762.00 BOOL  ; RK_16 U6_Z 激光焊接Z轴待机位[SW]
762.01 BOOL  ; RK_16 U6_Z 激光焊接Z轴#1移载焊接位[SW]
762.02 BOOL  ; RK_16 U6_Z 激光焊接Z轴#2移载焊接位[SW]
762.03 BOOL  ; 备用[SW]
762.04 BOOL  ; 备用[SW]
762.05 BOOL  ; 备用[SW]
762.06 BOOL  ; 备用[SW]
762.07 BOOL  ; 备用[SW]
762.08 BOOL  ; 备用[SW]
762.09 BOOL  ; 备用[SW]
762.10 BOOL  ; RK_16 U6_Z 激光焊接Z轴回原点[SW]
762.11 BOOL  ; RK_16 U6_Z 激光焊接Z轴JOG+[SW]
762.12 BOOL  ; RK_16 U6_Z 激光焊接Z轴JOG-[SW]
762.13 BOOL  ; RK_16 U6_Z 激光焊接Z轴JOG高速[SW]
762.14 BOOL  ; RK_16 U6_Z 激光焊接Z轴JOG低速[SW]
762.15 BOOL  ; 备用[SW]
763.00 BOOL  ; RK_06 U8_X 电池上下料X轴待机位[SW]
763.01 BOOL  ; RK_06 U8_X 电池上下料X轴铝壳除尘取料位[SW]
763.02 BOOL  ; RK_06 U8_X 电池上下料X轴#1入壳放料位[SW]
763.03 BOOL  ; RK_06 U8_X 电池上下料X轴#2入壳放料位[SW]
763.04 BOOL  ; RK_06 U8_X 电池上下料X轴#1入壳取料位[SW]
763.05 BOOL  ; RK_06 U8_X 电池上下料X轴#2入壳取料位[SW]
763.06 BOOL  ; RK_06 U8_X 电池上下料X轴#1Hipot检测放料位[SW]
763.07 BOOL  ; RK_06 U8_X 电池上下料X轴#2Hipot检测放料位[SW]
763.08 BOOL  ; 备用[SW]
763.09 BOOL  ; 备用[SW]
763.10 BOOL  ; RK_06 U8_X 电池上下料X轴回原点[SW]
763.11 BOOL  ; RK_06 U8_X 电池上下料X轴JOG+[SW]
763.12 BOOL  ; RK_06 U8_X 电池上下料X轴JOG-[SW]
763.13 BOOL  ; RK_06 U8_X 电池上下料X轴JOG高速[SW]
763.14 BOOL  ; RK_06 U8_X 电池上下料X轴JOG低速[SW]
763.15 BOOL  ; 备用[SW]
764.00 BOOL  ; RK_07 U8_Y 铝壳进料X轴等待位[SW]
764.01 BOOL  ; RK_07 U8_Y 铝壳进料X轴取料位[SW]
764.02 BOOL  ; RK_07 U8_Y 铝壳进料X轴放料位[SW]
764.03 BOOL  ; 备用[SW]
764.04 BOOL  ; 备用[SW]
764.05 BOOL  ; 备用[SW]
764.06 BOOL  ; 备用[SW]
764.07 BOOL  ; 备用[SW]
764.08 BOOL  ; 备用[SW]
764.09 BOOL  ; 备用[SW]
764.10 BOOL  ; RK_07 U8_Y 铝壳进料X轴回原点[SW]
764.11 BOOL  ; RK_07 U8_Y 铝壳进料X轴JOG+[SW]
764.12 BOOL  ; RK_07 U8_Y 铝壳进料X轴JOG-[SW]
764.13 BOOL  ; RK_07 U8_Y 铝壳进料X轴JOG高速[SW]
764.14 BOOL  ; RK_07 U8_Y 铝壳进料X轴JOG低速[SW]
764.15 BOOL  ; 备用[SW]
765.00 BOOL  ; RK_07 U8_Z 铝壳上料移载Y轴待料位[SW]
765.01 BOOL  ; RK_07 U8_Z 铝壳上料移载Y轴#1铝壳上料位[SW]
765.02 BOOL  ; RK_07 U8_Z 铝壳上料移载Y轴#2铝壳上料位[SW]
765.03 BOOL  ; RK_07 U8_Z 铝壳上料移载Y轴#3铝壳托盘下料位[SW]
765.04 BOOL  ; RK_07 U8_Z 铝壳上料移载Y轴铝壳取料位[SW]
765.05 BOOL  ; 备用[SW]
765.06 BOOL  ; 备用[SW]
765.07 BOOL  ; 备用[SW]
765.08 BOOL  ; 备用[SW]
765.09 BOOL  ; 备用[SW]
765.10 BOOL  ; RK_07 U8_Z 铝壳上料移载Y轴回原点[SW]
765.11 BOOL  ; RK_07 U8_Z 铝壳上料移载Y轴JOG+[SW]
765.12 BOOL  ; RK_07 U8_Z 铝壳上料移载Y轴JOG-[SW]
765.13 BOOL  ; RK_07 U8_Z 铝壳上料移载Y轴JOG高速[SW]
765.14 BOOL  ; RK_07 U8_Z 铝壳上料移载Y轴JOG低速[SW]
765.15 BOOL  ; 备用[SW]
766.00 BOOL  ; RK_10 U8_U 电池除尘上料X轴待料位[SW]
766.01 BOOL  ; RK_10 U8_U 电池除尘上料X轴#1Hipot检测取料位[SW]
766.02 BOOL  ; RK_10 U8_U 电池除尘上料X轴#2Hipot检测取料位[SW]
766.03 BOOL  ; RK_10 U8_U 电池除尘上料X轴Hipot OK放料位[SW]
766.04 BOOL  ; RK_10 U8_U 电池除尘上料X轴Hipot NG放料位[SW]
766.05 BOOL  ; 备用[SW]
766.06 BOOL  ; 备用[SW]
766.07 BOOL  ; 备用[SW]
766.08 BOOL  ; 备用[SW]
766.09 BOOL  ; 备用[SW]
766.10 BOOL  ; RK_10 U8_U 电池除尘上料X轴回原点[SW]
766.11 BOOL  ; RK_10 U8_U 电池除尘上料X轴JOG+[SW]
766.12 BOOL  ; RK_10 U8_U 电池除尘上料X轴JOG-[SW]
766.13 BOOL  ; RK_10 U8_U 电池除尘上料X轴JOG高速[SW]
766.14 BOOL  ; RK_10 U8_U 电池除尘上料X轴JOG低速[SW]
766.15 BOOL  ; 备用[SW]
787.00 BOOL  ; RK_07 铝壳进料机构X轴当前列数+[SW]
787.01 BOOL  ; RK_07 铝壳进料机构X轴当前列数-[SW]
788.00 BOOL  ; RK_07 铝壳上料移载机构Y轴当前行数+[SW]
788.01 BOOL  ; RK_07 铝壳上料移载机构Y轴当前行数-[SW]
7.00 BOOL  ; 扫码阻挡#1伸出传感器
7.01 BOOL  ; 扫码阻挡#1缩回传感器
7.02 BOOL  ; 扫码阻挡#2伸出传感器
7.03 BOOL  ; 扫码阻挡#2缩回
7.04 BOOL  ; 扫码位有料检测
7.05 BOOL  ; 扫码完成信号
800.00 BOOL  ; RK_02 电芯进料机械手夹爪气缸夹紧位标志[0000.00]
800.01 BOOL  ; RK_02 电芯进料机械手夹爪气缸张开位标志[0000.01]
800.02 BOOL  ; RK_02 电芯进料机械手#1压紧气缸松开位标志[0000.02]
800.03 BOOL  ; RK_02 电芯进料机械手#2压紧气缸松开位标志[0000.03]
800.04 BOOL  ; RK_03 电芯上料机械手夹爪气缸夹紧位标志[0000.04]
800.05 BOOL  ; RK_03 电芯上料机械手夹爪气缸张开位标志[0000.05]
800.06 BOOL  ; RK_03 电芯上料机械手#1压紧气缸松开位标志[0000.06]
800.07 BOOL  ; RK_03 电芯上料机械手#2压紧气缸松开位标志[0000.07]
800.08 BOOL  ; RK_03 电芯上料升降气缸下降位标志[0000.08]
800.09 BOOL  ; RK_03 电芯上料升降气缸上升位标志[0000.09]
800.10 BOOL  ; RK_04 电芯除尘伸缩气缸缩回位标志[0000.10]
800.11 BOOL  ; RK_04 电芯除尘伸缩气缸伸出位标志[0000.11]
800.12 BOOL  ; RK_05 #1入壳滚轮夹紧气缸夹紧位标志[0000.12]
800.13 BOOL  ; RK_05 #1入壳滚轮夹紧气缸松开位标志[0000.13]
800.14 BOOL  ; RK_05 #1入壳铝壳定位平台伸缩气缸缩回位标志[0000.14]
800.15 BOOL  ; RK_05 #1入壳铝壳定位平台伸缩气缸伸出位标志[0000.15]
801.00 BOOL  ; RK_05 #1入壳铝壳定位平台升降气缸上升位标志[0001.00]
801.01 BOOL  ; RK_05 #1入壳铝壳定位平台升降气缸下降位标志[0001.01]
801.02 BOOL  ; RK_05 #1入壳铝壳定位伸缩气缸缩回位标志[0001.02]
801.03 BOOL  ; RK_05 #1入壳铝壳定位伸缩气缸伸出位标志[0001.03]
801.04 BOOL  ; RK_05 #1入壳铝壳定位夹爪气缸夹紧位标志[0001.04]
801.05 BOOL  ; RK_05 #1入壳铝壳定位夹爪气缸张开位标志[0001.05]
801.06 BOOL  ; RK_05 #2入壳滚轮夹紧气缸夹紧位标志[0001.06]
801.07 BOOL  ; RK_05 #2入壳滚轮夹紧气缸松开位标志[0001.07]
801.08 BOOL  ; RK_05 #2入壳铝壳定位平台伸缩气缸缩回位标志[0001.08]
801.09 BOOL  ; RK_05 #2入壳铝壳定位平台伸缩气缸伸出位标志[0001.09]
801.10 BOOL  ; RK_05 #2入壳铝壳定位平台升降气缸上升位标志[0001.10]
801.11 BOOL  ; RK_05 #2入壳铝壳定位平台升降气缸下降位标志[0001.11]
801.12 BOOL  ; RK_05 #2入壳铝壳定位伸缩气缸缩回位标志[0001.12]
801.13 BOOL  ; RK_05 #2入壳铝壳定位伸缩气缸伸出位标志[0001.13]
801.14 BOOL  ; RK_05 #2入壳铝壳定位夹爪气缸夹紧位标志[0001.14]
801.15 BOOL  ; RK_05 #2入壳铝壳定位夹爪气缸张开位标志[0001.15]
802.00 BOOL  ; RK_01 U0_X 电芯来料Y轴报警信号标志[0002.00]
802.01 BOOL  ; RK_01 U0_X 电芯来料Y轴准备好了信号标志[0002.01]
802.02 BOOL  ; RK_02 U0_Y 电芯进料X轴报警信号标志[0002.02]
802.03 BOOL  ; RK_02 U0_Y 电芯进料X轴准备好了信号标志[0002.03]
802.04 BOOL  ; RK_02 U0_Z 电芯进料Z轴报警信号标志[0002.04]
802.05 BOOL  ; RK_02 U0_Z 电芯进料Z轴准备好了信号标志[0002.05]
802.06 BOOL  ; RK_03 U0_U 电芯上料X轴报警信号标志[0002.06]
802.07 BOOL  ; RK_03 U0_U 电芯上料X轴准备好了信号标志[0002.07]
802.08 BOOL  ; RK_05 U2_X #1入壳Y轴报警信号标志[0002.08]
802.09 BOOL  ; RK_05 U2_X #1入壳Y轴准备好了信号标志[0002.09]
802.10 BOOL  ; RK_05 U2_Y #2入壳Y轴报警信号标志[0002.10]
802.11 BOOL  ; RK_05 U2_Y #2入壳Y轴准备好了信号标志[0002.11]
802.12 BOOL  ; 0标志[0002.12]
802.13 BOOL  ; RK_05 #1入壳定位陶瓷棒上#1夹紧气缸伸出位标志[0002.13]
802.14 BOOL  ; RK_05 #1入壳定位陶瓷棒上#2夹紧气缸伸出位标志[0002.14]
802.15 BOOL  ; RK_05 #1入壳定位陶瓷棒下#1夹紧气缸伸出位标志[0002.15]
803.00 BOOL  ; RK_05 #1入壳定位陶瓷棒下#2夹紧气缸伸出位标志[0003.00]
803.01 BOOL  ; RK_05 #1入壳定位陶瓷棒上#1夹紧气缸缩回位标志[0003.01]
803.02 BOOL  ; RK_05 #1入壳定位陶瓷棒上#2夹紧气缸缩回位标志[0003.02]
803.03 BOOL  ; RK_05 #1入壳定位陶瓷棒下#1夹紧气缸缩回位标志[0003.03]
803.04 BOOL  ; RK_05 #1入壳定位陶瓷棒下#2夹紧气缸缩回位标志[0003.04]
803.05 BOOL  ; RK_05 #1入壳吸盘上#1伸缩气缸缩回位标志[0003.05]
803.06 BOOL  ; RK_05 #1入壳吸盘上#2伸缩气缸缩回位标志[0003.06]
803.07 BOOL  ; RK_05 #1入壳吸盘上#3伸缩气缸缩回位标志[0003.07]
803.08 BOOL  ; RK_05 #1入壳吸盘下#1伸缩气缸缩回位标志[0003.08]
803.09 BOOL  ; RK_05 #1入壳吸盘下#2伸缩气缸缩回位标志[0003.09]
803.10 BOOL  ; RK_05 #1入壳吸盘下#3伸缩气缸缩回位标志[0003.10]
803.11 BOOL  ; RK_05 #1入壳电芯#1定位夹爪气缸松开位标志[0003.11]
803.12 BOOL  ; RK_05 #1入壳电芯#2定位夹爪气缸松开位标志[0003.12]
803.13 BOOL  ; RK_05 #1入壳电芯#1定位夹爪气缸夹紧位标志[0003.13]
803.14 BOOL  ; RK_05 #1入壳电芯#2定位夹爪气缸夹紧位标志[0003.14]
803.15 BOOL  ; RK_05 #2入壳定位陶瓷棒上#1夹紧气缸伸出位标志[0003.15]
804.00 BOOL  ; RK_05 #2入壳定位陶瓷棒上#2夹紧气缸伸出位标志[0004.00]
804.01 BOOL  ; RK_05 #2入壳定位陶瓷棒下#1夹紧气缸伸出位标志[0004.01]
804.02 BOOL  ; RK_05 #2入壳定位陶瓷棒下#2夹紧气缸伸出位标志[0004.02]
804.03 BOOL  ; RK_05 #2入壳定位陶瓷棒上#1夹紧气缸缩回位标志[0004.03]
804.04 BOOL  ; RK_05 #2入壳定位陶瓷棒上#2夹紧气缸缩回位标志[0004.04]
804.05 BOOL  ; RK_05 #2入壳定位陶瓷棒下#1夹紧气缸缩回位标志[0004.05]
804.06 BOOL  ; RK_05 #2入壳定位陶瓷棒下#2夹紧气缸缩回位标志[0004.06]
804.07 BOOL  ; RK_05 #2入壳吸盘上#1伸缩气缸缩回位标志[0004.07]
804.08 BOOL  ; RK_05 #2入壳吸盘上#2伸缩气缸缩回位标志[0004.08]
804.09 BOOL  ; RK_05 #2入壳吸盘上#3伸缩气缸缩回位标志[0004.09]
804.10 BOOL  ; RK_05 #2入壳吸盘下#1伸缩气缸缩回位标志[0004.10]
804.11 BOOL  ; RK_05 #2入壳吸盘下#2伸缩气缸缩回位标志[0004.11]
804.12 BOOL  ; RK_05 #2入壳吸盘下#3伸缩气缸缩回位标志[0004.12]
804.13 BOOL  ; RK_05 #2入壳电芯#1定位夹爪气缸松开位标志[0004.13]
804.14 BOOL  ; RK_05 #2入壳电芯#2定位夹爪气缸松开位标志[0004.14]
804.15 BOOL  ; RK_05 #2入壳电芯#1定位夹爪气缸夹紧位标志[0004.15]
805.00 BOOL  ; RK_05 #2入壳电芯#2定位夹爪气缸夹紧位标志[0005.00]
805.01 BOOL  ; RK_01 电芯来料有料感应标志[0005.01]
805.02 BOOL  ; RK_02 电芯进料机械手夹爪柔性报警标志[0005.02]
805.03 BOOL  ; RK_03 电芯上料机械手夹爪柔性报警标志[0005.03]
805.04 BOOL  ; RK_04 电芯除尘有料感应标志[0005.04]
805.05 BOOL  ; RK_02 扫码NG拉带有料感应#1标志[0005.05]
805.06 BOOL  ; RK_02 扫码NG拉带有料感应#2标志[0005.06]
805.07 BOOL  ; RK_02 扫码NG拉带料满感应标志[0005.07]
805.08 BOOL  ; RK_05 #1入壳电芯有料感应标志[0005.08]
805.09 BOOL  ; RK_05 #1入壳铝壳有料感应标志[0005.09]
805.10 BOOL  ; RK_05 #2入壳电芯有料感应标志[0005.10]
805.11 BOOL  ; RK_05 #2入壳铝壳有料感应标志[0005.11]
805.12 BOOL  ; RK_05 #1入壳吸盘真空标志[0005.12]
805.13 BOOL  ; RK_05 #2入壳吸盘真空标志[0005.13]
805.14 BOOL  ; 前端设备对接输入信号（公共）标志[0005.14]
805.15 BOOL  ; 后端设备对接输入信号（公共）标志[0005.15]
806.00 BOOL  ; 小屏插入信号（公共）标志[0006.00]
806.01 BOOL  ; NC433模块DC5V电源信号（公共）标志[0006.01]
806.02 BOOL  ; DC24V伺服刹车电源信号（公共）标志[0006.02]
806.03 BOOL  ; 出料端急停（公共）标志[0006.03]
806.04 BOOL  ; 小移动屏急停（公共）标志[0006.04]
806.05 BOOL  ; A机架#1门磁（公共）标志[0006.05]
806.06 BOOL  ; A机架#2门磁（公共）标志[0006.06]
806.07 BOOL  ; A机架#3门磁（公共）标志[0006.07]
806.08 BOOL  ; A机架#4门磁（公共）标志[0006.08]
806.09 BOOL  ; A机架#5门磁（公共）标志[0006.09]
806.10 BOOL  ; A机架#6门磁（公共）标志[0006.10]
806.11 BOOL  ; A机架#7门磁（公共）标志[0006.11]
806.12 BOOL  ; A机架#8门磁（公共）标志[0006.12]
806.13 BOOL  ; A机架#9门磁（公共）标志[0006.13]
806.14 BOOL  ; RK_01 电芯来料上料位有料感应标志[0006.14]
806.15 BOOL  ; 0标志[0006.15]
807.00 BOOL  ; 0标志[0007.00]
807.01 BOOL  ; 0标志[0007.01]
807.02 BOOL  ; 0标志[0007.02]
807.03 BOOL  ; 0标志[0007.03]
807.04 BOOL  ; 0标志[0007.04]
807.05 BOOL  ; 0标志[0007.05]
807.06 BOOL  ; 0标志[0007.06]
807.07 BOOL  ; 0标志[0007.07]
807.08 BOOL  ; 0标志[0007.08]
807.09 BOOL  ; 0标志[0007.09]
807.10 BOOL  ; 0标志[0007.10]
807.11 BOOL  ; 0标志[0007.11]
807.12 BOOL  ; 0标志[0007.12]
807.13 BOOL  ; 0标志[0007.13]
807.14 BOOL  ; 0标志[0007.14]
807.15 BOOL  ; 0标志[0007.15]
808.00 BOOL  ; RK_11 电池除尘旋转伸缩气缸到位标志[0008.00]
808.01 BOOL  ; RK_11 电池除尘旋转伸缩气缸原位标志[0008.01]
808.02 BOOL  ; RK_11 电池除尘伸缩气缸伸出位标志[0008.02]
808.03 BOOL  ; RK_11 电池除尘伸缩气缸缩回位标志[0008.03]
808.04 BOOL  ; RK_11 电池除尘夹爪气缸夹紧位标志[0008.04]
808.05 BOOL  ; RK_11 电池除尘夹爪气缸张开位标志[0008.05]
808.06 BOOL  ; RK_12 预焊上料机械手夹爪气缸夹紧位标志[0008.06]
808.07 BOOL  ; RK_12 预焊上料机械手夹爪气缸张开位标志[0008.07]
808.08 BOOL  ; RK_12 预焊下料机械手夹爪气缸夹紧位标志[0008.08]
808.09 BOOL  ; RK_12 预焊下料机械手夹爪气缸张开位标志[0008.09]
808.10 BOOL  ; RK_13 #1移载升降气缸上升位标志[0008.10]
808.11 BOOL  ; RK_13 #1移载升降气缸下降位标志[0008.11]
808.12 BOOL  ; RK_13 #1移载定位#1伸缩气缸缩回位标志[0008.12]
808.13 BOOL  ; RK_13 #1移载定位#1伸缩气缸伸出位标志[0008.13]
808.14 BOOL  ; RK_13 #1移载定位#2伸缩气缸缩回位标志[0008.14]
808.15 BOOL  ; RK_13 #1移载定位#2伸缩气缸伸出位标志[0008.15]
809.00 BOOL  ; RK_13 #1移载导向#1伸缩气缸伸出位标志[0009.00]
809.01 BOOL  ; RK_13 #1移载导向#1伸缩气缸缩回位标志[0009.01]
809.02 BOOL  ; RK_13 #1移载导向#2伸缩气缸伸出位标志[0009.02]
809.03 BOOL  ; RK_13 #1移载导向#2伸缩气缸缩回位标志[0009.03]
809.04 BOOL  ; RK_13 #1移载左右定位伸缩气缸伸出位标志[0009.04]
809.05 BOOL  ; RK_13 #1移载左右定位伸缩气缸缩回位标志[0009.05]
809.06 BOOL  ; RK_13 #2移载升降气缸上升位标志[0009.06]
809.07 BOOL  ; RK_13 #2移载升降气缸下降位标志[0009.07]
809.08 BOOL  ; RK_13 #2移载定位#1伸缩气缸缩回位标志[0009.08]
809.09 BOOL  ; RK_13 #2移载定位#1伸缩气缸伸出位标志[0009.09]
809.10 BOOL  ; RK_13 #2移载定位#2伸缩气缸缩回位标志[0009.10]
809.11 BOOL  ; RK_13 #2移载定位#2伸缩气缸伸出位标志[0009.11]
809.12 BOOL  ; RK_13 #2移载导向#1伸缩气缸伸出位标志[0009.12]
809.13 BOOL  ; RK_13 #2移载导向#1伸缩气缸缩回位标志[0009.13]
809.14 BOOL  ; RK_13 #2移载导向#2伸缩气缸伸出位标志[0009.14]
809.15 BOOL  ; RK_13 #2移载导向#2伸缩气缸缩回位标志[0009.15]
810.00 BOOL  ; RK_13 #2移载左右定位伸缩气缸伸出位标志[0010.00]
810.01 BOOL  ; RK_13 #2移载左右定位伸缩气缸缩回位标志[0010.01]
810.02 BOOL  ; RK_14 #1压装升降气缸下降位标志[0010.02]
810.03 BOOL  ; RK_14 #1压装升降气缸上升位标志[0010.03]
810.04 BOOL  ; RK_14 #1压装#1吸盘升降气缸下降位标志[0010.04]
810.05 BOOL  ; RK_14 #1压装#1吸盘升降气缸上升位标志[0010.05]
810.06 BOOL  ; RK_14 #1压装#2吸盘升降气缸下降位标志[0010.06]
810.07 BOOL  ; RK_14 #1压装#2吸盘升降气缸上升位标志[0010.07]
810.08 BOOL  ; RK_14 #2压装升降气缸下降位标志[0010.08]
810.09 BOOL  ; RK_14 #2压装升降气缸上升位标志[0010.09]
810.10 BOOL  ; RK_14 #2压装#1吸盘升降气缸下降位标志[0010.10]
810.11 BOOL  ; RK_14 #2压装#1吸盘升降气缸上升位标志[0010.11]
810.12 BOOL  ; RK_14 #2压装#2吸盘升降气缸下降位标志[0010.12]
810.13 BOOL  ; RK_14 #2压装#2吸盘升降气缸上升位标志[0010.13]
810.14 BOOL  ; RK_15 轮廓检测#1伸缩气缸伸出位标志[0010.14]
810.15 BOOL  ; RK_15 轮廓检测#1伸缩气缸缩回位标志[0010.15]
811.00 BOOL  ; RK_15 轮廓检测#2伸缩气缸伸出位标志[0011.00]
811.01 BOOL  ; RK_15 轮廓检测#2伸缩气缸缩回位标志[0011.01]
811.02 BOOL  ; RK_12 轮廓检测NG拨料气缸伸出位标志[0011.02]
811.03 BOOL  ; RK_12 轮廓检测NG拨料气缸缩回位标志[0011.03]
811.04 BOOL  ; RK_11 电池除尘有料感应标志[0011.04]
811.05 BOOL  ; RK_12 预焊上料机械手夹爪柔性报警标志[0011.05]
811.06 BOOL  ; RK_12 预焊下料机械手夹爪柔性报警标志[0011.06]
811.07 BOOL  ; RK_16 激光焊接完成信号标志[0011.07]
811.08 BOOL  ; RK_16 激光焊机故障信号标志[0011.08]
811.09 BOOL  ; RK_13 #1移载电池顶盖超高检测标志[0011.09]
811.10 BOOL  ; RK_16 激光焊机急停信号标志[0011.10]
811.11 BOOL  ; RK_13 #2移载电池顶盖超高检测标志[0011.09]
811.12 BOOL  ; RK_13 #1移载有料感应标志[0011.12]
811.13 BOOL  ; RK_13 #2移载有料感应标志[0011.13]
811.14 BOOL  ; RK_14 #1压装吸盘真空标志[0011.14]
811.15 BOOL  ; RK_14 #2压装吸盘真空标志[0011.15]
812.00 BOOL  ; RK_12 U4_X 预焊上下料X轴报警信号标志[0012.00]
812.01 BOOL  ; RK_12 U4_X 预焊上下料X轴准备好了信号标志[0012.01]
812.02 BOOL  ; RK_12 U4_Y 预焊上料Z轴报警信号标志[0012.02]
812.03 BOOL  ; RK_12 U4_Y 预焊上料Z轴准备好了信号标志[0012.03]
812.04 BOOL  ; RK_12 U4_Z 预焊下料Z轴报警信号标志[0012.04]
812.05 BOOL  ; RK_12 U4_Z 预焊下料Z轴准备好了信号标志[0012.05]
812.06 BOOL  ; RK_13 U4_U #1移载Y轴报警信号标志[0012.06]
812.07 BOOL  ; RK_13 U4_U #1移载Y轴准备好了信号标志[0012.07]
812.08 BOOL  ; RK_13 U6_X #2移载Y轴报警信号标志[0012.08]
812.09 BOOL  ; RK_13 U6_X #2移载Y轴准备好了信号标志[0012.09]
812.10 BOOL  ; RK_16 U6_Y 激光焊接X轴报警信号标志[0012.10]
812.11 BOOL  ; RK_16 U6_Y 激光焊接X轴准备好了信号标志[0012.11]
812.12 BOOL  ; RK_16 U6_Z 激光焊接Z轴报警信号标志[0012.12]
812.13 BOOL  ; RK_16 U6_Z 激光焊接Z轴准备好了信号标志[0012.13]
812.14 BOOL  ; 0标志[0012.14]
812.15 BOOL  ; 0标志[0012.15]
813.00 BOOL  ; 0标志[0013.00]
813.01 BOOL  ; RK_12 轮廓检测NG料槽#1有料感应标志[0013.01]
813.02 BOOL  ; RK_12 轮廓检测NG料槽#1料满感应标志[0013.02]
813.03 BOOL  ; RK_12 轮廓检测NG料槽#2有料感应标志[0013.03]
813.04 BOOL  ; RK_12 轮廓检测NG料槽#2料满感应标志[0013.04]
813.05 BOOL  ; RK_12 OK出料拉带放料位有料感应#1标志[0013.05]
813.06 BOOL  ; RK_12 OK出料拉带放料位有料感应#2标志[0013.06]
813.07 BOOL  ; RK_12 OK出料拉带出料位有料感应标志[0013.07]
813.08 BOOL  ; 0标志[0013.08]
813.09 BOOL  ; 0标志[0013.09]
813.10 BOOL  ; 0标志[0013.10]
813.11 BOOL  ; 0标志[0013.11]
813.12 BOOL  ; 0标志[0013.12]
813.13 BOOL  ; 0标志[0013.13]
813.14 BOOL  ; 0标志[0013.14]
813.15 BOOL  ; 0标志[0013.15]
814.00 BOOL  ; RK_06 铝壳上料升降气缸下降位标志[0014.00]
814.01 BOOL  ; RK_06 铝壳上料升降气缸上升位标志[0014.01]
814.02 BOOL  ; RK_06 电池下料升降气缸下降位标志[0014.02]
814.03 BOOL  ; RK_06 电池下料升降气缸上升位标志[0014.03]
814.04 BOOL  ; RK_06 铝壳上料夹爪气缸夹紧位标志[0014.04]
814.05 BOOL  ; RK_06 铝壳上料夹爪气缸张开位标志[0014.05]
814.06 BOOL  ; RK_06 电池下料夹爪气缸夹紧位标志[0014.06]
814.07 BOOL  ; RK_06 电池下料夹爪气缸张开位标志[0014.07]
814.08 BOOL  ; RK_07 #1铝壳上料车定位升降气缸上升位标志[0014.08]
814.09 BOOL  ; RK_07 #1铝壳上料车定位升降气缸下降位标志[0014.09]
814.10 BOOL  ; RK_07 #2铝壳上料车定位升降气缸上升位标志[0014.10]
814.11 BOOL  ; RK_07 #2铝壳上料车定位升降气缸下降位标志[0014.11]
814.12 BOOL  ; RK_07 #3托盘下料车定位升降气缸上升位标志[0014.12]
814.13 BOOL  ; RK_07 #3托盘下料车定位升降气缸下降位标志[0014.13]
814.14 BOOL  ; RK_07 铝壳进料机械手升降气缸下降位标志[0014.14]
814.15 BOOL  ; $?St$Bk?_#[5050] / RK_07 铝壳进料机械手升降气缸上升位标志[0014.15] / $?St$Bk?_#[5050]
815.00 BOOL  ; RK_08 铝壳除尘旋转伸缩气缸原位标志[0015.00]
815.01 BOOL  ; RK_08 铝壳除尘旋转伸缩气缸到位标志[0015.01]
815.02 BOOL  ; RK_08 铝壳除尘伸缩气缸伸出位标志[0015.02]
815.03 BOOL  ; RK_08 铝壳除尘伸缩气缸缩回位标志[0015.03]
815.04 BOOL  ; RK_08 铝壳除尘夹爪气缸夹紧位标志[0015.04]
815.05 BOOL  ; RK_08 铝壳除尘夹爪气缸张开位标志[0015.05]
815.06 BOOL  ; RK_09 #1Hipot测试旋转伸缩气缸到位标志[0015.06]
815.07 BOOL  ; RK_09 #1Hipot测试旋转伸缩气缸原位标志[0015.07]
815.08 BOOL  ; RK_09 #1Hipot测试平台伸缩气缸缩回位标志[0015.08]
815.09 BOOL  ; RK_09 #1Hipot测试平台伸缩气缸伸出位标志[0015.09]
815.10 BOOL  ; RK_09 #1Hipot测试伸缩气缸伸出位标志[0015.10]
815.11 BOOL  ; RK_09 #1Hipot测试伸缩气缸缩回位标志[0015.11]
815.12 BOOL  ; RK_09 #2Hipot测试旋转伸缩气缸到位标志[0015.12]
815.13 BOOL  ; RK_09 #2Hipot测试旋转伸缩气缸原位标志[0015.13]
815.14 BOOL  ; RK_09 #2Hipot测试平台伸缩气缸缩回位标志[0015.14]
815.15 BOOL  ; RK_09 #2Hipot测试平台伸缩气缸伸出位标志[0015.15]
816.00 BOOL  ; RK_09 #2Hipot测试伸缩气缸伸出位标志[0016.00]
816.01 BOOL  ; RK_09 #2Hipot测试伸缩气缸缩回位标志[0016.01]
816.02 BOOL  ; RK_10 电池除尘上料机械手升降气缸下降位标志[0016.02]
816.03 BOOL  ; RK_10 电池除尘上料机械手升降气缸上升位标志[0016.03]
816.04 BOOL  ; RK_10 电池除尘上料机械手夹爪气缸夹紧位标志[0016.04]
816.05 BOOL  ; RK_10 电池除尘上料机械手夹爪气缸张开位标志[0016.05]
816.06 BOOL  ; RK_06 U8_X 电池上下料X轴报警信号标志[0016.06]
816.07 BOOL  ; RK_06 U8_X 电池上下料X轴准备好了信号标志[0016.07]
816.08 BOOL  ; RK_07 U8_Y 铝壳进料X轴报警信号标志[0016.08]
816.09 BOOL  ; RK_07 U8_Y 铝壳进料X轴准备好了信号标志[0016.09]
816.10 BOOL  ; RK_07 U8_Z 铝壳上料移载Y轴报警信号标志[0016.10]
816.11 BOOL  ; RK_07 U8_Z 铝壳上料移载Y轴准备好了信号标志[0016.11]
816.12 BOOL  ; RK_10 U8_U 电池除尘上料X轴报警信号标志[0016.12]
816.13 BOOL  ; RK_10 U8_U 电池除尘上料X轴准备好了信号标志[0016.13]
816.14 BOOL  ; RK_09 Hipot测试完成信号标志[0016.14]
816.15 BOOL  ; RK_07 #1铝壳上料启动按钮标志[0016.15]
817.00 BOOL  ; RK_07 #2铝壳上料启动按钮标志[0017.00]
817.01 BOOL  ; RK_07 #3托盘下料启动按钮标志[0017.01]
817.02 BOOL  ; RK_07 铝壳上料移载吸盘真空标志[0017.02]
817.03 BOOL  ; RK_07 铝壳进料吸盘真空标志[0017.03]
817.04 BOOL  ; RK_07 #1铝壳上料托盘到位感应标志[0017.04]
817.05 BOOL  ; RK_07 #1铝壳上料位物料车到位感应标志[0017.05]
817.06 BOOL  ; RK_07 #1铝壳上料初始位（#1）标志[0017.06]
817.07 BOOL  ; RK_07 #1铝壳上料一个托盘位（#2）标志[0017.07]
817.08 BOOL  ; RK_07 #1铝壳上料高限位（#3）标志[0017.08]
817.09 BOOL  ; RK_07 #2铝壳上料托盘到位感应标志[0017.09]
817.10 BOOL  ; RK_07 #2铝壳上料位物料车到位感应标志[0017.10]
817.11 BOOL  ; RK_07 #2铝壳上料初始位（#1）标志[0017.11]
817.12 BOOL  ; RK_07 #2铝壳上料一个托盘位（#2）标志[0017.12]
817.13 BOOL  ; RK_07 #2铝壳上料高限位（#3）标志[0017.13]
817.14 BOOL  ; RK_07 #3托盘下料上升到位感应标志[0017.14]
817.15 BOOL  ; RK_07 #3托盘下料位物料车到位感应标志[0017.15]
818.00 BOOL  ; RK_07 #3托盘下料初始位（#1）标志[0018.00]
818.01 BOOL  ; RK_07 #3托盘下料满托盘位（#2）标志[0018.01]
818.02 BOOL  ; RK_07 #3托盘下料高限位（#3）标志[0018.02]
818.03 BOOL  ; RK_07 铝壳上料移载托盘到位感应标志[0018.03]
818.04 BOOL  ; RK_08 铝壳除尘有料感应标志[0018.04]
818.05 BOOL  ; RK_09 #1Hipot测试有料感应标志[0018.05]
818.06 BOOL  ; RK_09 #2Hipot测试有料感应标志[0018.06]
818.07 BOOL  ; RK_10 Hipot检测NG拉带有料感应#1标志[0018.07]
818.08 BOOL  ; RK_10 Hipot检测NG拉带有料感应#2标志[0018.08]
818.09 BOOL  ; RK_10 Hipot检测NG拉带料满感应标志[0018.09]
818.10 BOOL  ; RK_06 铝壳上料夹爪柔性报警标志[0018.10]
818.11 BOOL  ; RK_06 电池下料夹爪柔性报警标志[0018.11]
818.12 BOOL  ; RK_07 铝壳进料机械手柔性报警标志[0018.12]
818.13 BOOL  ; RK_10 电池除尘上料机械手夹爪柔性报警标志[0018.13]
818.14 BOOL  ; 手/自动选择（公共）标志[0018.14]
818.15 BOOL  ; 启动按钮_绿（公共）标志[0018.15]
819.00 BOOL  ; 停止按钮_红（公共）标志[0019.00]
819.01 BOOL  ; 复位按钮_黄（公共）标志[0019.01]
819.02 BOOL  ; 机台进气压力（正压）（公共）标志[0019.02]
819.03 BOOL  ; 机台进气压力（负压）（公共）标志[0019.03]
819.04 BOOL  ; 主屏急停（公共）标志[0019.04]
819.05 BOOL  ; 铝壳上料端急停（公共）标志[0019.05]
819.06 BOOL  ; HipotNG端急停（公共）标志[0019.06]
819.07 BOOL  ; B机架#1门磁（公共）标志[0019.07]
819.08 BOOL  ; B机架#2门磁（公共）标志[0019.08]
819.09 BOOL  ; B机架#3门磁（公共）标志[0019.09]
819.10 BOOL  ; B机架#4门磁（公共）标志[0019.10]
819.11 BOOL  ; B机架#5门磁（公共）标志[0019.11]
819.12 BOOL  ; B机架#6门磁（公共）标志[0019.12]
819.13 BOOL  ; RK_07 #3托盘下料下降到位感应标志[0019.13]
819.14 BOOL  ; RK_07 #3托盘下料位物料车到位感应#2标志[0019.14]
819.15 BOOL  ; RK_07 铝壳上料移载托盘到位保护感应标志[0019.15]
820.02 BOOL  ; RK_02 电芯进料机械手#1压紧气缸压紧位标志
820.03 BOOL  ; RK_02 电芯进料机械手#2压紧气缸压紧位标志
820.06 BOOL  ; RK_03 电芯上料机械手#1压紧气缸压紧位标志
820.07 BOOL  ; RK_03 电芯上料机械手#2压紧气缸压紧位标志
823.05 BOOL  ; RK_05 #1入壳吸盘上#1伸缩气缸伸出位标志
823.06 BOOL  ; RK_05 #1入壳吸盘上#2伸缩气缸伸出位标志
823.07 BOOL  ; RK_05 #1入壳吸盘上#3伸缩气缸伸出位标志
823.08 BOOL  ; RK_05 #1入壳吸盘下#1伸缩气缸伸出位标志
823.09 BOOL  ; RK_05 #1入壳吸盘下#2伸缩气缸伸出位标志
823.10 BOOL  ; RK_05 #1入壳吸盘下#3伸缩气缸伸出位标志
824.07 BOOL  ; RK_05 #2入壳吸盘上#1伸缩气缸伸出位标志
824.08 BOOL  ; RK_05 #2入壳吸盘上#2伸缩气缸伸出位标志
824.09 BOOL  ; RK_05 #2入壳吸盘上#3伸缩气缸伸出位标志
824.10 BOOL  ; RK_05 #2入壳吸盘下#1伸缩气缸伸出位标志
824.11 BOOL  ; RK_05 #2入壳吸盘下#2伸缩气缸伸出位标志
824.12 BOOL  ; RK_05 #2入壳吸盘下#3伸缩气缸伸出位标志
850.00 BOOL  ; RK_01 U0_X 电芯来料Y轴待料位标志
850.01 BOOL  ; RK_01 U0_X 电芯来料Y轴上料位标志
850.02 BOOL  ; RK_01 U0_X 电芯来料Y轴扫码位标志
850.03 BOOL  ; RK_01 U0_X 电芯来料Y轴下料位标志
851.00 BOOL  ; RK_02 U0_Y 电芯进料X轴待料位标志
851.01 BOOL  ; RK_02 U0_Y 电芯进料X轴取料位标志
851.02 BOOL  ; RK_02 U0_Y 电芯进料X轴扫码OK放料位标志
851.03 BOOL  ; RK_02 U0_Y 电芯进料X轴扫码NG放料位标志
852.00 BOOL  ; RK_02 U0_Z 电芯进料Z轴待料位（扫码）标志
852.01 BOOL  ; RK_02 U0_Z 电芯进料Z轴取料位标志
852.02 BOOL  ; RK_02 U0_Z 电芯进料Z轴扫码OK放料位标志
852.03 BOOL  ; RK_02 U0_Z 电芯进料Z轴扫码NG放料位标志
852.04 BOOL  ; RK_02 U0_Z 电芯进料Z轴扫码位标志
853.00 BOOL  ; RK_03 U0_U 电芯上料X轴待料位标志
853.01 BOOL  ; RK_03 U0_U 电芯上料X轴取料位标志
853.02 BOOL  ; RK_03 U0_U 电芯上料X轴#1入壳放料位标志
853.03 BOOL  ; RK_03 U0_U 电芯上料X轴#2入壳放料位标志
854.00 BOOL  ; RK_05 U2_X #1入壳Y轴待料位标志
854.01 BOOL  ; RK_05 U2_X #1入壳Y轴滚轮压紧位标志
854.02 BOOL  ; RK_05 U2_X #1入壳Y轴滚轮松开位标志
854.03 BOOL  ; RK_05 U2_X #1入壳Y轴入壳位标志
854.04 BOOL  ; RK_05 U2_X #1入壳Y轴电芯定位夹爪松开位标志
855.00 BOOL  ; RK_05 U2_Y #2入壳Y轴待料位标志
855.01 BOOL  ; RK_05 U2_Y #2入壳Y轴滚轮压紧位标志
855.02 BOOL  ; RK_05 U2_Y #2入壳Y轴滚轮松开位标志
855.03 BOOL  ; RK_05 U2_Y #2入壳Y轴入壳位标志
855.04 BOOL  ; RK_05 U2_Y #2入壳Y轴电芯定位夹爪松开位标志
856.00 BOOL  ; RK_12 U4_X 预焊上下料X轴待料位标志
856.01 BOOL  ; RK_12 U4_X 预焊上下料X轴除尘取料位标志
856.02 BOOL  ; RK_12 U4_X 预焊上下料X轴#1移载放料位标志
856.03 BOOL  ; RK_12 U4_X 预焊上下料X轴#2移载放料位标志
856.04 BOOL  ; RK_12 U4_X 预焊上下料X轴#1移载取料位标志
856.05 BOOL  ; RK_12 U4_X 预焊上下料X轴#2移载取料位标志
856.06 BOOL  ; RK_12 U4_X 预焊上下料X轴OK放料位标志
856.07 BOOL  ; RK_12 U4_X 预焊上下料X轴#1NG放料位标志
856.08 BOOL  ; RK_12 U4_X 预焊上下料X轴#2NG放料位标志
857.00 BOOL  ; RK_12 U4_Y 预焊上料Z轴待料位标志
857.01 BOOL  ; RK_12 U4_Y 预焊上料Z轴除尘取料位标志
857.02 BOOL  ; RK_12 U4_Y 预焊上料Z轴#1移载放料位标志
857.03 BOOL  ; RK_12 U4_Y 预焊上料Z轴#2移载放料位标志
858.00 BOOL  ; RK_12 U4_Z 预焊下料Z轴待料位标志
858.01 BOOL  ; RK_12 U4_Z 预焊下料Z轴#1移载取料位标志
858.02 BOOL  ; RK_12 U4_Z 预焊下料Z轴#2移载取料位标志
858.03 BOOL  ; RK_12 U4_Z 预焊下料Z轴OK放料位标志
858.04 BOOL  ; RK_12 U4_Z 预焊下料Z轴#1NG放料位标志
858.05 BOOL  ; RK_12 U4_Z 预焊下料Z轴#2NG放料位标志
859.00 BOOL  ; RK_13 U4_U #1移载Y轴待料位标志
859.01 BOOL  ; RK_13 U4_U #1移载Y轴取放料位标志
859.02 BOOL  ; RK_13 U4_U #1移载Y轴压装位标志
859.03 BOOL  ; RK_13 U4_U #1移载Y轴#1轮廓检测位标志
859.04 BOOL  ; RK_13 U4_U #1移载Y轴#2轮廓检测位标志
859.05 BOOL  ; RK_13 U4_U #1移载Y轴激光焊接位标志
860.00 BOOL  ; RK_13 U6_X #2移载Y轴待料位标志
860.01 BOOL  ; RK_13 U6_X #2移载Y轴取放料位标志
860.02 BOOL  ; RK_13 U6_X #2移载Y轴压装位标志
860.03 BOOL  ; RK_13 U6_X #2移载Y轴#1轮廓检测位标志
860.04 BOOL  ; RK_13 U6_X #2移载Y轴#2轮廓检测位标志
860.05 BOOL  ; RK_13 U6_X #2移载Y轴激光焊接位标志
861.00 BOOL  ; RK_16 U6_Y 激光焊接X轴待机位标志
861.01 BOOL  ; RK_16 U6_Y 激光焊接X轴#1移载焊接位标志
861.02 BOOL  ; RK_16 U6_Y 激光焊接X轴#2移载焊接位标志
862.00 BOOL  ; RK_16 U6_Z 激光焊接Z轴待机位标志
862.01 BOOL  ; RK_16 U6_Z 激光焊接Z轴#1移载焊接位标志
862.02 BOOL  ; RK_16 U6_Z 激光焊接Z轴#2移载焊接位标志
863.00 BOOL  ; RK_06 U8_X 电池上下料X轴待机位标志
863.01 BOOL  ; RK_06 U8_X 电池上下料X轴铝壳除尘取料位标志
863.02 BOOL  ; RK_06 U8_X 电池上下料X轴#1入壳放料位标志
863.03 BOOL  ; RK_06 U8_X 电池上下料X轴#2入壳放料位标志
863.04 BOOL  ; RK_06 U8_X 电池上下料X轴#1入壳取料位标志
863.05 BOOL  ; RK_06 U8_X 电池上下料X轴#2入壳取料位标志
863.06 BOOL  ; RK_06 U8_X 电池上下料X轴#1Hipot检测放料位标志
863.07 BOOL  ; RK_06 U8_X 电池上下料X轴#2Hipot检测放料位标志
864.00 BOOL  ; RK_07 U8_Y 铝壳进料X轴等待位标志
864.01 BOOL  ; RK_07 U8_Y 铝壳进料X轴取料位标志
864.02 BOOL  ; RK_07 U8_Y 铝壳进料X轴放料位标志
865.00 BOOL  ; RK_07 U8_Z 铝壳上料移载Y轴待料位标志
865.01 BOOL  ; RK_07 U8_Z 铝壳上料移载Y轴#1铝壳上料位标志
865.02 BOOL  ; RK_07 U8_Z 铝壳上料移载Y轴#2铝壳上料位标志
865.03 BOOL  ; RK_07 U8_Z 铝壳上料移载Y轴#3铝壳托盘下料位标志
865.04 BOOL  ; RK_07 U8_Z 铝壳上料移载Y轴铝壳取料位标志
866.00 BOOL  ; RK_10 U8_U 电池除尘上料X轴待料位标志
866.01 BOOL  ; RK_10 U8_U 电池除尘上料X轴#1Hipot检测取料位标志
866.02 BOOL  ; RK_10 U8_U 电池除尘上料X轴#2Hipot检测取料位标志
866.03 BOOL  ; RK_10 U8_U 电池除尘上料X轴Hipot OK放料位标志
866.04 BOOL  ; RK_10 U8_U 电池除尘上料X轴Hipot NG放料位标志
886.00 BOOL  ; RK_07 U8_Y 铝壳进料X轴#1取料位标志
886.01 BOOL  ; RK_07 U8_Y 铝壳进料X轴#2取料位标志
886.02 BOOL  ; RK_07 U8_Y 铝壳进料X轴#3取料位标志
886.03 BOOL  ; RK_07 U8_Y 铝壳进料X轴#4取料位标志
886.04 BOOL  ; RK_07 U8_Y 铝壳进料X轴#5取料位标志
888.00 BOOL  ; RK_07 U8_Z 铝壳上料移载Y轴#1铝壳取料位标志
888.01 BOOL  ; RK_07 U8_Z 铝壳上料移载Y轴#2铝壳取料位标志
888.02 BOOL  ; RK_07 U8_Z 铝壳上料移载Y轴#3铝壳取料位标志
8.00 BOOL  ; RK_11 电池除尘旋转伸缩气缸到位
8.01 BOOL  ; RK_11 电池除尘旋转伸缩气缸原位
8.02 BOOL  ; RK_11 电池除尘伸缩气缸伸出位
8.03 BOOL  ; RK_11 电池除尘伸缩气缸缩回位
8.04 BOOL  ; RK_11 电池除尘夹爪气缸夹紧位
8.05 BOOL  ; RK_11 电池除尘夹爪气缸张开位
8.06 BOOL  ; RK_12 预焊上料机械手夹爪气缸夹紧位
8.07 BOOL  ; RK_12 预焊上料机械手夹爪气缸张开位
8.08 BOOL  ; RK_12 预焊下料机械手夹爪气缸夹紧位
8.09 BOOL  ; RK_12 预焊下料机械手夹爪气缸张开位
8.10 BOOL  ; RK_13 #1移载升降气缸上升位
8.11 BOOL  ; RK_13 #1移载升降气缸下降位
8.12 BOOL  ; RK_13 #1移载定位#1伸缩气缸缩回位
8.13 BOOL  ; RK_13 #1移载定位#1伸缩气缸伸出位
8.14 BOOL  ; RK_13 #1移载定位#2伸缩气缸缩回位
8.15 BOOL  ; RK_13 #1移载定位#2伸缩气缸伸出位
900.00 BOOL  ; RK_02 电芯进料机械手夹爪气缸夹紧位[lamp]
900.01 BOOL  ; RK_02 电芯进料机械手夹爪气缸张开位[lamp]
900.02 BOOL  ; RK_02 电芯进料机械手#1压紧气缸压紧位[lamp]
900.03 BOOL  ; RK_02 电芯进料机械手#2压紧气缸松开位[lamp]
900.04 BOOL  ; RK_03 电芯上料机械手夹爪气缸夹紧位[lamp]
900.05 BOOL  ; RK_03 电芯上料机械手夹爪气缸张开位[lamp]
900.06 BOOL  ; RK_03 电芯上料机械手#1压紧气缸压紧位[lamp]
900.07 BOOL  ; RK_03 电芯上料机械手#2压紧气缸松开位[lamp]
900.08 BOOL  ; RK_03 电芯上料升降气缸下降位[lamp]
900.09 BOOL  ; RK_03 电芯上料升降气缸上升位[lamp]
900.10 BOOL  ; RK_04 电芯除尘伸缩气缸缩回位[lamp]
900.11 BOOL  ; RK_04 电芯除尘伸缩气缸伸出位[lamp]
900.12 BOOL  ; RK_05 #1入壳滚轮夹紧气缸夹紧位[lamp]
900.13 BOOL  ; RK_05 #1入壳滚轮夹紧气缸松开位[lamp]
900.14 BOOL  ; RK_05 #1入壳铝壳定位平台伸缩气缸缩回位[lamp]
900.15 BOOL  ; RK_05 #1入壳铝壳定位平台伸缩气缸伸出位[lamp]
901.00 BOOL  ; RK_05 #1入壳铝壳定位平台升降气缸上升位[lamp]
901.01 BOOL  ; RK_05 #1入壳铝壳定位平台升降气缸下降位[lamp]
901.02 BOOL  ; RK_05 #1入壳铝壳定位伸缩气缸缩回位[lamp]
901.03 BOOL  ; RK_05 #1入壳铝壳定位伸缩气缸伸出位[lamp]
901.04 BOOL  ; RK_05 #1入壳铝壳定位夹爪气缸夹紧位[lamp]
901.05 BOOL  ; RK_05 #1入壳铝壳定位夹爪气缸张开位[lamp]
901.06 BOOL  ; RK_05 #2入壳滚轮夹紧气缸夹紧位[lamp]
901.07 BOOL  ; RK_05 #2入壳滚轮夹紧气缸松开位[lamp]
901.08 BOOL  ; RK_05 #2入壳铝壳定位平台伸缩气缸缩回位[lamp]
901.09 BOOL  ; RK_05 #2入壳铝壳定位平台伸缩气缸伸出位[lamp]
901.10 BOOL  ; RK_05 #2入壳铝壳定位平台升降气缸上升位[lamp]
901.11 BOOL  ; RK_05 #2入壳铝壳定位平台升降气缸下降位[lamp]
901.12 BOOL  ; RK_05 #2入壳铝壳定位伸缩气缸缩回位[lamp]
901.13 BOOL  ; RK_05 #2入壳铝壳定位伸缩气缸伸出位[lamp]
901.14 BOOL  ; RK_05 #2入壳铝壳定位夹爪气缸夹紧位[lamp]
901.15 BOOL  ; RK_05 #2入壳铝壳定位夹爪气缸张开位[lamp]
902.00 BOOL  ; RK_01 U0_X 电芯来料Y轴报警信号[lamp]
902.01 BOOL  ; RK_01 U0_X 电芯来料Y轴准备好了信号[lamp]
902.02 BOOL  ; RK_02 U0_Y 电芯进料X轴报警信号[lamp]
902.03 BOOL  ; RK_02 U0_Y 电芯进料X轴准备好了信号[lamp]
902.04 BOOL  ; RK_02 U0_Z 电芯进料Z轴报警信号[lamp]
902.05 BOOL  ; RK_02 U0_Z 电芯进料Z轴准备好了信号[lamp]
902.06 BOOL  ; RK_03 U0_U 电芯上料X轴报警信号[lamp]
902.07 BOOL  ; RK_03 U0_U 电芯上料X轴准备好了信号[lamp]
902.08 BOOL  ; RK_05 U2_X #1入壳Y轴报警信号[lamp]
902.09 BOOL  ; RK_05 U2_X #1入壳Y轴准备好了信号[lamp]
902.10 BOOL  ; RK_05 U2_Y #2入壳Y轴报警信号[lamp]
902.11 BOOL  ; RK_05 U2_Y #2入壳Y轴准备好了信号[lamp]
902.12 BOOL  ; RK_02 电芯进料Z轴刹车使能[lamp]
902.13 BOOL  ; RK_05 #1入壳定位陶瓷棒上#1夹紧气缸伸出位[lamp]
902.14 BOOL  ; RK_05 #1入壳定位陶瓷棒上#2夹紧气缸伸出位[lamp]
902.15 BOOL  ; RK_05 #1入壳定位陶瓷棒下#1夹紧气缸伸出位[lamp]
903.00 BOOL  ; RK_05 #1入壳定位陶瓷棒下#2夹紧气缸伸出位[lamp]
903.01 BOOL  ; RK_05 #1入壳定位陶瓷棒上#1夹紧气缸缩回位[lamp]
903.02 BOOL  ; RK_05 #1入壳定位陶瓷棒上#2夹紧气缸缩回位[lamp]
903.03 BOOL  ; RK_05 #1入壳定位陶瓷棒下#1夹紧气缸缩回位[lamp]
903.04 BOOL  ; RK_05 #1入壳定位陶瓷棒下#2夹紧气缸缩回位[lamp]
903.05 BOOL  ; RK_05 #1入壳吸盘上#1伸缩气缸缩回位[lamp]
903.06 BOOL  ; RK_05 #1入壳吸盘上#2伸缩气缸缩回位[lamp]
903.07 BOOL  ; RK_05 #1入壳吸盘上#3伸缩气缸缩回位[lamp]
903.08 BOOL  ; RK_05 #1入壳吸盘下#1伸缩气缸缩回位[lamp]
903.09 BOOL  ; RK_05 #1入壳吸盘下#2伸缩气缸缩回位[lamp]
903.10 BOOL  ; RK_05 #1入壳吸盘下#3伸缩气缸缩回位[lamp]
903.11 BOOL  ; RK_05 #1入壳电芯#1定位夹爪气缸松开位[lamp]
903.12 BOOL  ; RK_05 #1入壳电芯#2定位夹爪气缸松开位[lamp]
903.13 BOOL  ; RK_05 #1入壳电芯#1定位夹爪气缸夹紧位[lamp]
903.14 BOOL  ; RK_05 #1入壳电芯#2定位夹爪气缸夹紧位[lamp]
903.15 BOOL  ; RK_05 #2入壳定位陶瓷棒上#1夹紧气缸伸出位[lamp]
904.00 BOOL  ; RK_05 #2入壳定位陶瓷棒上#2夹紧气缸伸出位[lamp]
904.01 BOOL  ; RK_05 #2入壳定位陶瓷棒下#1夹紧气缸伸出位[lamp]
904.02 BOOL  ; RK_05 #2入壳定位陶瓷棒下#2夹紧气缸伸出位[lamp]
904.03 BOOL  ; RK_05 #2入壳定位陶瓷棒上#1夹紧气缸缩回位[lamp]
904.04 BOOL  ; RK_05 #2入壳定位陶瓷棒上#2夹紧气缸缩回位[lamp]
904.05 BOOL  ; RK_05 #2入壳定位陶瓷棒下#1夹紧气缸缩回位[lamp]
904.06 BOOL  ; RK_05 #2入壳定位陶瓷棒下#2夹紧气缸缩回位[lamp]
904.07 BOOL  ; RK_05 #2入壳吸盘上#1伸缩气缸缩回位[lamp]
904.08 BOOL  ; RK_05 #2入壳吸盘上#2伸缩气缸缩回位[lamp]
904.09 BOOL  ; RK_05 #2入壳吸盘上#3伸缩气缸缩回位[lamp]
904.10 BOOL  ; RK_05 #2入壳吸盘下#1伸缩气缸缩回位[lamp]
904.11 BOOL  ; RK_05 #2入壳吸盘下#2伸缩气缸缩回位[lamp]
904.12 BOOL  ; RK_05 #2入壳吸盘下#3伸缩气缸缩回位[lamp]
904.13 BOOL  ; RK_05 #2入壳电芯#1定位夹爪气缸松开位[lamp]
904.14 BOOL  ; RK_05 #2入壳电芯#2定位夹爪气缸松开位[lamp]
904.15 BOOL  ; RK_05 #2入壳电芯#1定位夹爪气缸夹紧位[lamp]
905.00 BOOL  ; RK_05 #2入壳电芯#2定位夹爪气缸夹紧位[lamp]
905.01 BOOL  ; RK_01 电芯来料有料感应[lamp]
905.02 BOOL  ; RK_02 电芯进料机械手夹爪柔性报警[lamp]
905.03 BOOL  ; RK_03 电芯上料机械手夹爪柔性报警[lamp]
905.04 BOOL  ; RK_04 电芯除尘有料感应[lamp]
905.05 BOOL  ; RK_02 扫码NG拉带有料感应#1[lamp]
905.06 BOOL  ; RK_02 扫码NG拉带有料感应#2[lamp]
905.07 BOOL  ; RK_02 扫码NG拉带料满感应[lamp]
905.08 BOOL  ; RK_05 #1入壳电芯有料感应[lamp]
905.09 BOOL  ; RK_05 #1入壳铝壳有料感应[lamp]
905.10 BOOL  ; RK_05 #2入壳电芯有料感应[lamp]
905.11 BOOL  ; RK_05 #2入壳铝壳有料感应[lamp]
905.12 BOOL  ; RK_05 #1入壳吸盘真空[lamp]
905.13 BOOL  ; RK_05 #2入壳吸盘真空[lamp]
905.14 BOOL  ; 前端设备对接输入信号（公共）[lamp]
905.15 BOOL  ; 后端设备对接输入信号（公共）[lamp]
906.00 BOOL  ; 小屏插入信号（公共）[lamp]
906.01 BOOL  ; NC433模块DC5V电源信号（公共）[lamp]
906.02 BOOL  ; DC24V伺服刹车电源信号（公共）[lamp]
906.03 BOOL  ; 出料端急停（公共）[lamp]
906.04 BOOL  ; 小移动屏急停（公共）[lamp]
906.05 BOOL  ; A机架#1门磁（公共）[lamp]
906.06 BOOL  ; A机架#2门磁（公共）[lamp]
906.07 BOOL  ; A机架#3门磁（公共）[lamp]
906.08 BOOL  ; A机架#4门磁（公共）[lamp]
906.09 BOOL  ; A机架#5门磁（公共）[lamp]
906.10 BOOL  ; A机架#6门磁（公共）[lamp]
906.11 BOOL  ; A机架#7门磁（公共）[lamp]
906.12 BOOL  ; A机架#8门磁（公共）[lamp]
906.13 BOOL  ; A机架#9门磁（公共）[lamp]
906.14 BOOL  ; 0[lamp]
906.15 BOOL  ; 0[lamp]
907.00 BOOL  ; 0[lamp]
907.01 BOOL  ; 0[lamp]
907.02 BOOL  ; 0[lamp]
907.03 BOOL  ; 0[lamp]
907.04 BOOL  ; 0[lamp]
907.05 BOOL  ; 0[lamp]
907.06 BOOL  ; 0[lamp]
907.07 BOOL  ; 0[lamp]
907.08 BOOL  ; 0[lamp]
907.09 BOOL  ; 0[lamp]
907.10 BOOL  ; 0[lamp]
907.11 BOOL  ; 0[lamp]
907.12 BOOL  ; 0[lamp]
907.13 BOOL  ; 0[lamp]
907.14 BOOL  ; 0[lamp]
907.15 BOOL  ; 0[lamp]
908.00 BOOL  ; RK_11 电池除尘旋转伸缩气缸到位[lamp]
908.01 BOOL  ; RK_11 电池除尘旋转伸缩气缸原位[lamp]
908.02 BOOL  ; RK_11 电池除尘伸缩气缸伸出位[lamp]
908.03 BOOL  ; RK_11 电池除尘伸缩气缸缩回位[lamp]
908.04 BOOL  ; RK_11 电池除尘夹爪气缸夹紧位[lamp]
908.05 BOOL  ; RK_11 电池除尘夹爪气缸张开位[lamp]
908.06 BOOL  ; RK_12 预焊上料机械手夹爪气缸夹紧位[lamp]
908.07 BOOL  ; RK_12 预焊上料机械手夹爪气缸张开位[lamp]
908.08 BOOL  ; RK_12 预焊下料机械手夹爪气缸夹紧位[lamp]
908.09 BOOL  ; RK_12 预焊下料机械手夹爪气缸张开位[lamp]
908.10 BOOL  ; RK_13 #1移载升降气缸上升位[lamp]
908.11 BOOL  ; RK_13 #1移载升降气缸下降位[lamp]
908.12 BOOL  ; RK_13 #1移载定位#1伸缩气缸缩回位[lamp]
908.13 BOOL  ; RK_13 #1移载定位#1伸缩气缸伸出位[lamp]
908.14 BOOL  ; RK_13 #1移载定位#2伸缩气缸缩回位[lamp]
908.15 BOOL  ; RK_13 #1移载定位#2伸缩气缸伸出位[lamp]
909.00 BOOL  ; RK_13 #1移载导向#1伸缩气缸伸出位[lamp]
909.01 BOOL  ; RK_13 #1移载导向#1伸缩气缸缩回位[lamp]
909.02 BOOL  ; RK_13 #1移载导向#2伸缩气缸伸出位[lamp]
909.03 BOOL  ; RK_13 #1移载导向#2伸缩气缸缩回位[lamp]
909.04 BOOL  ; RK_13 #1移载左右定位伸缩气缸伸出位[lamp]
909.05 BOOL  ; RK_13 #1移载左右定位伸缩气缸缩回位[lamp]
909.06 BOOL  ; RK_13 #2移载升降气缸上升位[lamp]
909.07 BOOL  ; RK_13 #2移载升降气缸下降位[lamp]
909.08 BOOL  ; RK_13 #2移载定位#1伸缩气缸缩回位[lamp]
909.09 BOOL  ; RK_13 #2移载定位#1伸缩气缸伸出位[lamp]
909.10 BOOL  ; RK_13 #2移载定位#2伸缩气缸缩回位[lamp]
909.11 BOOL  ; RK_13 #2移载定位#2伸缩气缸伸出位[lamp]
909.12 BOOL  ; RK_13 #2移载导向#1伸缩气缸伸出位[lamp]
909.13 BOOL  ; RK_13 #2移载导向#1伸缩气缸缩回位[lamp]
909.14 BOOL  ; RK_13 #2移载导向#2伸缩气缸伸出位[lamp]
909.15 BOOL  ; RK_13 #2移载导向#2伸缩气缸缩回位[lamp]
910.00 BOOL  ; RK_13 #2移载左右定位伸缩气缸伸出位[lamp]
910.01 BOOL  ; RK_13 #2移载左右定位伸缩气缸缩回位[lamp]
910.02 BOOL  ; RK_14 #1压装升降气缸下降位[lamp]
910.03 BOOL  ; RK_14 #1压装升降气缸上升位[lamp]
910.04 BOOL  ; RK_14 #1压装#1吸盘升降气缸下降位[lamp]
910.05 BOOL  ; RK_14 #1压装#1吸盘升降气缸上升位[lamp]
910.06 BOOL  ; RK_14 #1压装#2吸盘升降气缸下降位[lamp]
910.07 BOOL  ; RK_14 #1压装#2吸盘升降气缸上升位[lamp]
910.08 BOOL  ; RK_14 #2压装升降气缸下降位[lamp]
910.09 BOOL  ; RK_14 #2压装升降气缸上升位[lamp]
910.10 BOOL  ; RK_14 #2压装#1吸盘升降气缸下降位[lamp]
910.11 BOOL  ; RK_14 #2压装#1吸盘升降气缸上升位[lamp]
910.12 BOOL  ; RK_14 #2压装#2吸盘升降气缸下降位[lamp]
910.13 BOOL  ; RK_14 #2压装#2吸盘升降气缸上升位[lamp]
910.14 BOOL  ; RK_15 轮廓检测#1伸缩气缸伸出位[lamp]
910.15 BOOL  ; RK_15 轮廓检测#1伸缩气缸缩回位[lamp]
911.00 BOOL  ; RK_15 轮廓检测#2伸缩气缸伸出位[lamp]
911.01 BOOL  ; RK_15 轮廓检测#2伸缩气缸缩回位[lamp]
911.02 BOOL  ; RK_12 轮廓检测NG拨料气缸伸出位[lamp]
911.03 BOOL  ; RK_12 轮廓检测NG拨料气缸缩回位[lamp]
911.04 BOOL  ; RK_11 电池除尘有料感应[lamp]
911.05 BOOL  ; RK_12 预焊上料机械手夹爪柔性报警[lamp]
911.06 BOOL  ; RK_12 预焊下料机械手夹爪柔性报警[lamp]
911.07 BOOL  ; RK_16 激光焊接完成信号[lamp]
911.08 BOOL  ; RK_16 激光焊机故障信号[lamp]
911.09 BOOL  ; RK_13 #1移载电池顶盖超高检测[lamp]
911.10 BOOL  ; RK_16 激光焊机急停信号[lamp]
911.11 BOOL  ; RK_13 #2移载电池顶盖超高检测[lamp]
911.12 BOOL  ; RK_16 集尘器运行信号[lamp]
911.13 BOOL  ; RK_16 集尘器故障信号[lamp]
911.14 BOOL  ; RK_14 #1压装吸盘真空[lamp]
911.15 BOOL  ; RK_14 #2压装吸盘真空[lamp]
912.00 BOOL  ; RK_12 U4_X 预焊上下料X轴报警信号[lamp]
912.01 BOOL  ; RK_12 U4_X 预焊上下料X轴准备好了信号[lamp]
912.02 BOOL  ; RK_12 U4_Y 预焊上料Z轴报警信号[lamp]
912.03 BOOL  ; RK_12 U4_Y 预焊上料Z轴准备好了信号[lamp]
912.04 BOOL  ; RK_12 U4_Z 预焊下料Z轴报警信号[lamp]
912.05 BOOL  ; RK_12 U4_Z 预焊下料Z轴准备好了信号[lamp]
912.06 BOOL  ; RK_13 U4_U #1移载Y轴报警信号[lamp]
912.07 BOOL  ; RK_13 U4_U #1移载Y轴准备好了信号[lamp]
912.08 BOOL  ; RK_13 U6_X #2移载Y轴报警信号[lamp]
912.09 BOOL  ; RK_13 U6_X #2移载Y轴准备好了信号[lamp]
912.10 BOOL  ; RK_16 U6_Y 激光焊接X轴报警信号[lamp]
912.11 BOOL  ; RK_16 U6_Y 激光焊接X轴准备好了信号[lamp]
912.12 BOOL  ; RK_16 U6_Z 激光焊接Z轴报警信号[lamp]
912.13 BOOL  ; RK_16 U6_Z 激光焊接Z轴准备好了信号[lamp]
912.14 BOOL  ; RK_12 预焊上料Z轴刹车使能[lamp]
912.15 BOOL  ; RK_12 预焊下料Z轴刹车使能[lamp]
913.00 BOOL  ; RK_16 激光焊接Z轴刹车使能[lamp]
913.01 BOOL  ; RK_12 轮廓检测NG料槽#1有料感应[lamp]
913.02 BOOL  ; RK_12 轮廓检测NG料槽#1料满感应[lamp]
913.03 BOOL  ; RK_12 轮廓检测NG料槽#2有料感应[lamp]
913.04 BOOL  ; RK_12 轮廓检测NG料槽#2料满感应[lamp]
913.05 BOOL  ; RK_12 OK出料拉带放料位有料感应#1[lamp]
913.06 BOOL  ; RK_12 OK出料拉带放料位有料感应#2[lamp]
913.07 BOOL  ; RK_12 OK出料拉带出料位有料感应[lamp]
913.08 BOOL  ; 0[lamp]
913.09 BOOL  ; 0[lamp]
913.10 BOOL  ; 0[lamp]
913.11 BOOL  ; 0[lamp]
913.12 BOOL  ; 0[lamp]
913.13 BOOL  ; 0[lamp]
913.14 BOOL  ; 0[lamp]
913.15 BOOL  ; 0[lamp]
914.00 BOOL  ; RK_06 铝壳上料升降气缸下降位[lamp]
914.01 BOOL  ; RK_06 铝壳上料升降气缸上升位[lamp]
914.02 BOOL  ; RK_06 电池下料升降气缸下降位[lamp]
914.03 BOOL  ; RK_06 电池下料升降气缸上升位[lamp]
914.04 BOOL  ; RK_06 铝壳上料夹爪气缸夹紧位[lamp]
914.05 BOOL  ; RK_06 铝壳上料夹爪气缸张开位[lamp]
914.06 BOOL  ; RK_06 电池下料夹爪气缸夹紧位[lamp]
914.07 BOOL  ; RK_06 电池下料夹爪气缸张开位[lamp]
914.08 BOOL  ; RK_07 #1铝壳上料车定位升降气缸上升位[lamp]
914.09 BOOL  ; RK_07 #1铝壳上料车定位升降气缸下降位[lamp]
914.10 BOOL  ; RK_07 #2铝壳上料车定位升降气缸上升位[lamp]
914.11 BOOL  ; RK_07 #2铝壳上料车定位升降气缸下降位[lamp]
914.12 BOOL  ; RK_07 #3托盘下料车定位升降气缸上升位[lamp]
914.13 BOOL  ; RK_07 #3托盘下料车定位升降气缸下降位[lamp]
914.14 BOOL  ; RK_07 铝壳进料机械手升降气缸下降位[lamp]
914.15 BOOL  ; RK_07 铝壳进料机械手升降气缸上升位[lamp]
915.00 BOOL  ; RK_08 铝壳除尘旋转伸缩气缸原位[lamp]
915.01 BOOL  ; RK_08 铝壳除尘旋转伸缩气缸到位[lamp]
915.02 BOOL  ; RK_08 铝壳除尘伸缩气缸伸出位[lamp]
915.03 BOOL  ; RK_08 铝壳除尘伸缩气缸缩回位[lamp]
915.04 BOOL  ; RK_08 铝壳除尘夹爪气缸夹紧位[lamp]
915.05 BOOL  ; RK_08 铝壳除尘夹爪气缸张开位[lamp]
915.06 BOOL  ; RK_09 #1Hipot测试旋转伸缩气缸到位[lamp]
915.07 BOOL  ; RK_09 #1Hipot测试旋转伸缩气缸原位[lamp]
915.08 BOOL  ; RK_09 #1Hipot测试平台伸缩气缸缩回位[lamp]
915.09 BOOL  ; RK_09 #1Hipot测试平台伸缩气缸伸出位[lamp]
915.10 BOOL  ; RK_09 #1Hipot测试伸缩气缸伸出位[lamp]
915.11 BOOL  ; RK_09 #1Hipot测试伸缩气缸缩回位[lamp]
915.12 BOOL  ; RK_09 #2Hipot测试旋转伸缩气缸到位[lamp]
915.13 BOOL  ; RK_09 #2Hipot测试旋转伸缩气缸原位[lamp]
915.14 BOOL  ; RK_09 #2Hipot测试平台伸缩气缸缩回位[lamp]
915.15 BOOL  ; RK_09 #2Hipot测试平台伸缩气缸伸出位[lamp]
916.00 BOOL  ; RK_09 #2Hipot测试伸缩气缸伸出位[lamp]
916.01 BOOL  ; RK_09 #2Hipot测试伸缩气缸缩回位[lamp]
916.02 BOOL  ; RK_10 电池除尘上料机械手升降气缸下降位[lamp]
916.03 BOOL  ; RK_10 电池除尘上料机械手升降气缸上升位[lamp]
916.04 BOOL  ; RK_10 电池除尘上料机械手夹爪气缸夹紧位[lamp]
916.05 BOOL  ; RK_10 电池除尘上料机械手夹爪气缸张开位[lamp]
916.06 BOOL  ; RK_06 U8_X 电池上下料X轴报警信号[lamp]
916.07 BOOL  ; RK_06 U8_X 电池上下料X轴准备好了信号[lamp]
916.08 BOOL  ; RK_07 U8_Y 铝壳进料X轴报警信号[lamp]
916.09 BOOL  ; RK_07 U8_Y 铝壳进料X轴准备好了信号[lamp]
916.10 BOOL  ; RK_07 U8_Z 铝壳上料移载Y轴报警信号[lamp]
916.11 BOOL  ; RK_07 U8_Z 铝壳上料移载Y轴准备好了信号[lamp]
916.12 BOOL  ; RK_10 U8_U 电池除尘上料X轴报警信号[lamp]
916.13 BOOL  ; RK_10 U8_U 电池除尘上料X轴准备好了信号[lamp]
916.14 BOOL  ; RK_09 Hipot测试完成信号[lamp]
916.15 BOOL  ; RK_07 #1铝壳上料启动按钮[lamp]
917.00 BOOL  ; RK_07 #2铝壳上料启动按钮[lamp]
917.01 BOOL  ; RK_07 #3托盘下料启动按钮[lamp]
917.02 BOOL  ; RK_07 铝壳上料移载吸盘真空[lamp]
917.03 BOOL  ; RK_07 铝壳进料吸盘真空[lamp]
917.04 BOOL  ; RK_07 #1铝壳上料托盘到位感应[lamp]
917.05 BOOL  ; RK_07 #1铝壳上料位物料车到位感应[lamp]
917.06 BOOL  ; RK_07 #1铝壳上料初始位（#1）[lamp]
917.07 BOOL  ; RK_07 #1铝壳上料一个托盘位（#2）[lamp]
917.08 BOOL  ; RK_07 #1铝壳上料高限位（#3）[lamp]
917.09 BOOL  ; RK_07 #2铝壳上料托盘到位感应[lamp]
917.10 BOOL  ; RK_07 #2铝壳上料位物料车到位感应[lamp]
917.11 BOOL  ; RK_07 #2铝壳上料初始位（#1）[lamp]
917.12 BOOL  ; RK_07 #2铝壳上料一个托盘位（#2）[lamp]
917.13 BOOL  ; RK_07 #2铝壳上料高限位（#3）[lamp]
917.14 BOOL  ; RK_07 #3托盘下料上升到位感应[lamp]
917.15 BOOL  ; RK_07 #3托盘下料位物料车到位感应[lamp]
918.00 BOOL  ; RK_07 #3托盘下料初始位（#1）[lamp]
918.01 BOOL  ; RK_07 #3托盘下料一个托盘位（#2）[lamp]
918.02 BOOL  ; RK_07 #3托盘下料高限位（#3）[lamp]
918.03 BOOL  ; RK_07 铝壳上料移载托盘到位感应[lamp]
918.04 BOOL  ; RK_08 铝壳除尘有料感应[lamp]
918.05 BOOL  ; RK_09 #1Hipot测试有料感应[lamp]
918.06 BOOL  ; RK_09 #2Hipot测试有料感应[lamp]
918.07 BOOL  ; RK_10 Hipot检测NG拉带有料感应#1[lamp]
918.08 BOOL  ; RK_10 Hipot检测NG拉带有料感应#2[lamp]
918.09 BOOL  ; RK_10 Hipot检测NG拉带料满感应[lamp]
918.10 BOOL  ; RK_06 铝壳上料夹爪柔性报警[lamp]
918.11 BOOL  ; RK_06 电池下料夹爪柔性报警[lamp]
918.12 BOOL  ; RK_07 铝壳进料机械手柔性报警[lamp]
918.13 BOOL  ; RK_10 电池除尘上料机械手夹爪柔性报警[lamp]
918.14 BOOL  ; 手/自动选择（公共）[lamp]
918.15 BOOL  ; 启动按钮_绿（公共）[lamp]
919.00 BOOL  ; 停止按钮_红（公共）[lamp]
919.01 BOOL  ; 复位按钮_黄（公共）[lamp]
919.02 BOOL  ; 机台进气压力（正压）（公共）[lamp]
919.03 BOOL  ; 机台进气压力（负压）（公共）[lamp]
919.04 BOOL  ; 主屏急停（公共）[lamp]
919.05 BOOL  ; 铝壳上料端急停（公共）[lamp]
919.06 BOOL  ; HipotNG端急停（公共）[lamp]
919.07 BOOL  ; B机架#1门磁（公共）[lamp]
919.08 BOOL  ; B机架#2门磁（公共）[lamp]
919.09 BOOL  ; B机架#3门磁（公共）[lamp]
919.10 BOOL  ; B机架#4门磁（公共）[lamp]
919.11 BOOL  ; B机架#5门磁（公共）[lamp]
919.12 BOOL  ; B机架#6门磁（公共）[lamp]
919.13 BOOL  ; RK_07 #3托盘下料下降到位感应[lamp]
920.02 BOOL  ; RK_02 电芯进料机械手#1压紧气缸压紧位[lamp]
920.03 BOOL  ; RK_02 电芯进料机械手#2压紧气缸压紧位[lamp]
920.06 BOOL  ; RK_03 电芯上料机械手#1压紧气缸压紧位[lamp]
920.07 BOOL  ; RK_03 电芯上料机械手#2压紧气缸压紧位[lamp]
923.05 BOOL  ; RK_05 #1入壳吸盘上#1伸缩气缸伸出位[lamp]
923.06 BOOL  ; RK_05 #1入壳吸盘上#2伸缩气缸伸出位[lamp]
923.07 BOOL  ; RK_05 #1入壳吸盘上#3伸缩气缸伸出位[lamp]
923.08 BOOL  ; RK_05 #1入壳吸盘下#1伸缩气缸伸出位[lamp]
923.09 BOOL  ; RK_05 #1入壳吸盘下#2伸缩气缸伸出位[lamp]
923.10 BOOL  ; RK_05 #1入壳吸盘下#3伸缩气缸伸出位[lamp]
924.07 BOOL  ; RK_05 #2入壳吸盘上#1伸缩气缸伸出位[lamp]
924.08 BOOL  ; RK_05 #2入壳吸盘上#2伸缩气缸伸出位[lamp]
924.09 BOOL  ; RK_05 #2入壳吸盘上#3伸缩气缸伸出位[lamp]
924.10 BOOL  ; RK_05 #2入壳吸盘下#1伸缩气缸伸出位[lamp]
924.11 BOOL  ; RK_05 #2入壳吸盘下#2伸缩气缸伸出位[lamp]
924.12 BOOL  ; RK_05 #2入壳吸盘下#3伸缩气缸伸出位[lamp]
950.00 BOOL  ; RK_01 U0_X 电芯来料Y轴待料位[lamp]
950.01 BOOL  ; RK_01 U0_X 电芯来料Y轴上料位[lamp]
950.02 BOOL  ; RK_01 U0_X 电芯来料Y轴扫码位[lamp]
950.03 BOOL  ; RK_01 U0_X 电芯来料Y轴下料位[lamp]
950.10 BOOL  ; RK_01 U0_X 电芯来料Y轴回原点[lamp]
950.11 BOOL  ; $?St$Bk?_#[5051] / RK_01 U0_X 电芯来料Y轴JOG+[lamp] / $?St$Bk?_#[5051]
950.12 BOOL  ; RK_01 U0_X 电芯来料Y轴JOG-[lamp]
950.13 BOOL  ; RK_01 U0_X 电芯来料Y轴JOG高速[lamp]
950.14 BOOL  ; RK_01 U0_X 电芯来料Y轴JOG低速[lamp]
951.00 BOOL  ; RK_02 U0_Y 电芯进料X轴待料位[lamp]
951.01 BOOL  ; RK_02 U0_Y 电芯进料X轴取料位[lamp]
951.02 BOOL  ; RK_02 U0_Y 电芯进料X轴扫码OK放料位[lamp]
951.03 BOOL  ; RK_02 U0_Y 电芯进料X轴扫码NG放料位[lamp]
951.10 BOOL  ; RK_02 U0_Y 电芯进料X轴回原点[lamp]
951.11 BOOL  ; RK_02 U0_Y 电芯进料X轴JOG+[lamp]
951.12 BOOL  ; RK_02 U0_Y 电芯进料X轴JOG-[lamp]
951.13 BOOL  ; RK_02 U0_Y 电芯进料X轴JOG高速[lamp]
951.14 BOOL  ; RK_02 U0_Y 电芯进料X轴JOG低速[lamp]
952.00 BOOL  ; RK_02 U0_Z 电芯进料Z轴待料位（扫码）[lamp]
952.01 BOOL  ; RK_02 U0_Z 电芯进料Z轴取料位[lamp]
952.02 BOOL  ; RK_02 U0_Z 电芯进料Z轴扫码OK放料位[lamp]
952.03 BOOL  ; RK_02 U0_Z 电芯进料Z轴扫码NG放料位[lamp]
952.04 BOOL  ; RK_02 U0_Z 电芯进料Z轴扫码位[lamp]
952.10 BOOL  ; RK_02 U0_Z 电芯进料Z轴回原点[lamp]
952.11 BOOL  ; RK_02 U0_Z 电芯进料Z轴JOG+[lamp]
952.12 BOOL  ; RK_02 U0_Z 电芯进料Z轴JOG-[lamp]
952.13 BOOL  ; RK_02 U0_Z 电芯进料Z轴JOG高速[lamp]
952.14 BOOL  ; RK_02 U0_Z 电芯进料Z轴JOG低速[lamp]
953.00 BOOL  ; RK_03 U0_U 电芯上料X轴待料位[lamp]
953.01 BOOL  ; RK_03 U0_U 电芯上料X轴取料位[lamp]
953.02 BOOL  ; RK_03 U0_U 电芯上料X轴#1入壳放料位[lamp]
953.03 BOOL  ; RK_03 U0_U 电芯上料X轴#2入壳放料位[lamp]
953.10 BOOL  ; RK_03 U0_U 电芯上料X轴回原点[lamp]
953.11 BOOL  ; RK_03 U0_U 电芯上料X轴JOG+[lamp]
953.12 BOOL  ; RK_03 U0_U 电芯上料X轴JOG-[lamp]
953.13 BOOL  ; RK_03 U0_U 电芯上料X轴JOG高速[lamp]
953.14 BOOL  ; RK_03 U0_U 电芯上料X轴JOG低速[lamp]
954.00 BOOL  ; RK_05 U2_X #1入壳Y轴待料位[lamp]
954.01 BOOL  ; RK_05 U2_X #1入壳Y轴滚轮压紧位[lamp]
954.02 BOOL  ; RK_05 U2_X #1入壳Y轴滚轮松开位[lamp]
954.03 BOOL  ; RK_05 U2_X #1入壳Y轴入壳位[lamp]
954.04 BOOL  ; RK_05 U2_X #1入壳Y轴电芯定位夹爪松开位[lamp]
954.10 BOOL  ; RK_05 U2_X #1入壳Y轴回原点[lamp]
954.11 BOOL  ; RK_05 U2_X #1入壳Y轴JOG+[lamp]
954.12 BOOL  ; RK_05 U2_X #1入壳Y轴JOG-[lamp]
954.13 BOOL  ; RK_05 U2_X #1入壳Y轴JOG高速[lamp]
954.14 BOOL  ; RK_05 U2_X #1入壳Y轴JOG低速[lamp]
955.00 BOOL  ; RK_05 U2_Y #2入壳Y轴待料位[lamp]
955.01 BOOL  ; RK_05 U2_Y #2入壳Y轴滚轮压紧位[lamp]
955.02 BOOL  ; RK_05 U2_Y #2入壳Y轴滚轮松开位[lamp]
955.03 BOOL  ; RK_05 U2_Y #2入壳Y轴入壳位[lamp]
955.04 BOOL  ; RK_05 U2_Y #2入壳Y轴电芯定位夹爪松开位[lamp]
955.10 BOOL  ; RK_05 U2_Y #2入壳Y轴回原点[lamp]
955.11 BOOL  ; RK_05 U2_Y #2入壳Y轴JOG+[lamp]
955.12 BOOL  ; RK_05 U2_Y #2入壳Y轴JOG-[lamp]
955.13 BOOL  ; RK_05 U2_Y #2入壳Y轴JOG高速[lamp]
955.14 BOOL  ; RK_05 U2_Y #2入壳Y轴JOG低速[lamp]
956.00 BOOL  ; RK_12 U4_X 预焊上下料X轴待料位[lamp]
956.01 BOOL  ; RK_12 U4_X 预焊上下料X轴除尘取料位[lamp]
956.02 BOOL  ; RK_12 U4_X 预焊上下料X轴#1移载放料位[lamp]
956.03 BOOL  ; RK_12 U4_X 预焊上下料X轴#2移载放料位[lamp]
956.04 BOOL  ; RK_12 U4_X 预焊上下料X轴#1移载取料位[lamp]
956.05 BOOL  ; RK_12 U4_X 预焊上下料X轴#2移载取料位[lamp]
956.06 BOOL  ; RK_12 U4_X 预焊上下料X轴OK放料位[lamp]
956.07 BOOL  ; RK_12 U4_X 预焊上下料X轴#1NG放料位[lamp]
956.08 BOOL  ; RK_12 U4_X 预焊上下料X轴#2NG放料位[lamp]
956.10 BOOL  ; RK_12 U4_X 预焊上下料X轴回原点[lamp]
956.11 BOOL  ; RK_12 U4_X 预焊上下料X轴JOG+[lamp]
956.12 BOOL  ; RK_12 U4_X 预焊上下料X轴JOG-[lamp]
956.13 BOOL  ; RK_12 U4_X 预焊上下料X轴JOG高速[lamp]
956.14 BOOL  ; RK_12 U4_X 预焊上下料X轴JOG低速[lamp]
957.00 BOOL  ; RK_12 U4_Y 预焊上料Z轴待料位[lamp]
957.01 BOOL  ; RK_12 U4_Y 预焊上料Z轴除尘取料位[lamp]
957.02 BOOL  ; RK_12 U4_Y 预焊上料Z轴#1移载放料位[lamp]
957.03 BOOL  ; RK_12 U4_Y 预焊上料Z轴#2移载放料位[lamp]
957.10 BOOL  ; RK_12 U4_Y 预焊上料Z轴回原点[lamp]
957.11 BOOL  ; RK_12 U4_Y 预焊上料Z轴JOG+[lamp]
957.12 BOOL  ; RK_12 U4_Y 预焊上料Z轴JOG-[lamp]
957.13 BOOL  ; RK_12 U4_Y 预焊上料Z轴JOG高速[lamp]
957.14 BOOL  ; RK_12 U4_Y 预焊上料Z轴JOG低速[lamp]
958.00 BOOL  ; RK_12 U4_Z 预焊下料Z轴待料位[lamp]
958.01 BOOL  ; RK_12 U4_Z 预焊下料Z轴#1移载取料位[lamp]
958.02 BOOL  ; RK_12 U4_Z 预焊下料Z轴#2移载取料位[lamp]
958.03 BOOL  ; RK_12 U4_Z 预焊下料Z轴OK放料位[lamp]
958.04 BOOL  ; RK_12 U4_Z 预焊下料Z轴#1NG放料位[lamp]
958.05 BOOL  ; RK_12 U4_Z 预焊下料Z轴#2NG放料位[lamp]
958.10 BOOL  ; RK_12 U4_Z 预焊下料Z轴回原点[lamp]
958.11 BOOL  ; RK_12 U4_Z 预焊下料Z轴JOG+[lamp]
958.12 BOOL  ; RK_12 U4_Z 预焊下料Z轴JOG-[lamp]
958.13 BOOL  ; RK_12 U4_Z 预焊下料Z轴JOG高速[lamp]
958.14 BOOL  ; RK_12 U4_Z 预焊下料Z轴JOG低速[lamp]
959.00 BOOL  ; RK_13 U4_U #1移载Y轴待料位[lamp]
959.01 BOOL  ; RK_13 U4_U #1移载Y轴取放料位[lamp]
959.02 BOOL  ; RK_13 U4_U #1移载Y轴压装位[lamp]
959.03 BOOL  ; RK_13 U4_U #1移载Y轴#1轮廓检测位[lamp]
959.04 BOOL  ; RK_13 U4_U #1移载Y轴#2轮廓检测位[lamp]
959.05 BOOL  ; RK_13 U4_U #1移载Y轴激光焊接位[lamp]
959.10 BOOL  ; RK_13 U4_U #1移载Y轴回原点[lamp]
959.11 BOOL  ; RK_13 U4_U #1移载Y轴JOG+[lamp]
959.12 BOOL  ; RK_13 U4_U #1移载Y轴JOG-[lamp]
959.13 BOOL  ; RK_13 U4_U #1移载Y轴JOG高速[lamp]
959.14 BOOL  ; RK_13 U4_U #1移载Y轴JOG低速[lamp]
960.00 BOOL  ; RK_13 U6_X #2移载Y轴待料位[lamp]
960.01 BOOL  ; RK_13 U6_X #2移载Y轴取放料位[lamp]
960.02 BOOL  ; RK_13 U6_X #2移载Y轴压装位[lamp]
960.03 BOOL  ; RK_13 U6_X #2移载Y轴#1轮廓检测位[lamp]
960.04 BOOL  ; RK_13 U6_X #2移载Y轴#2轮廓检测位[lamp]
960.05 BOOL  ; RK_13 U6_X #2移载Y轴激光焊接位[lamp]
960.10 BOOL  ; RK_13 U6_X #2移载Y轴回原点[lamp]
960.11 BOOL  ; RK_13 U6_X #2移载Y轴JOG+[lamp]
960.12 BOOL  ; RK_13 U6_X #2移载Y轴JOG-[lamp]
960.13 BOOL  ; RK_13 U6_X #2移载Y轴JOG高速[lamp]
960.14 BOOL  ; RK_13 U6_X #2移载Y轴JOG低速[lamp]
961.00 BOOL  ; RK_16 U6_Y 激光焊接X轴待机位[lamp]
961.01 BOOL  ; RK_16 U6_Y 激光焊接X轴#1移载焊接位[lamp]
961.02 BOOL  ; RK_16 U6_Y 激光焊接X轴#2移载焊接位[lamp]
961.10 BOOL  ; RK_16 U6_Y 激光焊接X轴回原点[lamp]
961.11 BOOL  ; RK_16 U6_Y 激光焊接X轴JOG+[lamp]
961.12 BOOL  ; RK_16 U6_Y 激光焊接X轴JOG-[lamp]
961.13 BOOL  ; RK_16 U6_Y 激光焊接X轴JOG高速[lamp]
961.14 BOOL  ; RK_16 U6_Y 激光焊接X轴JOG低速[lamp]
962.00 BOOL  ; RK_16 U6_Z 激光焊接Z轴待机位[lamp]
962.01 BOOL  ; RK_16 U6_Z 激光焊接Z轴#1移载焊接位[lamp]
962.02 BOOL  ; RK_16 U6_Z 激光焊接Z轴#2移载焊接位[lamp]
962.10 BOOL  ; RK_16 U6_Z 激光焊接Z轴回原点[lamp]
962.11 BOOL  ; RK_16 U6_Z 激光焊接Z轴JOG+[lamp]
962.12 BOOL  ; RK_16 U6_Z 激光焊接Z轴JOG-[lamp]
962.13 BOOL  ; RK_16 U6_Z 激光焊接Z轴JOG高速[lamp]
962.14 BOOL  ; RK_16 U6_Z 激光焊接Z轴JOG低速[lamp]
963.00 BOOL  ; RK_06 U8_X 电池上下料X轴待机位[lamp]
963.01 BOOL  ; RK_06 U8_X 电池上下料X轴铝壳除尘取料位[lamp]
963.02 BOOL  ; RK_06 U8_X 电池上下料X轴#1入壳放料位[lamp]
963.03 BOOL  ; RK_06 U8_X 电池上下料X轴#2入壳放料位[lamp]
963.04 BOOL  ; RK_06 U8_X 电池上下料X轴#1入壳取料位[lamp]
963.05 BOOL  ; RK_06 U8_X 电池上下料X轴#2入壳取料位[lamp]
963.06 BOOL  ; RK_06 U8_X 电池上下料X轴#1Hipot检测放料位[lamp]
963.07 BOOL  ; RK_06 U8_X 电池上下料X轴#2Hipot检测放料位[lamp]
963.10 BOOL  ; RK_06 U8_X 电池上下料X轴回原点[lamp]
963.11 BOOL  ; RK_06 U8_X 电池上下料X轴JOG+[lamp]
963.12 BOOL  ; RK_06 U8_X 电池上下料X轴JOG-[lamp]
963.13 BOOL  ; RK_06 U8_X 电池上下料X轴JOG高速[lamp]
963.14 BOOL  ; RK_06 U8_X 电池上下料X轴JOG低速[lamp]
964.00 BOOL  ; RK_07 U8_Y 铝壳进料X轴等待位[lamp]
964.01 BOOL  ; RK_07 U8_Y 铝壳进料X轴取料位[lamp]
964.02 BOOL  ; RK_07 U8_Y 铝壳进料X轴放料位[lamp]
964.10 BOOL  ; RK_07 U8_Y 铝壳进料X轴回原点[lamp]
964.11 BOOL  ; RK_07 U8_Y 铝壳进料X轴JOG+[lamp]
964.12 BOOL  ; RK_07 U8_Y 铝壳进料X轴JOG-[lamp]
964.13 BOOL  ; RK_07 U8_Y 铝壳进料X轴JOG高速[lamp]
964.14 BOOL  ; RK_07 U8_Y 铝壳进料X轴JOG低速[lamp]
965.00 BOOL  ; RK_07 U8_Z 铝壳上料移载Y轴待料位[lamp]
965.01 BOOL  ; RK_07 U8_Z 铝壳上料移载Y轴#1铝壳上料位[lamp]
965.02 BOOL  ; RK_07 U8_Z 铝壳上料移载Y轴#2铝壳上料位[lamp]
965.03 BOOL  ; RK_07 U8_Z 铝壳上料移载Y轴#3铝壳托盘下料位[lamp]
965.04 BOOL  ; RK_07 U8_Z 铝壳上料移载Y轴铝壳取料位[lamp]
965.10 BOOL  ; RK_07 U8_Z 铝壳上料移载Y轴回原点[lamp]
965.11 BOOL  ; RK_07 U8_Z 铝壳上料移载Y轴JOG+[lamp]
965.12 BOOL  ; RK_07 U8_Z 铝壳上料移载Y轴JOG-[lamp]
965.13 BOOL  ; RK_07 U8_Z 铝壳上料移载Y轴JOG高速[lamp]
965.14 BOOL  ; RK_07 U8_Z 铝壳上料移载Y轴JOG低速[lamp]
966.00 BOOL  ; RK_10 U8_U 电池除尘上料X轴待料位[lamp]
966.01 BOOL  ; RK_10 U8_U 电池除尘上料X轴#1Hipot检测取料位[lamp]
966.02 BOOL  ; RK_10 U8_U 电池除尘上料X轴#2Hipot检测取料位[lamp]
966.03 BOOL  ; RK_10 U8_U 电池除尘上料X轴Hipot OK放料位[lamp]
966.04 BOOL  ; RK_10 U8_U 电池除尘上料X轴Hipot NG放料位[lamp]
966.10 BOOL  ; RK_10 U8_U 电池除尘上料X轴回原点[lamp]
966.11 BOOL  ; RK_10 U8_U 电池除尘上料X轴JOG+[lamp]
966.12 BOOL  ; RK_10 U8_U 电池除尘上料X轴JOG-[lamp]
966.13 BOOL  ; RK_10 U8_U 电池除尘上料X轴JOG高速[lamp]
966.14 BOOL  ; RK_10 U8_U 电池除尘上料X轴JOG低速[lamp]
9.00 BOOL  ; RK_13 #1移载导向#1伸缩气缸伸出位
9.01 BOOL  ; RK_13 #1移载导向#1伸缩气缸缩回位
9.02 BOOL  ; RK_13 #1移载导向#2伸缩气缸伸出位
9.03 BOOL  ; RK_13 #1移载导向#2伸缩气缸缩回位
9.04 BOOL  ; RK_13 #1移载左右定位伸缩气缸伸出位
9.05 BOOL  ; RK_13 #1移载左右定位伸缩气缸缩回位
9.06 BOOL  ; RK_13 #2移载升降气缸上升位
9.07 BOOL  ; RK_13 #2移载升降气缸下降位
9.08 BOOL  ; RK_13 #2移载定位#1伸缩气缸缩回位
9.09 BOOL  ; RK_13 #2移载定位#1伸缩气缸伸出位
9.10 BOOL  ; RK_13 #2移载定位#2伸缩气缸缩回位
9.11 BOOL  ; RK_13 #2移载定位#2伸缩气缸伸出位
9.12 BOOL  ; RK_13 #2移载导向#1伸缩气缸伸出位
9.13 BOOL  ; RK_13 #2移载导向#1伸缩气缸缩回位
9.14 BOOL  ; RK_13 #2移载导向#2伸缩气缸伸出位
9.15 BOOL  ; RK_13 #2移载导向#2伸缩气缸缩回位
A202.01 BOOL  ; 通讯端口#1可执行标志
A202.02 BOOL  ; 通讯端口#2可执行标志
A392.04 BOOL  ; 内置串行端口错误标志
A392.05 BOOL  ; 内置串行端口发送就绪
A392.06 BOOL  ; 内置串口接收就绪
A392.07 BOOL  ; 串行端口 1接收超限标志
A392.12 BOOL  ; $?St$Bk?_#[5052] / 串行端口 1 / 通信异常标志$?St$Bk?_#[5052]
A392.13 BOOL  ; 串行端口 1 发送准备标志
A392.14 BOOL  ; 串行端口 1接收结束标志
A392.15 BOOL  ; 串行端口 1接收超限标志
A393 CHANNEL  ; 内置串口接收数据长度
A526.00 BOOL  ; 串行端口 0 端口再起动标志
A526.01 BOOL  ; 串行端口 1 端口再起动标志
A622.01 BOOL  ; #2unit#1port restar
A622.02 BOOL  ; #2unit#2port restar
C0050 BOOL  ; 电芯进料机构扫码NG后重复次数计数
D0 CHANNEL  ; HMI窗口控制
D10 CHANNEL  ; PLC&PC数据交互超时报警延时设定
D100 CHANNEL  ; 发送内容“T”+“0D”
D1000.00 BOOL  ; RK_01 电芯来料机构初始位
D1000.05 BOOL  ; RK_01 电芯来料机构停止标志
D1000.06 BOOL  ; RK_01 电芯来料机构清料完成标志
D1000.07 BOOL  ; RK_01 电芯来料机构异常标志
D1001.00 BOOL  ; RK_01 电芯来料机构运行条件
D1002.00 BOOL  ; RK_01 U0_X 电芯来料Y轴运行条件
D1002.01 BOOL  ; RK_01 U0_X 电芯来料Y轴回原点条件
D1002.15 BOOL  ; RK_01 U0_X 电芯来料Y轴手自动运行条件
D1003.00 BOOL  ; RK_01 电芯来料机构单步/自动循环运行中（总）
D1003.10 BOOL  ; RK_01 电芯来料机构记忆显示（Lamp）
D1003.11 BOOL  ; RK_01 电芯来料机构初始化显示（Lamp）
D1003.13 BOOL  ; RK_01 电芯来料机构记忆清除（SW）
D1003.14 BOOL  ; RK_01 电芯来料机构复位按钮（SW）
D1003.15 BOOL  ; RK_01 电芯来料机构单步（SW）
D1004.00 BOOL  ; RK_01 电芯来料机构单步运行中
D1004.01 BOOL  ; RK_01 电芯来料机构单步/自动循环运行中
D1004.10 BOOL  ; RK_01 电芯来料机构单步运行条件
D1005.00 BOOL  ; RK_01 电芯来料机构开始运行条件
D1005.01 BOOL  ; RK_01 电芯来料机构步进条件
D1005.15 BOOL  ; RK_01 电芯来料机构步进
D1006 CHANNEL  ; RK_01 电芯来料机构步序
D1006.00 BOOL  ; RK_01 电芯来料机构自动开始（步）
D1006.01 BOOL  ; RK_01  电芯来料机构允许前端设备放料（步）
D1006.02 BOOL  ; RK_01  电芯来料机构Y轴下料位（步）
D1006.03 BOOL  ; RK_01  电芯来料机构Y轴下料位取料（步）
D1006.04 BOOL  ; RK_01  电芯来料机构Y轴上料位（步）
D1006.05 BOOL  ; RK_01 电芯来料机构循环完成
D1007.00 BOOL  ; RK_01 电芯来料机构复位（M）
D1007.01 BOOL  ; RK_01 U0_X 电芯来料Y轴回原点（复位）
D1007.02 BOOL  ; RK_01 U0_X 电芯来料Y轴上料位（复位）
D1009 CHANNEL  ; RK_01 电芯来料机构步序号
D101 CHANNEL  ; 发送内容“0A”
D1010.00 BOOL  ; RK_02 电芯进料机构初始位
D1010.05 BOOL  ; RK_02 电芯进料机构停止标志
D1010.06 BOOL  ; RK_02 电芯进料机构清料完成标志
D1010.07 BOOL  ; RK_02 电芯进料机构异常标志
D1011.00 BOOL  ; RK_02 电芯进料机构运行条件
D1012.00 BOOL  ; RK_02 U0_Y 电芯进料X轴运行条件
D1012.01 BOOL  ; RK_02 U0_Y 电芯进料X轴回原点条件
D1012.02 BOOL  ; RK_02 U0_Z 电芯进料Z轴运行条件
D1012.03 BOOL  ; RK_02 U0_Z 电芯进料Z轴回原点条件
D1012.04 BOOL  ; RK_02 U0_Z 电芯进料Z轴取料位条件
D1012.05 BOOL  ; RK_02 U0_Z 电芯进料Z轴扫码OK放料位条件
D1012.06 BOOL  ; RK_02 U0_Y 电芯进料X轴扫码NG放料位条件
D1012.15 BOOL  ; RK_02 U0_Y 电芯进料X轴手自动运行条件
D1013.00 BOOL  ; RK_02 电芯进料机构单步/自动循环运行中（总）
D1013.10 BOOL  ; RK_02 电芯进料工站记忆显示（Lamp）
D1013.11 BOOL  ; RK_02 电芯进料工站初始化显示（Lamp）
D1013.13 BOOL  ; RK_02 电芯进料机构记忆清除（SW）
D1013.14 BOOL  ; RK_02 电芯进料机构复位按钮（SW）
D1013.15 BOOL  ; RK_02 电芯进料机构单步（SW）
D1014.00 BOOL  ; RK_02 电芯进料机构单步运行中
D1014.01 BOOL  ; RK_02 电芯进料机构单步/自动循环运行中
D1014.10 BOOL  ; RK_02 电芯进料机构单步运行条件
D1015.00 BOOL  ; RK_02 电芯进料机构开始运行条件
D1015.01 BOOL  ; RK_02 电芯进料机构步进条件
D1015.15 BOOL  ; RK_02 电芯进料机构步进
D1016 CHANNEL  ; RK_02 电芯进料机构步序
D1016.00 BOOL  ; RK_02 电芯进料机构自动开始（步）
D1016.01 BOOL  ; RK_02 电芯进料机构进料Z轴取料位（步）
D1016.02 BOOL  ; RK_02 电芯进料机构进料夹爪气缸夹紧（步）
D1016.03 BOOL  ; RK_02 电芯进料机构进料压紧气缸压紧（步）
D1016.04 BOOL  ; RK_02 电芯进料机构进料Z轴待料位（扫码）&扫码数据初始化（步）
D1016.05 BOOL  ; RK_02 电芯进料机构扫码触发（步）
D1016.06 BOOL  ; RK_02 电芯进料机构扫码结果&扫码入站MES校验结果（步）
D1016.07 BOOL  ; RK_02 电芯进料机构进料X轴NG/OK放料位（步）
D1016.08 BOOL  ; RK_02 电芯进料机构进料Z轴NG放料位（步）
D1016.09 BOOL  ; RK_02 电芯进料机构进料Z轴OK放料位（步）
D1016.10 BOOL  ; RK_02 电芯进料机构进料压紧气缸松开（步）
D1016.11 BOOL  ; RK_02 电芯进料机构进料夹爪气缸张开（步）
D1016.12 BOOL  ; RK_02 电芯进料机构进料Z轴待料位（扫码）（步）
D1016.13 BOOL  ; RK_02 电芯进料机构进料X轴取料位（步）
D1016.14 BOOL  ; 备用
D1016.15 BOOL  ; RK_02 电芯进料机构循环完成
D1017.00 BOOL  ; RK_02 电芯进料机构复位（M）
D1017.01 BOOL  ; RK_02 电芯进料机械手夹爪气缸张开（复位）
D1017.02 BOOL  ; RK_02 电芯进料机械手夹爪气缸夹紧（复位）
D1017.03 BOOL  ; RK_02 电芯进料机械手压紧气缸缩回（复位）
D1017.04 BOOL  ; RK_02 电芯进料机械手压紧气缸伸出（复位）
D1017.05 BOOL  ; RK_02 U0_Z 电芯进料Z轴回原点（复位）
D1017.06 BOOL  ; RK_02 U0_Z 电芯进料Z轴待料位（扫码）（复位）
D1017.07 BOOL  ; RK_02 U0_Y 电芯进料X轴回原点（复位）
D1017.08 BOOL  ; RK_02 U0_Y 电芯进料X轴取料位（复位）
D1019 CHANNEL  ; RK_02 电芯进料机构步序号
D1020.00 BOOL  ; RK_03 电芯上料机构初始位
D1020.05 BOOL  ; RK_03 电芯上料机构停止标志
D1020.06 BOOL  ; RK_03 电芯上料机构清料完成标志
D1020.07 BOOL  ; RK_03 电芯上料机构异常标志
D1021.00 BOOL  ; RK_03 电芯上料机构运行条件
D1022.00 BOOL  ; RK_03 U0_U 电芯上料X轴运行条件
D1022.01 BOOL  ; RK_03 U0_U 电芯上料X轴回原点条件
D1022.15 BOOL  ; RK_03 U0_U 电芯上料X轴手自动运行条件
D1023.00 BOOL  ; RK_03 电芯上料机构单步/自动循环运行中（总）
D1023.10 BOOL  ; RK_03 电芯上料工站记忆显示（Lamp）
D1023.11 BOOL  ; RK_03 电芯上料工站初始化显示（Lamp）
D1023.13 BOOL  ; RK_03 电芯上料机构记忆清除（SW）
D1023.14 BOOL  ; RK_03 电芯上料机构复位按钮（SW）
D1023.15 BOOL  ; RK_03 电芯上料机构单步（SW）
D1024.00 BOOL  ; RK_03 电芯上料机构单步运行中
D1024.01 BOOL  ; RK_03 电芯上料机构单步/自动循环运行中
D1024.10 BOOL  ; RK_03 电芯上料机构单步运行条件
D1025.00 BOOL  ; RK_03 电芯上料机构开始运行条件
D1025.01 BOOL  ; RK_03 电芯上料机构步进条件
D1025.15 BOOL  ; RK_03 电芯上料机构步进
D1026 CHANNEL  ; RK_03 电芯上料机构步序
D1026.00 BOOL  ; RK_03 电芯上料机构自动开始（步）
D1026.01 BOOL  ; RK_03 电芯上料机构上料X轴取料位（步）
D1026.02 BOOL  ; RK_03 电芯上料机构上料升降气缸下降1（步）
D1026.03 BOOL  ; RK_03 电芯上料机构上料夹爪气缸夹紧（步）
D1026.04 BOOL  ; RK_03 电芯上料机构上料压紧气缸压紧（步）
D1026.05 BOOL  ; RK_03 电芯上料机构上料升降气缸上升1（步）
D1026.06 BOOL  ; RK_03 电芯上料机构上料X轴待料位（步）
D1026.07 BOOL  ; RK_03 电芯上料机构上料X轴#1|#2入壳放料位（步）
D1026.08 BOOL  ; RK_03 电芯上料机构上料升降气缸下降2（步）
D1026.09 BOOL  ; RK_03 电芯上料机构上料压紧气缸松开（步）
D1026.10 BOOL  ; RK_03 电芯上料机构上料夹爪气缸张开（步）
D1026.11 BOOL  ; RK_03 电芯上料机构上料升降气缸上升2（步）
D1026.12 BOOL  ; 备用
D1026.13 BOOL  ; RK_03 电芯上料机构循环完成
D1027.00 BOOL  ; RK_03 电芯上料机构复位（M）
D1027.01 BOOL  ; RK_03 电芯上料机械手夹爪气缸张开（复位）
D1027.02 BOOL  ; RK_03 电芯上料机械手夹爪气缸夹紧（复位）
D1027.03 BOOL  ; RK_03 电芯上料机械手压紧气缸缩回（复位）
D1027.04 BOOL  ; RK_03 电芯上料机械手压紧气缸伸出（复位）
D1027.05 BOOL  ; RK_03 电芯上料升降气缸上升（复位）
D1027.06 BOOL  ; RK_03 U0_U 电芯上料X轴回原点（复位）
D1027.07 BOOL  ; RK_03 U0_U 电芯上料X轴#1入壳放料位（复位）
D1029 CHANNEL  ; RK_03 电芯上料机构步序号
D1030.00 BOOL  ; RK_04 电芯除尘机构初始位
D1030.05 BOOL  ; RK_04 电芯除尘机构停止标志
D1030.06 BOOL  ; RK_04 电芯除尘机构清料完成标志
D1030.07 BOOL  ; RK_04 电芯除尘机构异常标志
D1031.00 BOOL  ; RK_04 电芯除尘机构运行条件
D1033.00 BOOL  ; RK_04 电芯除尘机构单步/自动循环运行中（总）
D1033.10 BOOL  ; RK_04 电芯除尘工站记忆显示（Lamp）
D1033.11 BOOL  ; RK_04 电芯除尘工站初始化显示（Lamp）
D1033.13 BOOL  ; RK_04 电芯除尘机构记忆清除（SW）
D1033.14 BOOL  ; RK_04 电芯除尘机构复位按钮（SW）
D1033.15 BOOL  ; RK_04 电芯除尘机构单步（SW）
D1034.00 BOOL  ; RK_04 电芯除尘机构单步运行中
D1034.01 BOOL  ; RK_04 电芯除尘机构单步/自动循环运行中
D1034.10 BOOL  ; RK_04 电芯除尘机构单步运行条件
D1035.00 BOOL  ; RK_04 电芯除尘机构开始运行条件
D1035.01 BOOL  ; RK_04 电芯除尘机构步进条件
D1035.15 BOOL  ; RK_04 电芯除尘机构步进
D1036 CHANNEL  ; RK_04 电芯除尘机构步序
D1036.00 BOOL  ; RK_04 电芯除尘机构自动开始（步）
D1036.01 BOOL  ; RK_04 电芯除尘机构伸缩气缸缩回（步）
D1036.02 BOOL  ; RK_04 电芯除尘机构吹气阀开（步）
D1036.03 BOOL  ; RK_04 电芯除尘机构吹气阀关（步）
D1036.04 BOOL  ; RK_04 电芯除尘机构伸缩气缸伸出（步）
D1036.05 BOOL  ; 备用
D1036.06 BOOL  ; RK_04 电芯除尘机构循环完成
D1037.00 BOOL  ; RK_04 电芯除尘机构复位（M）
D1037.01 BOOL  ; RK_04 电芯除尘吹气阀关（复位）
D1037.02 BOOL  ; RK_04 电芯除尘伸缩气缸伸出（复位）
D1039 CHANNEL  ; RK_04 电芯除尘机构步序号
D1040.00 BOOL  ; RK_05 #1入壳机构初始位
D1040.05 BOOL  ; RK_05 #1入壳机构停止标志
D1040.06 BOOL  ; RK_05 #1入壳机构清料完成标志
D1040.07 BOOL  ; RK_05 #1入壳机构异常标志（总）
D1040.08 BOOL  ; RK_05 #1入壳机构异常标志1
D1040.09 BOOL  ; RK_05 #1入壳机构异常标志2
D1041.00 BOOL  ; #1入壳机构运行条件（公共）
D1041.01 BOOL  ; RK_05 #1入壳机构运行条件1（铝壳定位）
D1041.02 BOOL  ; RK_05 #1入壳机构运行条件2（电芯定位&入壳）
D1042.00 BOOL  ; RK_05 U2_X #1入壳Y轴运行条件
D1042.01 BOOL  ; RK_05 U2_X #1入壳Y轴回原点条件
D1042.02 BOOL  ; RK_05 U2_X #1入壳Y轴待料位条件
D1042.03 BOOL  ; RK_05 U2_X #1入壳Y轴滚轮压紧位条件
D1042.04 BOOL  ; RK_05 U2_X #1入壳Y轴滚轮松开位条件
D1042.05 BOOL  ; RK_05 U2_X #1入壳Y轴入壳位条件
D1042.06 BOOL  ; RK_05 U2_X #1入壳Y轴电芯定位夹爪松开位条件
D1043.00 BOOL  ; RK_05 #1入壳机构单步/自动循环运行中（总）
D1043.10 BOOL  ; RK_05 #1入壳工站记忆显示（Lamp）
D1043.11 BOOL  ; RK_05 #1入壳工站初始化显示（Lamp）
D1043.13 BOOL  ; RK_05 #1入壳机构记忆清除（SW）
D1043.14 BOOL  ; RK_05 #1入壳机构复位按钮（SW）
D1043.15 BOOL  ; RK_05 #1入壳机构单步（SW）
D1044.00 BOOL  ; RK_05 #1入壳机构单步运行中1（铝壳定位）
D1044.01 BOOL  ; RK_05 #1入壳机构单步/自动循环运行中1（铝壳定位）
D1044.02 BOOL  ; RK_05 #1入壳机构单步运行中2（电芯定位&入壳）
D1044.03 BOOL  ; RK_05 #1入壳机构单步/自动循环运行中2（电芯定位&入壳）
D1044.10 BOOL  ; RK_05 #1入壳机构单步运行条件1（铝壳定位）
D1044.11 BOOL  ; RK_05 #1入壳机构单步运行条件2（电芯定位&入壳）
D1045.00 BOOL  ; RK_05 #1入壳机构开始运行条件1（铝壳定位）
D1045.01 BOOL  ; RK_05 #1入壳机构步进条件1（铝壳定位）
D1045.15 BOOL  ; RK_05 #1入壳机构步进1（铝壳定位）
D1046 CHANNEL  ; RK_05 #1入壳机构步序1（铝壳定位）
D1046.00 BOOL  ; RK_05 #1入壳机构自动开始1（步）
D1046.01 BOOL  ; RK_05 #1入壳机构铝壳定位夹爪气缸夹紧1（步）
D1046.02 BOOL  ; RK_05 #1入壳机构铝壳定位伸缩气缸缩回&定位陶瓷棒夹紧气缸伸出1（步）
D1046.03 BOOL  ; 备用
D1046.04 BOOL  ; RK_05 #1入壳机构铝壳定位平台伸缩气缸缩回1（步）
D1046.05 BOOL  ; RK_05 #1入壳机构铝壳定位平台升降气缸上升1（步）
D1046.06 BOOL  ; RK_05 #1入壳机构吸盘伸缩气缸伸出1（步）
D1046.07 BOOL  ; RK_05 #1入壳机构吸盘立真空1（步）
D1046.08 BOOL  ; RK_05 #1入壳机构吸盘伸缩气缸缩回1（步）
D1046.09 BOOL  ; 备用
D1046.10 BOOL  ; RK_05 #1入壳机构吸盘破真空&定位陶瓷棒夹紧气缸缩回&铝壳定位平台升降气缸下降1（步）
D1046.11 BOOL  ; 备用
D1046.12 BOOL  ; RK_05 #1入壳机构铝壳定位平台伸缩气缸伸出1（步）
D1046.13 BOOL  ; RK_05 #1入壳机构铝壳定位夹爪气缸张开1（步）
D1046.14 BOOL  ; RK_05 #1入壳机构铝壳定位伸缩气缸伸出1（步）
D1046.15 BOOL  ; RK_05 #1入壳机构循环完成1
D1048.00 BOOL  ; RK_05 #1入壳机构开始运行条件2（电芯定位&入壳）
D1048.01 BOOL  ; RK_05 #1入壳机构步进条件2（电芯定位&入壳）
D1048.15 BOOL  ; RK_05 #1入壳机构步进2（电芯定位&入壳）
D1049 CHANNEL  ; RK_05 #1入壳机构步序2（电芯定位&入壳）
D1049.00 BOOL  ; RK_05 #1入壳机构自动开始2（步）
D1049.01 BOOL  ; RK_05 #1入壳机构电芯定位夹爪气缸夹紧2（步）
D1049.02 BOOL  ; RK_05 #1入壳机构Y轴电芯定位夹爪气缸松开位2（步）
D1049.03 BOOL  ; RK_05 #1入壳机构电芯定位夹爪气缸松开2（步）
D1049.04 BOOL  ; RK_05 #1入壳机构Y轴滚轮压紧位2（步）
D1049.05 BOOL  ; RK_05 #1入壳机构滚轮夹紧气缸夹紧2（步）
D1049.06 BOOL  ; RK_05 #1入壳机构Y轴滚轮松开位2（步）
D1049.07 BOOL  ; RK_05 #1入壳机构滚轮夹紧气缸松开2（步）
D1049.08 BOOL  ; RK_05 #1入壳机构Y轴入壳位2（步）
D1049.09 BOOL  ; RK_05 #1入壳机构Y轴待料位2（步）
D1049.10 BOOL  ; 备用
D1049.11 BOOL  ; RK_05 #1入壳机构循环完成2
D1055 CHANNEL  ; #1入壳机构步序号1（入壳定位）
D1056 CHANNEL  ; #1入壳机构步序号2（电芯定位&入壳）
D1057.00 BOOL  ; RK_05 #1入壳机构复位（M）
D1057.01 BOOL  ; RK_05 #1入壳电芯定位夹爪气缸缩回（复位）
D1057.02 BOOL  ; RK_05 #1入壳滚轮夹紧气缸缩回（复位）
D1057.03 BOOL  ; RK_05 #1入壳电芯定位夹爪气缸伸出（复位）
D1057.04 BOOL  ; RK_05 #1入壳滚轮夹紧气缸伸出（复位）
D1057.05 BOOL  ; RK_05 #1入壳吸盘破真空（复位）
D1057.06 BOOL  ; RK_05 #1入壳吸盘伸缩气缸缩回（复位）
D1057.07 BOOL  ; RK_05 #1入壳铝壳定位平台升降气缸下降（复位）
D1057.08 BOOL  ; RK_05 #1入壳定位陶瓷棒夹紧气缸缩回（复位）
D1057.09 BOOL  ; RK_05 #1入壳铝壳定位平台伸缩气缸伸出（复位）
D1057.10 BOOL  ; RK_05 #1入壳铝壳定位伸缩气缸伸出（复位）
D1057.11 BOOL  ; RK_05 #1入壳铝壳定位夹爪气缸张开（复位）
D1057.12 BOOL  ; RK_05 #1入壳铝壳定位夹爪气缸夹紧（复位）
D1057.13 BOOL  ; RK_05 #1入壳铝壳定位伸缩气缸缩回（复位）
D1057.14 BOOL  ; RK_05 #1入壳定位陶瓷棒夹紧气缸伸出（复位）
D1057.15 BOOL  ; RK_05 #1入壳铝壳定位平台伸缩气缸缩回（复位）
D1058.00 BOOL  ; RK_05 #1入壳铝壳定位平台升降气缸上升（复位）
D1058.01 BOOL  ; RK_05 #1入壳吸盘伸缩气缸伸出（复位）
D1058.02 BOOL  ; RK_05 #1入壳吸盘立真空（复位）
D1058.03 BOOL  ; RK_05 #1入壳吸盘伸缩气缸缩回（复位）
D1058.04 BOOL  ; $?St$Bk?_#[5053] / RK_05 U2_X #1入壳Y轴回原点（复位） / $?St$Bk?_#[5053]
D1058.05 BOOL  ; RK_05 U2_X #1入壳Y轴待料位（复位）
D1058.06 BOOL  ; RK_05 #1入壳铝壳定位伸缩气缸缩回（复位）
D1060.00 BOOL  ; RK_05 #2入壳机构初始位
D1060.05 BOOL  ; RK_05 #2入壳机构停止标志
D1060.06 BOOL  ; RK_05 #2入壳机构清料完成标志
D1060.07 BOOL  ; RK_05 #2入壳机构异常标志（总）
D1060.08 BOOL  ; RK_05 #2入壳机构异常标志1
D1060.09 BOOL  ; RK_05 #2入壳机构异常标志2
D1061.00 BOOL  ; #2入壳机构运行条件（公共）
D1061.01 BOOL  ; RK_05 #2入壳机构运行条件1（铝壳定位）
D1061.02 BOOL  ; RK_05 #2入壳机构运行条件2（电芯定位&入壳）
D1062.00 BOOL  ; RK_05 U2_Y #2入壳Y轴运行条件
D1062.01 BOOL  ; RK_05 U2_Y #2入壳Y轴回原点条件
D1062.02 BOOL  ; RK_05 U2_Y #2入壳Y轴待料位条件
D1062.03 BOOL  ; RK_05 U2_Y #2入壳Y轴滚轮压紧位条件
D1062.04 BOOL  ; RK_05 U2_Y #2入壳Y轴滚轮松开位条件
D1062.05 BOOL  ; RK_05 U2_Y #2入壳Y轴入壳位条件
D1062.06 BOOL  ; RK_05 U2_Y #2入壳Y轴电芯定位夹爪松开位条件
D1063.00 BOOL  ; RK_05 #2入壳机构单步/自动循环运行中（总）
D1063.10 BOOL  ; RK_05 #2入壳工站记忆显示（Lamp）
D1063.11 BOOL  ; RK_05 #2入壳工站初始化显示（Lamp）
D1063.13 BOOL  ; RK_05 #2入壳机构记忆清除（SW）
D1063.14 BOOL  ; RK_05 #2入壳机构复位按钮（SW）
D1063.15 BOOL  ; RK_05 #2入壳机构单步（SW）
D1064.00 BOOL  ; RK_05 #2入壳机构单步运行中1（铝壳定位）
D1064.01 BOOL  ; RK_05 #2入壳机构单步/自动循环运行中1（铝壳定位）
D1064.02 BOOL  ; RK_05 #2入壳机构单步运行中2（电芯定位&入壳）
D1064.03 BOOL  ; RK_05 #2入壳机构单步/自动循环运行中2（电芯定位&入壳）
D1064.10 BOOL  ; RK_05 #2入壳机构单步运行条件1（铝壳定位）
D1064.11 BOOL  ; RK_05 #2入壳机构单步运行条件2（电芯定位&入壳）
D1065.00 BOOL  ; RK_05 #2入壳机构开始运行条件1（铝壳定位）
D1065.01 BOOL  ; RK_05 #2入壳机构步进条件1（铝壳定位）
D1065.15 BOOL  ; RK_05 #2入壳机构步进1（铝壳定位）
D1066 CHANNEL  ; RK_05 #2入壳机构步序1（铝壳定位）
D1066.00 BOOL  ; RK_05 #2入壳机构自动开始1（步）
D1066.01 BOOL  ; RK_05 #2入壳机构铝壳定位夹爪气缸夹紧1（步）
D1066.02 BOOL  ; RK_05 #2入壳机构铝壳定位伸缩气缸缩回&定位陶瓷棒夹紧气缸伸出1（步）
D1066.03 BOOL  ; 备用
D1066.04 BOOL  ; RK_05 #2入壳机构铝壳定位平台伸缩气缸缩回1（步）
D1066.05 BOOL  ; RK_05 #2入壳机构铝壳定位平台升降气缸上升1（步）
D1066.06 BOOL  ; RK_05 #2入壳机构吸盘伸缩气缸伸出1（步）
D1066.07 BOOL  ; RK_05 #2入壳机构吸盘立真空1（步）
D1066.08 BOOL  ; RK_05 #2入壳机构吸盘伸缩气缸缩回1（步）
D1066.09 BOOL  ; 备用
D1066.10 BOOL  ; RK_05 #2入壳机构吸盘破真空&定位陶瓷棒夹紧气缸缩回&铝壳定位平台升降气缸下降1（步）
D1066.11 BOOL  ; 备用
D1066.12 BOOL  ; RK_05 #2入壳机构铝壳定位平台伸缩气缸伸出1（步）
D1066.13 BOOL  ; RK_05 #2入壳机构铝壳定位夹爪气缸张开1（步）
D1066.14 BOOL  ; RK_05 #2入壳机构铝壳定位伸缩气缸伸出1（步）
D1066.15 BOOL  ; RK_05 #2入壳机构循环完成1
D1068.00 BOOL  ; RK_05 #2入壳机构开始运行条件2（电芯定位&入壳）
D1068.01 BOOL  ; RK_05 #2入壳机构步进条件2（电芯定位&入壳）
D1068.15 BOOL  ; RK_05 #2入壳机构步进2（电芯定位&入壳）
D1069 CHANNEL  ; RK_05 #2入壳机构步序2（电芯定位&入壳）
D1069.00 BOOL  ; RK_05 #2入壳机构自动开始2（步）
D1069.01 BOOL  ; RK_05 #2入壳机构电芯定位夹爪气缸夹紧2（步）
D1069.02 BOOL  ; RK_05 #2入壳机构Y轴电芯定位夹爪气缸松开位2（步）
D1069.03 BOOL  ; RK_05 #2入壳机构电芯定位夹爪气缸松开2（步）
D1069.04 BOOL  ; RK_05 #2入壳机构Y轴滚轮压紧位2（步）
D1069.05 BOOL  ; RK_05 #2入壳机构滚轮夹紧气缸夹紧2（步）
D1069.06 BOOL  ; RK_05 #2入壳机构Y轴滚轮松开位2（步）
D1069.07 BOOL  ; RK_05 #2入壳机构滚轮夹紧气缸松开2（步）
D1069.08 BOOL  ; RK_05 #2入壳机构Y轴入壳位2（步）
D1069.09 BOOL  ; RK_05 #2入壳机构Y轴待料位2（步）
D1069.10 BOOL  ; 备用
D1069.11 BOOL  ; RK_05 #2入壳机构循环完成2
D1075 CHANNEL  ; #2入壳机构步序号1（入壳定位）
D1076 CHANNEL  ; #2入壳机构步序号2（电芯定位&入壳）
D1077.00 BOOL  ; RK_05 #2入壳机构复位（M）
D1077.01 BOOL  ; RK_05 #2入壳电芯定位夹爪气缸缩回（复位）
D1077.02 BOOL  ; RK_05 #2入壳滚轮夹紧气缸缩回（复位）
D1077.03 BOOL  ; RK_05 #2入壳电芯定位夹爪气缸伸出（复位）
D1077.04 BOOL  ; RK_05 #2入壳滚轮夹紧气缸伸出（复位）
D1077.05 BOOL  ; RK_05 #2入壳吸盘破真空（复位）
D1077.06 BOOL  ; RK_05 #2入壳吸盘伸缩气缸缩回（复位）
D1077.07 BOOL  ; RK_05 #2入壳铝壳定位平台升降气缸下降（复位）
D1077.08 BOOL  ; RK_05 #2入壳定位陶瓷棒夹紧气缸缩回（复位）
D1077.09 BOOL  ; RK_05 #2入壳铝壳定位平台伸缩气缸伸出（复位）
D1077.10 BOOL  ; RK_05 #2入壳铝壳定位伸缩气缸伸出（复位）
D1077.11 BOOL  ; RK_05 #2入壳铝壳定位夹爪气缸张开（复位）
D1077.12 BOOL  ; RK_05 #2入壳铝壳定位夹爪气缸夹紧（复位）
D1077.13 BOOL  ; RK_05 #2入壳铝壳定位伸缩气缸缩回（复位）
D1077.14 BOOL  ; RK_05 #2入壳定位陶瓷棒夹紧气缸伸出（复位）
D1077.15 BOOL  ; RK_05 #2入壳铝壳定位平台伸缩气缸缩回（复位）
D1078.00 BOOL  ; RK_05 #2入壳铝壳定位平台升降气缸上升（复位）
D1078.01 BOOL  ; RK_05 #2入壳吸盘伸缩气缸伸出（复位）
D1078.02 BOOL  ; RK_05 #2入壳吸盘立真空（复位）
D1078.03 BOOL  ; RK_05 #2入壳吸盘伸缩气缸缩回（复位）
D1078.04 BOOL  ; RK_05 U2_Y #2入壳Y轴回原点（复位）
D1078.05 BOOL  ; RK_05 U2_Y #2入壳Y轴待料位（复位）
D1078.06 BOOL  ; RK_05 #2入壳铝壳定位伸缩气缸缩回（复位）
D1080.00 BOOL  ; RK_06 电池上下料机构初始位
D1080.05 BOOL  ; RK_06 电池上下料机构停止标志
D1080.06 BOOL  ; RK_06 电池上下料机构清料完成标志
D1080.07 BOOL  ; RK_06 电池上下料机构异常标志
D1081.00 BOOL  ; RK_06 电池上下料机构运行条件（公共）
D1081.01 BOOL  ; RK_06 电池上下料机构运行条件1（铝壳取料）
D1081.02 BOOL  ; RK_06 电池上下料机构运行条件2（铝壳下料）
D1081.03 BOOL  ; RK_06 电池上下料机构运行条件3（电池取料）
D1081.04 BOOL  ; RK_06 电池上下料机构运行条件4（电池下料）
D1082.00 BOOL  ; RK_06 U8_X 电池上下料X轴运行条件
D1082.01 BOOL  ; RK_06 U8_X 电池上下料X轴回原点条件
D1082.15 BOOL  ; RK_06 U8_X 电池上下料X轴手自动运行条件
D1083.00 BOOL  ; RK_06 电池上下料机构单步/自动循环运行中（总）
D1083.10 BOOL  ; RK_06 电池上下料工站记忆显示（Lamp）
D1083.11 BOOL  ; RK_06 电池上下料工站初始化显示（Lamp）
D1083.13 BOOL  ; RK_06 电池上下料机构记忆清除（SW）
D1083.14 BOOL  ; RK_06 电池上下料机构复位按钮（SW）
D1083.15 BOOL  ; RK_06 电池上下料机构单步（SW）
D1084.00 BOOL  ; RK_06 电池上下料机构单步运行中1（铝壳取料）
D1084.01 BOOL  ; RK_06 电池上下料机构单步/自动循环运行中1（铝壳取料）
D1084.02 BOOL  ; RK_06 电池上下料机构单步运行中2（铝壳下料）
D1084.03 BOOL  ; RK_06 电池上下料机构单步/自动循环运行中2（铝壳下料）
D1084.04 BOOL  ; RK_06 电池上下料机构单步运行中3（电池取料）
D1084.05 BOOL  ; RK_06 电池上下料机构单步/自动循环运行中3（电池取料）
D1084.06 BOOL  ; RK_06 电池上下料机构单步运行中4（电池下料）
D1084.07 BOOL  ; RK_06 电池上下料机构单步/自动循环运行中4（电池下料）
D1084.10 BOOL  ; RK_06 电池上下料机构单步运行条件1（铝壳取料）
D1084.11 BOOL  ; RK_06 电池上下料机构单步运行条件2（铝壳下料）
D1084.12 BOOL  ; RK_06 电池上下料机构单步运行条件3（电池取料）
D1084.13 BOOL  ; RK_06 电池上下料机构单步运行条件4（电池下料）
D1085.00 BOOL  ; RK_06 电池上下料机构开始运行条件1（铝壳取料）
D1085.01 BOOL  ; RK_06 电池上下料机构步进条件1（铝壳取料）
D1085.15 BOOL  ; RK_06 电池上下料机构步进1（铝壳取料）
D1086 CHANNEL  ; RK_06 电池上下料机构步序1（铝壳取料）
D1086.00 BOOL  ; RK_06 电池上下料机构自动开始1（步）
D1086.01 BOOL  ; RK_06 电池上下料机构X轴铝壳除尘取料位1（步）
D1086.02 BOOL  ; RK_06 电池上下料机构铝壳上料升降气缸下降1（步）
D1086.03 BOOL  ; RK_06 电池上下料机构铝壳上料夹爪气缸夹紧1（步）
D1086.04 BOOL  ; RK_06 电池上下料机构铝壳上料升降气缸上升1（步）
D1086.05 BOOL  ; 备用
D1086.06 BOOL  ; RK_06 电池上下料机构循环完成1
D1088.00 BOOL  ; RK_06 电池上下料机构开始运行条件2（铝壳下料）
D1088.01 BOOL  ; RK_06 电池上下料机构步进条件2（铝壳下料）
D1088.15 BOOL  ; RK_06 电池上下料机构步进2（铝壳下料）
D1089 CHANNEL  ; RK_06 电池上下料机构步序2（铝壳下料）
D1089.00 BOOL  ; RK_06 电池上下料机构自动开始2（步）
D1089.01 BOOL  ; RK_06 电池上下料机构X轴#1|#2入壳放料位2（步）
D1089.02 BOOL  ; RK_06 电池上下料机构铝壳上料升降气缸下降2（步）
D1089.03 BOOL  ; RK_06 电池上下料机构铝壳上料夹爪气缸张开2（步）
D1089.04 BOOL  ; RK_06 电池上下料机构铝壳上料升降气缸上升2（步）
D1089.05 BOOL  ; 备用
D1089.06 BOOL  ; RK_06 电池上下料机构循环完成2
D1091.00 BOOL  ; RK_06 电池上下料机构开始运行条件3（电池取料）
D1091.01 BOOL  ; RK_06 电池上下料机构步进条件3（电池取料）
D1091.15 BOOL  ; RK_06 电池上下料机构步进3（电池取料）
D1092 CHANNEL  ; RK_06 电池上下料机构步序3（电池取料）
D1092.00 BOOL  ; RK_06 电池上下料机构自动开始3（步）
D1092.01 BOOL  ; RK_06 电池上下料机构X轴#1|#2入壳取料位3（步）
D1092.02 BOOL  ; RK_06 电池上下料机构电池下料升降气缸下降3（步）
D1092.03 BOOL  ; RK_06 电池上下料机构电池下料夹爪气缸夹紧3（步）
D1092.04 BOOL  ; RK_06 电池上下料机构电池下料升降气缸上升3（步）
D1092.05 BOOL  ; 备用
D1092.06 BOOL  ; RK_06 电池上下料机构循环完成3
D1094.00 BOOL  ; RK_06 电池上下料机构开始运行条件4（电池下料）
D1094.01 BOOL  ; RK_06 电池上下料机构步进条件4（电池下料）
D1094.15 BOOL  ; RK_06 电池上下料机构步进4（电池下料）
D1095 CHANNEL  ; RK_06 电池上下料机构步序4（电池下料）
D1095.00 BOOL  ; RK_06 电池上下料机构自动开始4（步）
D1095.01 BOOL  ; RK_06 电池上下料机构X轴#1|#2Hipot检测放料位4（步）
D1095.02 BOOL  ; RK_06 电池上下料机构电池下料升降气缸下降4（步）
D1095.03 BOOL  ; RK_06 电池上下料机构电池下料夹爪气缸张开4（步）
D1095.04 BOOL  ; RK_06 电池上下料机构电池下料升降气缸上升4（步）
D1095.05 BOOL  ; 备用
D1095.06 BOOL  ; RK_06 电池上下料机构循环完成4
D1097.00 BOOL  ; RK_06 电池上下料机构复位（M）
D1097.01 BOOL  ; RK_06 铝壳上料夹爪气缸张开（复位）
D1097.02 BOOL  ; RK_06 铝壳上料夹爪气缸夹紧（复位）
D1097.03 BOOL  ; RK_06 电池下料夹爪气缸张开（复位）
D1097.04 BOOL  ; RK_06 电池下料夹爪气缸夹紧（复位）
D1097.05 BOOL  ; RK_06 铝壳上料升降气缸上升（复位）
D1097.06 BOOL  ; RK_06 电池下料升降气缸上升（复位）
D1097.07 BOOL  ; RK_06 U8_X 电池上下料X轴回原（复位）
D1097.08 BOOL  ; RK_06 U8_X 电池上下料X轴铝壳除尘取料位（复位）
D1099 CHANNEL  ; RK_06 电池上下料机构步序号
D110 CHANNEL  ; 电芯进料扫码数据开始字
D1100.00 BOOL  ; RK_07 铝壳进料机构初始位
D1100.05 BOOL  ; RK_07 铝壳进料机构停止标志
D1100.06 BOOL  ; RK_07 铝壳进料机构清料完成标志
D1100.07 BOOL  ; RK_07 铝壳进料机构异常标志
D1101.00 BOOL  ; RK_07 铝壳进料机构运行条件
D1102.00 BOOL  ; RK_07 U8_Y 铝壳进料X轴运行条件
D1102.01 BOOL  ; RK_07 U8_Y 铝壳进料X轴回原点条件
D1102.15 BOOL  ; RK_07 U8_Y 铝壳进料X轴手自动运行条件
D1103.00 BOOL  ; RK_07 铝壳进料机构单步/自动循环运行中（总）
D1103.10 BOOL  ; RK_07 铝壳进料工站记忆显示（Lamp）
D1103.11 BOOL  ; RK_07 铝壳进料工站初始化显示（Lamp）
D1103.13 BOOL  ; RK_07 铝壳进料机构记忆清除（SW）
D1103.14 BOOL  ; RK_07 铝壳进料机构复位按钮（SW）
D1103.15 BOOL  ; RK_07 铝壳进料机构单步（SW）
D1104.00 BOOL  ; RK_07 铝壳进料机构单步运行中
D1104.01 BOOL  ; RK_07 铝壳进料机构单步/自动循环运行中
D1104.10 BOOL  ; RK_07 铝壳进料机构单步运行条件
D1105.00 BOOL  ; RK_07 铝壳进料机构开始运行条件
D1105.01 BOOL  ; RK_07 铝壳进料机构步进条件
D1105.15 BOOL  ; RK_07 铝壳进料机构步进
D1106 CHANNEL  ; RK_07 铝壳进料机构步序
D1106.00 BOOL  ; RK_07 铝壳进料机构自动开始（步）
D1106.01 BOOL  ; RK_07 铝壳进料机构升降气缸下降（步）
D1106.02 BOOL  ; RK_07 铝壳进料机构吸盘立真空（步）
D1106.03 BOOL  ; RK_07 铝壳进料机构升降气缸上升（步）
D1106.04 BOOL  ; RK_07 铝壳进料机构X轴放料位（步）
D1106.05 BOOL  ; RK_07 铝壳进料机构升降气缸下降（步）
D1106.06 BOOL  ; RK_07 铝壳进料机构吸盘破真空（步）
D1106.07 BOOL  ; RK_07 铝壳进料机构升降气缸上升（步）
D1106.08 BOOL  ; RK_07 铝壳进料机构X轴取料位（步）
D1106.09 BOOL  ; 备用
D1106.10 BOOL  ; 备用
D1106.11 BOOL  ; 备用
D1106.12 BOOL  ; RK_07 铝壳进料机构循环完成
D1107.00 BOOL  ; RK_07 铝壳进料机构复位（M）
D1107.01 BOOL  ; RK_07 铝壳进料吸盘破真空（复位）
D1107.02 BOOL  ; RK_07 铝壳进料吸盘立真空（复位）
D1107.03 BOOL  ; RK_07 铝壳进料机械手升降气缸上升（复位）
D1107.04 BOOL  ; RK_07 U8_Y 铝壳进料X轴回原点（复位）
D1107.05 BOOL  ; RK_07 U8_Y 铝壳进料X轴取料位（复位）
D1109 CHANNEL  ; RK_07 铝壳进料机构步序号
D1110.00 BOOL  ; RK_07 铝壳上料移载机构初始位
D1110.05 BOOL  ; RK_07 铝壳上料移载机构停止标志
D1110.06 BOOL  ; RK_07 铝壳上料移载机构清料完成标志
D1110.07 BOOL  ; RK_07 铝壳上料移载机构异常标志
D1111.00 BOOL  ; RK_07 铝壳上料移载机构运行条件（公共）
D1111.01 BOOL  ; RK_07 铝壳上料移载机构运行条件1（铝壳上料）
D1111.02 BOOL  ; RK_07 铝壳上料移载机构运行条件2（铝壳取料）
D1111.03 BOOL  ; RK_07 铝壳上料移载机构运行条件3（铝壳托盘卸载）
D1112.00 BOOL  ; RK_07 U8_Z 铝壳上料移载Y轴运行条件
D1112.01 BOOL  ; RK_07 U8_Z 铝壳上料移载Y轴回原点条件
D1112.15 BOOL  ; RK_07 U8_Z 铝壳上料移载Y轴手自动运行条件
D1113.00 BOOL  ; RK_07 铝壳上料移载机构单步/自动循环运行中（总）
D1113.10 BOOL  ; RK_07 铝壳上料移载工站记忆显示（Lamp）
D1113.11 BOOL  ; RK_07 铝壳上料移载工站初始化显示（Lamp）
D1113.13 BOOL  ; RK_07 铝壳上料移载机构记忆清除（SW）
D1113.14 BOOL  ; RK_07 铝壳上料移载机构复位按钮（SW）
D1113.15 BOOL  ; RK_07 铝壳上料移载机构单步（SW）
D1114.00 BOOL  ; RK_07 铝壳上料移载机构单步运行中1（铝壳上料）
D1114.01 BOOL  ; RK_07 铝壳进料机构单步/自动循环运行中1（铝壳上料）
D1114.02 BOOL  ; RK_07 铝壳上料移载机构单步运行中2（铝壳取料）
D1114.03 BOOL  ; RK_07 铝壳进料机构单步/自动循环运行中2（铝壳取料）
D1114.04 BOOL  ; RK_07 铝壳上料移载机构单步运行中3（铝壳托盘卸载）
D1114.05 BOOL  ; RK_07 铝壳进料机构单步/自动循环运行中3（铝壳托盘卸载）
D1114.10 BOOL  ; RK_07 铝壳上料移载机构单步运行条件1（铝壳上料）
D1114.11 BOOL  ; RK_07 铝壳上料移载机构单步运行条件2（铝壳取料）
D1114.12 BOOL  ; RK_07 铝壳上料移载机构单步运行条件3（铝壳托盘卸载）
D1115.00 BOOL  ; RK_07 铝壳上料移载机构开始运行条件1（铝壳上料）
D1115.01 BOOL  ; RK_07 铝壳上料移载机构步进条件1（铝壳上料）
D1115.15 BOOL  ; RK_07 铝壳上料移载机构步进1（铝壳上料）
D1116 CHANNEL  ; RK_07 铝壳上料移载机构步序1（铝壳上料）
D1116.00 BOOL  ; RK_07 铝壳上料移载机构自动开始1（步）
D1116.01 BOOL  ; RK_07 铝壳上料移载机构Y轴#1/2铝壳上料位1（步）
D1116.02 BOOL  ; RK_07 铝壳上料移载机构#1/2铝壳上料电机正转1（步）
D1116.03 BOOL  ; RK_07 铝壳上料移载机构吸盘立真空1（步）
D1116.04 BOOL  ; RK_07 铝壳上料移载机构#1/2铝壳上料电机反转1（步）
D1116.05 BOOL  ; RK_07 铝壳上料移载机构Y轴铝壳取料位1（步）
D1116.06 BOOL  ; 备用
D1116.07 BOOL  ; RK_07 铝壳上料移载机构循环完成1
D1118.00 BOOL  ; RK_07 铝壳上料移载机构开始运行条件2（铝壳取料）
D1118.01 BOOL  ; RK_07 铝壳上料移载机构步进条件2（铝壳取料）
D1118.15 BOOL  ; RK_07 铝壳上料移载机构步进2（铝壳取料）
D1119 CHANNEL  ; RK_07 铝壳上料移载机构步序2（铝壳取料）
D1119.00 BOOL  ; RK_07 铝壳上料移载机构自动开始2（步）
D1119.01 BOOL  ; RK_07 铝壳上料移载机构Y轴铝壳取料位2（步）
D1119.02 BOOL  ; 备用
D1119.03 BOOL  ; RK_07 铝壳上料移载机构循环完成2
D1121.00 BOOL  ; RK_07 铝壳上料移载机构开始运行条件3（铝壳托盘卸载）
D1121.01 BOOL  ; RK_07 铝壳上料移载机构步进条件3（铝壳托盘卸载）
D1121.15 BOOL  ; RK_07 铝壳上料移载机构步进3（铝壳托盘卸载）
D1122 CHANNEL  ; RK_07 铝壳上料移载机构步序3（铝壳托盘卸载）
D1122.00 BOOL  ; RK_07 铝壳上料移载机构自动开始3（步）
D1122.01 BOOL  ; RK_07 铝壳上料移载机构Y轴铝壳托盘卸载位3（步）
D1122.02 BOOL  ; RK_07 铝壳上料移载机构#3铝壳托盘卸载电机正转3（步）
D1122.03 BOOL  ; RK_07 铝壳上料移载机构吸盘破真空3（步）
D1122.04 BOOL  ; RK_07 铝壳上料移载机构#3铝壳托盘卸载电机反转3（步）
D1122.05 BOOL  ; RK_07 铝壳上料移载机构Y轴铝壳取料位&#1/2铝壳上料位3（步）
D1122.06 BOOL  ; 备用
D1122.07 BOOL  ; RK_07 铝壳上料移载机构循环完成3
D1137.00 BOOL  ; RK_07 铝壳上料移载机构复位（M）
D1137.01 BOOL  ; RK_07 #1铝壳上料电机反转（复位）
D1137.02 BOOL  ; RK_07 #2铝壳上料电机反转（复位）
D1137.03 BOOL  ; RK_07 #3铝壳下料电机反转（复位）
D1137.04 BOOL  ; RK_07 #1铝壳上料车定位升降气缸下降（复位）
D1137.05 BOOL  ; RK_07 #1铝壳上料车定位升降气缸上升（复位）
D1137.06 BOOL  ; RK_07 #2铝壳上料车定位升降气缸下降（复位）
D1137.07 BOOL  ; RK_07 #2铝壳上料车定位升降气缸上升（复位）
D1137.08 BOOL  ; RK_07 #3托盘下料车定位升降气缸下降（复位）
D1137.09 BOOL  ; RK_07 #3托盘下料车定位升降气缸上升（复位）
D1137.10 BOOL  ; RK_07 铝壳上料移载吸盘破真空（复位）
D1137.11 BOOL  ; RK_07 铝壳上料移载吸盘立真空（复位）
D1137.12 BOOL  ; RK_07 U8_Z 铝壳上料移载Y轴回原点（复位）
D1137.13 BOOL  ; RK_07 U8_Z 铝壳上料移载Y轴铝壳取料位（复位）
D1139 CHANNEL  ; RK_07 铝壳上料移载机构步序号
D114 CHANNEL  ; 电芯进料接收条码开始字
D1140.00 BOOL  ; RK_07 #1铝壳上料升降机构初始位
D1140.07 BOOL  ; RK_07 #1铝壳上料升降机构异常标志
D1143.00 BOOL  ; RK_07 #1铝壳上料机构单步/自动循环运行中（总）
D1150.00 BOOL  ; RK_07 #2铝壳上料升降机构初始位
D1150.07 BOOL  ; RK_07 #2铝壳上料升降机构异常标志
D1153.00 BOOL  ; RK_07 #2铝壳上料机构单步/自动循环运行中（总）
D1160.00 BOOL  ; RK_07 铝壳托盘下料升降机构初始位
D1160.07 BOOL  ; RK_07 铝壳托盘下料升降机构异常标志
D1163.00 BOOL  ; RK_07 #3托盘下料机构单步/自动循环运行中（总）
D1170.00 BOOL  ; RK_08 铝壳除尘机构初始位
D1170.05 BOOL  ; RK_08 铝壳除尘机构停止标志
D1170.06 BOOL  ; RK_08 铝壳除尘机构清料完成标志
D1170.07 BOOL  ; RK_08 铝壳除尘机构异常标志
D1171.00 BOOL  ; RK_08 铝壳除尘机构运行条件
D1173.00 BOOL  ; RK_08 铝壳除尘机构单步/自动循环运行中（总）
D1173.10 BOOL  ; RK_08 铝壳除尘工站记忆显示（Lamp）
D1173.11 BOOL  ; RK_08 铝壳除尘工站初始化显示（Lamp）
D1173.13 BOOL  ; RK_08 铝壳除尘机构记忆清除（SW）
D1173.14 BOOL  ; RK_08 铝壳除尘机构复位按钮（SW）
D1173.15 BOOL  ; RK_08 铝壳除尘机构单步（SW）
D1174.00 BOOL  ; RK_08 铝壳除尘机构单步运行中
D1174.01 BOOL  ; RK_08 铝壳除尘机构单步/自动循环运行中
D1174.10 BOOL  ; RK_08 铝壳除尘机构单步运行条件
D1175.00 BOOL  ; RK_08 铝壳除尘机构开始运行条件
D1175.01 BOOL  ; RK_08 铝壳除尘机构步进条件
D1175.15 BOOL  ; RK_08 铝壳除尘机构步进
D1176 CHANNEL  ; RK_08 铝壳除尘机构步序
D1176.00 BOOL  ; RK_08 铝壳除尘机构自动开始（步）
D1176.01 BOOL  ; RK_08 铝壳除尘机构夹爪气缸夹紧（步）
D1176.02 BOOL  ; RK_08 铝壳除尘机构旋转伸缩气缸伸出（步）
D1176.03 BOOL  ; RK_08 铝壳除尘机构吹气阀开（步）
D1176.04 BOOL  ; RK_08 铝壳除尘机构吹气阀关（步）
D1176.05 BOOL  ; RK_08 铝壳除尘机构旋转伸缩气缸缩回（步）
D1176.06 BOOL  ; RK_08 铝壳除尘机构伸缩气缸伸出（步）
D1176.07 BOOL  ; RK_08 铝壳除尘机构夹爪气缸张开（步）
D1176.08 BOOL  ; RK_08 铝壳除尘机构伸缩气缸缩回（步）
D1176.09 BOOL  ; 备用
D1176.10 BOOL  ; RK_08 铝壳除尘机构循环完成
D1177.00 BOOL  ; RK_08 铝壳除尘机构复位（M）
D1177.01 BOOL  ; RK_08 铝壳除尘吹气阀关（复位）
D1177.02 BOOL  ; RK_08 铝壳除尘夹爪气缸张开（复位）
D1177.03 BOOL  ; RK_08 铝壳除尘夹爪气缸夹紧（复位）
D1177.04 BOOL  ; RK_08 铝壳除尘旋转伸缩气缸缩回（复位）
D1177.05 BOOL  ; RK_08 铝壳除尘伸缩气缸缩回（复位）
D1177.06 BOOL  ; RK_08 铝壳除尘伸缩气缸伸出（复位）
D1179 CHANNEL  ; RK_08 铝壳除尘机构步序号
D1180.00 BOOL  ; RK_09 #1Hipot检测机构初始位
D1180.05 BOOL  ; RK_09 #1Hipot检测机构停止标志
D1180.06 BOOL  ; RK_09 #1Hipot检测机构清料完成标志
D1180.07 BOOL  ; RK_09 #1Hipot检测机构异常标志
D1181.00 BOOL  ; RK_09 #1Hipot检测机构运行条件
D1183.00 BOOL  ; RK_09 #1Hipot测试机构单步/自动循环运行中（总）
D1183.10 BOOL  ; RK_09 #1Hipot检测工站记忆显示（Lamp）
D1183.11 BOOL  ; RK_09 #1Hipot检测工站初始化显示（Lamp）
D1183.13 BOOL  ; RK_09 #1Hipot检测机构记忆清除（SW）
D1183.14 BOOL  ; RK_09 #1Hipot检测机构复位按钮（SW）
D1183.15 BOOL  ; RK_09 #1Hipot检测机构单步（SW）
D1184.00 BOOL  ; RK_09 #1Hipot检测机构单步运行中
D1184.01 BOOL  ; RK_09 #1Hipot检测机构单步/自动循环运行中
D1184.10 BOOL  ; RK_09 #1Hipot检测机构单步运行条件
D1185.00 BOOL  ; RK_09 #1Hipot检测机构开始运行条件
D1185.01 BOOL  ; RK_09 #1Hipot检测机构步进条件
D1185.15 BOOL  ; RK_09 #1Hipot检测机构步进
D1186 CHANNEL  ; RK_09 #1Hipot检测机构步序
D1186.00 BOOL  ; RK_09 #1Hipot检测机构自动开始（步）
D1186.01 BOOL  ; RK_09 #1Hipot检测机构检测伸缩气缸伸出&Hipot检测数据初始化（步）
D1186.02 BOOL  ; RK_09 #1Hipot检测机构测试触发（步）
D1186.03 BOOL  ; RK_09 #1Hipot检测机构测试结果等待（步）
D1186.04 BOOL  ; RK_09 #1Hipot检测机构测试结果读取（步）
D1186.05 BOOL  ; RK_09 #1Hipot检测机构检测伸缩气缸缩回（步）
D1186.06 BOOL  ; RK_09 #1Hipot检测机构平台伸缩气缸伸出
D1186.07 BOOL  ; RK_09 #1Hipot检测机构旋转伸缩气缸伸出（步）
D1186.08 BOOL  ; RK_09 #1Hipot检测机构旋转伸缩气缸缩回（步）
D1186.09 BOOL  ; RK_09 #1Hipot检测机构平台伸缩气缸缩回（步）
D1186.10 BOOL  ; RK_09 #1Hipot检测机构循环完成
D1187.00 BOOL  ; RK_09 #1Hipot检测机构复位（M）
D1187.01 BOOL  ; RK_09 #1Hipot测试伸缩气缸缩回（复位）
D1187.02 BOOL  ; RK_09 #1Hipot测试旋转伸缩气缸缩回（复位）
D1187.03 BOOL  ; RK_09 #1Hipot测试平台伸缩气缸缩回（复位）
D1187.04 BOOL  ; RK_09 #1Hipot测试伸缩气缸伸出（复位）
D1189 CHANNEL  ; RK_09 #1Hipot检测机构步序号
D1190.00 BOOL  ; RK_09 #2Hipot检测机构初始位
D1190.05 BOOL  ; RK_09 #2Hipot检测机构停止标志
D1190.06 BOOL  ; RK_09 #2Hipot检测机构清料完成标志
D1190.07 BOOL  ; RK_09 #2Hipot检测机构异常标志
D1191.00 BOOL  ; RK_09 #2Hipot检测机构运行条件
D1193.00 BOOL  ; RK_09 #2Hipot测试机构单步/自动循环运行中（总）
D1193.10 BOOL  ; RK_09 #2Hipot检测工站记忆显示（Lamp）
D1193.11 BOOL  ; RK_09 #2Hipot检测工站初始化显示（Lamp）
D1193.13 BOOL  ; RK_09 #2Hipot检测机构记忆清除（SW）
D1193.14 BOOL  ; RK_09 #2Hipot检测机构复位按钮（SW）
D1193.15 BOOL  ; RK_09 #2Hipot检测机构单步（SW）
D1194.00 BOOL  ; RK_09 #2Hipot检测机构单步运行中
D1194.01 BOOL  ; RK_09 #2Hipot检测机构单步/自动循环运行中
D1194.10 BOOL  ; RK_09 #2Hipot检测机构单步运行条件
D1195.00 BOOL  ; RK_09 #2Hipot检测机构开始运行条件
D1195.01 BOOL  ; RK_09 #2Hipot检测机构步进条件
D1195.15 BOOL  ; RK_09 #2Hipot检测机构步进
D1196 CHANNEL  ; RK_09 #2Hipot检测机构步序
D1196.00 BOOL  ; RK_09 #2Hipot检测机构自动开始（步）
D1196.01 BOOL  ; RK_09 #2Hipot检测机构检测伸缩气缸伸出&Hipot检测数据初始化（步）
D1196.02 BOOL  ; RK_09 #2Hipot检测机构测试触发（步）
D1196.03 BOOL  ; RK_09 #2Hipot检测机构测试结果等待（步）
D1196.04 BOOL  ; RK_09 #2Hipot检测机构测试结果读取（步）
D1196.05 BOOL  ; RK_09 #2Hipot检测机构检测伸缩气缸缩回（步）
D1196.06 BOOL  ; RK_09 #2Hipot检测机构平台伸缩气缸伸出（步）
D1196.07 BOOL  ; RK_09 #2Hipot检测机构旋转伸缩气缸伸出（步）
D1196.08 BOOL  ; RK_09 #2Hipot检测机构旋转伸缩气缸缩回（步）
D1196.09 BOOL  ; RK_09 #2Hipot检测机构平台伸缩气缸缩回（步）
D1196.10 BOOL  ; RK_09 #2Hipot检测机构循环完成
D1197.00 BOOL  ; RK_09 #2Hipot检测机构复位（M）
D1197.01 BOOL  ; RK_09 #2Hipot测试伸缩气缸缩回（复位）
D1197.02 BOOL  ; RK_09 #2Hipot测试旋转伸缩气缸缩回（复位）
D1197.03 BOOL  ; RK_09 #2Hipot测试平台伸缩气缸缩回（复位）
D1199 CHANNEL  ; RK_09 #2Hipot检测机构步序号
D1200.00 BOOL  ; RK_10 电池除尘上料机构初始位
D1200.05 BOOL  ; RK_10 电池除尘上料机构停止标志
D1200.06 BOOL  ; RK_10 电池除尘上料机构清料完成标志
D1200.07 BOOL  ; RK_10 电池除尘上料机构异常标志
D1201.00 BOOL  ; RK_10 电池除尘上料机构运行条件
D1202.00 BOOL  ; RK_10 U8_U 电池除尘上料X轴运行条件
D1202.01 BOOL  ; RK_10 U8_U 电池除尘上料X轴回原点条件
D1202.15 BOOL  ; RK_10 U8_U 电池除尘上料X轴手自动运行条件
D1203.00 BOOL  ; RK_10 电池除尘上料机构单步/自动循环运行中（总）
D1203.10 BOOL  ; RK_10 电池除尘上料工站记忆显示（Lamp）
D1203.11 BOOL  ; RK_10 电池除尘上料工站初始化显示（Lamp）
D1203.13 BOOL  ; RK_10 电池除尘上料机构记忆清除（SW）
D1203.14 BOOL  ; RK_10 电池除尘上料机构复位按钮（SW）
D1203.15 BOOL  ; RK_10 电池除尘上料机构单步（SW）
D1204.00 BOOL  ; RK_10 电池除尘上料机构单步运行中
D1204.01 BOOL  ; RK_10 电池除尘上料机构单步/自动循环运行中
D1204.10 BOOL  ; RK_10 电池除尘上料机构单步运行条件
D1205.00 BOOL  ; RK_10 电池除尘上料机构开始运行条件
D1205.01 BOOL  ; RK_10 电池除尘上料机构步进条件
D1205.15 BOOL  ; RK_10 电池除尘上料机构步进
D1206 CHANNEL  ; RK_10 电池除尘上料机构步序
D1206.00 BOOL  ; RK_10 电池除尘上料机构自动开始（步）
D1206.01 BOOL  ; RK_10 电池除尘上料机构#1|#2Hipot检测取料位（步）
D1206.02 BOOL  ; RK_10 电池除尘上料机构升降气缸下降（步）
D1206.03 BOOL  ; RK_10 电池除尘上料机构夹爪气缸夹紧（步）
D1206.04 BOOL  ; RK_10 电池除尘上料机构升降气缸上升（步）
D1206.05 BOOL  ; RK_10 电池除尘上料机构Hipot NG放料位（步）
D1206.06 BOOL  ; RK_10 电池除尘上料机构Hipot OK放料位（步）
D1206.07 BOOL  ; RK_10 电池除尘上料机构升降气缸下降&Hipot NG出站MES校验结果（步）
D1206.08 BOOL  ; RK_10 电池除尘上料机构夹爪气缸张开（步）
D1206.09 BOOL  ; RK_10 电池除尘上料机构升降气缸上升（步）
D1206.10 BOOL  ; RK_10 电池除尘上料机构#1/2Hipot检测取料位（步）
D1206.11 BOOL  ; 备用
D1206.12 BOOL  ; RK_10 电池除尘上料机构循环完成
D1207.00 BOOL  ; RK_10 电池除尘上料机构复位（M）
D1207.01 BOOL  ; RK_10 电池除尘上料机械手夹爪气缸张开（复位）
D1207.02 BOOL  ; RK_10 电池除尘上料机械手夹爪气缸夹紧（复位）
D1207.03 BOOL  ; RK_10 电池除尘上料机械手升降气缸上升（复位）
D1207.04 BOOL  ; RK_10 U8_U 电池除尘上料X轴回原点（复位）
D1207.05 BOOL  ; RK_10 U8_U 电池除尘上料X轴#1Hipot检测取料位（复位）
D1209 CHANNEL  ; RK_10 电池除尘上料机构步序号
D1210.00 BOOL  ; RK_11 电池除尘机构初始位
D1210.05 BOOL  ; RK_11 电池除尘机构停止标志
D1210.06 BOOL  ; RK_11 电池除尘机构清料完成标志
D1210.07 BOOL  ; RK_11 电池除尘机构异常标志
D1211.00 BOOL  ; RK_11 电池除尘机构运行条件
D1213.00 BOOL  ; RK_11 电池除尘机构单步/自动循环运行中（总）
D1213.10 BOOL  ; RK_11 电池除尘工站记忆显示（Lamp）
D1213.11 BOOL  ; RK_11 电池除尘工站初始化显示（Lamp）
D1213.13 BOOL  ; RK_11 电池除尘机构记忆清除（SW）
D1213.14 BOOL  ; RK_11 电池除尘机构复位按钮（SW）
D1213.15 BOOL  ; RK_11 电池除尘机构单步（SW）
D1214.00 BOOL  ; RK_11 电池除尘机构单步运行中
D1214.01 BOOL  ; RK_11 电池除尘机构单步/自动循环运行中
D1214.10 BOOL  ; RK_11 电池除尘机构单步运行条件
D1215.00 BOOL  ; RK_11 电池除尘机构开始运行条件
D1215.01 BOOL  ; RK_11 电池除尘机构步进条件
D1215.15 BOOL  ; RK_11 电池除尘机构步进
D1216 CHANNEL  ; RK_11 电池除尘机构步序
D1216.00 BOOL  ; RK_11 电池除尘机构自动开始（步）
D1216.01 BOOL  ; RK_11 电池除尘机构夹爪气缸夹紧（步）
D1216.02 BOOL  ; RK_11 电池除尘机构伸缩气缸伸出（步）
D1216.03 BOOL  ; RK_11 电池除尘机构吹气阀开（步）
D1216.04 BOOL  ; RK_11 电池除尘机构吹气阀关（步）
D1216.05 BOOL  ; RK_11 电池除尘机构伸缩气缸缩回（步）
D1216.06 BOOL  ; RK_11 电池除尘机构旋转伸缩气缸缩回（步）
D1216.07 BOOL  ; RK_11 电池除尘机构夹爪气缸张开（步）
D1216.08 BOOL  ; RK_11 电池除尘机构旋转伸缩气缸伸出（步）
D1216.09 BOOL  ; 备用
D1216.10 BOOL  ; RK_11 电池除尘机构循环完成
D1217.00 BOOL  ; RK_11 电池除尘机构复位（M）
D1217.01 BOOL  ; RK_11 电池除尘夹爪气缸张开（复位）
D1217.02 BOOL  ; RK_11 电池除尘夹爪气缸夹紧（复位）
D1217.03 BOOL  ; RK_11 电池除尘伸缩气缸缩回（复位）
D1217.04 BOOL  ; RK_11 电池除尘旋转伸缩气缸伸出（复位）
D1217.05 BOOL  ; RK_11 电池除尘吹气阀关（复位）
D1219 CHANNEL  ; RK_11 电池除尘机构步序号
D1220.00 BOOL  ; RK_12 预焊上下料机构初始位
D1220.05 BOOL  ; RK_12 预焊上下料构停止标志
D1220.06 BOOL  ; RK_12 预焊上下料机构清料完成标志
D1220.07 BOOL  ; RK_12 预焊上下料机构异常标志
D1220.08 BOOL  ; RK_12 轮廓检测NG拨料气缸异常标志
D1221.00 BOOL  ; RK_12 预焊上下料机构运行条件（公共）
D1221.01 BOOL  ; RK_12 预焊上下料机构运行条件1（预焊电池取料）
D1221.02 BOOL  ; RK_12 预焊上下料机构运行条件2（预焊电池放料）
D1221.03 BOOL  ; RK_12 预焊上下料机构运行条件3（OK/NG电池取料）
D1221.04 BOOL  ; RK_12 预焊上下料机构运行条件4（OK/NG电池放料）
D1221.05 BOOL  ; RK_12 预焊上下料机构预焊电池取料
D1221.06 BOOL  ; RK_12 预焊上下料机构预焊电池放料
D1221.07 BOOL  ; RK_12 预焊上下料机构OK/NG电池取料
D1221.08 BOOL  ; RK_12 预焊上下料机构OK/NG电池放料
D1222.00 BOOL  ; RK_12 U4_X 预焊上下料X轴运行条件
D1222.01 BOOL  ; RK_12 U4_X 预焊上下料X轴回原点条件
D1222.02 BOOL  ; RK_12 U4_Y 预焊上料Z轴运行条件
D1222.03 BOOL  ; RK_12 U4_Y 预焊上料Z轴回原点条件
D1222.04 BOOL  ; RK_12 U4_Y 预焊上料Z轴除尘取料位条件
D1222.05 BOOL  ; RK_12 U4_Y 预焊上料Z轴#1移载放料位条件
D1222.06 BOOL  ; RK_12 U4_Y 预焊上料Z轴#2移载放料位条件
D1222.08 BOOL  ; RK_12 U4_Z 预焊下料Z轴运行条件
D1222.09 BOOL  ; RK_12 U4_Z 预焊下料Z轴回原点条件
D1222.10 BOOL  ; RK_12 U4_Z 预焊下料Z轴#1移载取料位条件
D1222.11 BOOL  ; RK_12 U4_Z 预焊下料Z轴#2移载取料位条件
D1222.12 BOOL  ; RK_12 U4_Z 预焊下料Z轴OK放料位条件
D1222.13 BOOL  ; RK_12 U4_Z 预焊下料Z轴#1NG放料位条件
D1222.14 BOOL  ; RK_12 U4_Z 预焊下料Z轴#2NG放料位条件
D1222.15 BOOL  ; RK_12 U4_X 预焊上下料X轴手自动运行条件
D1223.00 BOOL  ; RK_12 预焊上下料机构单步/自动循环运行中（总）
D1223.09 BOOL  ; RK_12 预焊上下料工站初始化显示（Lamp）
D1223.10 BOOL  ; RK_12 预焊上下料工站记忆显示（Lamp）
D1223.11 BOOL  ; RK_12 #1/2轮廓NG槽记忆显示（Lamp）
D1223.12 BOOL  ; RK_12 OK出料拉带记忆显示（Lamp）
D1223.13 BOOL  ; RK_12 预焊上下料机构记忆清除（SW）
D1223.14 BOOL  ; RK_12 预焊上下料机构复位按钮（SW）
D1223.15 BOOL  ; RK_12 预焊上下料机构单步（SW）
D1224.00 BOOL  ; RK_12 预焊上下料机构单步运行中1（预焊电池取料）
D1224.01 BOOL  ; RK_12 预焊上下料机构单步/自动循环运行中1（预焊电池取料）
D1224.02 BOOL  ; RK_12 预焊上下料机构单步运行中2（预焊电池放料）
D1224.03 BOOL  ; RK_12 预焊上下料机构单步/自动循环运行中2（预焊电池放料）
D1224.04 BOOL  ; RK_12 预焊上下料机构单步运行中3（OK/NG电池取料）
D1224.05 BOOL  ; RK_12 预焊上下料机构单步/自动循环运行中3（OK/NG电池取料）
D1224.06 BOOL  ; RK_12 预焊上下料机构单步运行中4（OK/NG电池放料）
D1224.07 BOOL  ; RK_12 预焊上下料机构单步/自动循环运行中4（OK/NG电池放料）
D1224.10 BOOL  ; RK_12 预焊上下料机构单步运行条件1（预焊电池取料）
D1224.11 BOOL  ; RK_12 预焊上下料机构单步运行条件2（预焊电池放料）
D1224.12 BOOL  ; RK_12 预焊上下料机构单步运行条件3（OK/NG电池取料）
D1224.13 BOOL  ; RK_12 预焊上下料机构单步运行条件4（OK/NG电池放料）
D1225.00 BOOL  ; RK_12 预焊上下料机构开始运行条件1（预焊电池取料）
D1225.01 BOOL  ; RK_12 预焊上下料机构步进条件1（预焊电池取料）
D1225.15 BOOL  ; RK_12 预焊上下料机构步进1（预焊电池取料）
D1226 CHANNEL  ; RK_12 预焊上下料机构步序1（预焊电池取料）
D1226.00 BOOL  ; RK_12 预焊上下料机构自动开始1（步）
D1226.01 BOOL  ; RK_12 预焊上下料机构X轴除尘取料位1（步）
D1226.02 BOOL  ; RK_12 预焊上下料机构上料Z轴除尘取料位1（步）
D1226.03 BOOL  ; RK_12 预焊上下料机构上料夹爪气缸夹紧1（步）
D1226.04 BOOL  ; RK_12 预焊上下料机构上料Z轴待料位1（步）
D1226.05 BOOL  ; RK_12 预焊上下料机构X轴#1移载放料位1（步）
D1226.06 BOOL  ; RK_12 预焊上下料机构循环完成1
D1228.00 BOOL  ; RK_12 预焊上下料机构开始运行条件2（预焊电池放料）
D1228.01 BOOL  ; RK_12 预焊上下料机构步进条件2（预焊电池放料）
D1228.15 BOOL  ; RK_12 预焊上下料机构步进2（预焊电池放料）
D1229 CHANNEL  ; RK_12 预焊上下料机构步序2（预焊电池放料）
D1229.00 BOOL  ; RK_12 预焊上下料机构自动开始2（步）
D1229.01 BOOL  ; RK_12 预焊上下料机构X轴#1|#2移载放料位2（步）
D1229.02 BOOL  ; RK_12 预焊上下料机构上料Z轴#1|#2移载放料位2（步）
D1229.03 BOOL  ; RK_12 预焊上下料机构上料夹爪气缸张开2（步）
D1229.04 BOOL  ; RK_12 预焊上下料机构上料Z轴待料位2（步）
D1229.05 BOOL  ; 备用
D1229.06 BOOL  ; RK_12 预焊上下料机构循环完成2
D1231.00 BOOL  ; RK_12 预焊上下料机构开始运行条件3（OK/NG电池取料）
D1231.01 BOOL  ; RK_12 预焊上下料机构步进条件3（OK/NG电池取料）
D1231.15 BOOL  ; RK_12 预焊上下料机构步进3（OK/NG电池取料）
D1232 CHANNEL  ; RK_12 预焊上下料机构步序3（OK/NG电池取料）
D1232.00 BOOL  ; RK_12 预焊上下料机构自动开始3（步）
D1232.01 BOOL  ; RK_12 预焊上下料机构X轴#1|#2移载取料位3（步）
D1232.02 BOOL  ; RK_12 预焊上下料机构下料Z轴#1|#2移载取料位3（步）
D1232.03 BOOL  ; RK_12 预焊上下料机构下料夹爪气缸夹紧3（步）
D1232.04 BOOL  ; RK_12 预焊上下料机构下料Z轴待料位3（步）
D1232.05 BOOL  ; 备用
D1232.06 BOOL  ; RK_12 预焊上下料机构循环完成3
D1234.00 BOOL  ; RK_12 预焊上下料机构开始运行条件4（OK/NG电池放料）
D1234.01 BOOL  ; RK_12 预焊上下料机构步进条件4（OK/NG电池放料）
D1234.15 BOOL  ; RK_12 预焊上下料机构步进4（OK/NG电池放料）
D1235 CHANNEL  ; RK_12 预焊上下料机构步序4（OK/NG电池放料）
D1235.00 BOOL  ; RK_12 预焊上下料机构自动开始4（步）
D1235.01 BOOL  ; RK_12 预焊上下料机构出站MES校验结果4（步）
D1235.02 BOOL  ; RK_12 预焊上下料机构X轴OK|#1|#2NG放料位4（步）
D1235.03 BOOL  ; RK_12 预焊上下料机构下料Z轴OK|#1|#2NG放料位4（步）
D1235.04 BOOL  ; RK_12 预焊上下料机构下料夹爪气缸张开4（步）
D1235.05 BOOL  ; RK_12 预焊上下料机构下料Z轴待料位4（步）
D1235.06 BOOL  ; RK_12 预焊上下料机构X轴#1移载放料位4（步）
D1235.07 BOOL  ; RK_12 预焊上下料机构循环完成4
D1237.00 BOOL  ; RK_12 预焊上下料机构复位（M）
D1237.01 BOOL  ; RK_12 预焊上料机械手夹爪气缸张开（复位）
D1237.02 BOOL  ; RK_12 预焊上料机械手夹爪气缸夹紧（复位）
D1237.03 BOOL  ; RK_12 预焊下料机械手夹爪气缸张开（复位）
D1237.04 BOOL  ; RK_12 预焊下料机械手夹爪气缸夹紧（复位）
D1237.05 BOOL  ; RK_12 U4_Y 预焊上料Z轴回原点（复位）
D1237.06 BOOL  ; RK_12 U4_Y 预焊上料Z轴待料位（复位）
D1237.07 BOOL  ; RK_12 U4_Z 预焊下料Z轴回原点（复位）
D1237.08 BOOL  ; RK_12 U4_Z 预焊下料Z轴待料位（复位）
D1237.09 BOOL  ; RK_12 U4_X 预焊上下料X轴回原点（复位）
D1237.10 BOOL  ; RK_12 U4_X 预焊上下料X轴#1移载放料位（复位）
D1237.11 BOOL  ; RK_12 轮廓检测NG拨料气缸缩回（复位）
D1239 CHANNEL  ; RK_12 预焊上下料机构步序号
D1240.00 BOOL  ; RK_13 #1移载机构初始位
D1240.05 BOOL  ; RK_13 #1移载机构停止标志
D1240.06 BOOL  ; RK_13 #1移载机构清料完成标志
D1240.07 BOOL  ; RK_13 #1移载机构异常标志
D1241.00 BOOL  ; RK_13 #1移载机构运行条件
D1242.00 BOOL  ; RK_13 U4_U #1移载Y轴运行条件
D1242.01 BOOL  ; RK_13 U4_U #1移载Y轴回原点条件
D1242.15 BOOL  ; RK_13 U4_U #1移载Y轴手自动运行条件
D1243.00 BOOL  ; RK_13 #1移载机构单步/自动循环运行中（总）
D1243.10 BOOL  ; RK_13 #1移载工站记忆显示（Lamp）
D1243.11 BOOL  ; RK_13 #1移载工站初始化显示（Lamp）
D1243.13 BOOL  ; RK_13 #1移载机构记忆清除（SW）
D1243.14 BOOL  ; RK_13 #1移载机构复位按钮（SW）
D1243.15 BOOL  ; RK_13 #1移载机构单步（SW）
D1244.00 BOOL  ; RK_13 #1移载机构单步运行中
D1244.01 BOOL  ; RK_13 #1移载机构单步/自动循环运行中
D1244.10 BOOL  ; RK_13 #1移载机构单步运行条件
D1245.00 BOOL  ; RK_13 #1移载机构开始运行条件
D1245.01 BOOL  ; RK_13 #1移载机构步进条件
D1245.15 BOOL  ; RK_13 #1移载机构步进
D1246 CHANNEL  ; RK_13 #1移载机构步序
D1246.00 BOOL  ; RK_13 #1移载机构自动开始（步）
D1246.01 BOOL  ; RK_13 #1移载机构升降气缸上升（步）
D1246.02 BOOL  ; RK_13 #1移载机构升降气缸下降（步）
D1246.03 BOOL  ; RK_13 #1移载机构左右定位伸缩气缸伸出（步）
D1246.04 BOOL  ; RK_13 #1移载机构Y轴压装位&导向#1/2伸缩气缸伸出（步）
D1246.05 BOOL  ; RK_13 #1移载机构导向#1/2伸缩气缸伸出（步）
D1246.06 BOOL  ; RK_13 #1移载机构定位#1/2伸缩气缸缩回（步）
D1246.07 BOOL  ; 预留
D1246.08 BOOL  ; RK_13 #1移载机构Y轴#1/2点轮廓检测位（步）
D1246.09 BOOL  ; RK_13 #1移载机构Y轴#1/2点轮廓检测结果（步）
D1246.10 BOOL  ; RK_13 #1移载机构Y轴#3/4点轮廓检测位（步）
D1246.11 BOOL  ; RK_13 #1移载机构Y轴#3/4点轮廓检测结果（步）
D1246.12 BOOL  ; RK_13 #1移载机构Y轴激光焊接位（步）
D1246.13 BOOL  ; 预留
D1246.14 BOOL  ; RK_13 #1移载机构Y轴取放料位（步）
D1246.15 BOOL  ; RK_13 #1移载机构定位#1/2伸缩气缸伸出&左右定位伸缩气缸缩回&导向#1/2伸缩气缸缩回（步）
D1247.00 BOOL  ; 预留
D1247.01 BOOL  ; RK_13 #1移载机构升降气缸上升（步）
D1247.02 BOOL  ; RK_13 #1移载机构升降气缸下降（步）
D1247.03 BOOL  ; 预留
D1247.04 BOOL  ; RK_13 #1移载机构循环完成
D1248.00 BOOL  ; RK_13 #1移载机构复位（M）
D1248.01 BOOL  ; RK_13 #1移载导向#1/2伸缩气缸缩回（复位）
D1248.02 BOOL  ; RK_13 #1移载定位#1/2伸缩气缸伸出（复位）
D1248.03 BOOL  ; RK_13 #1移载左右定位伸缩气缸缩回（复位）
D1248.04 BOOL  ; RK_13 #1移载升降气缸下降（复位）
D1248.05 BOOL  ; RK_13 #1移载导向#1/2伸缩气缸伸出（复位）
D1248.06 BOOL  ; RK_13 #1移载升降气缸下降（复位）
D1248.07 BOOL  ; RK_13 #1移载定位#1/2伸缩气缸缩回（复位）
D1248.08 BOOL  ; RK_13 #1移载左右定位伸缩气缸伸出（复位）
D1248.09 BOOL  ; RK_13 U4_U #1移载Y轴回原点（复位）
D1248.10 BOOL  ; RK_13 U4_U #1移载Y轴取放料位（复位）
D1249 CHANNEL  ; RK_13 #1移载机构步序号
D1250.00 BOOL  ; RK_13 #2移载机构初始位
D1250.05 BOOL  ; RK_13 #2移载机构停止标志
D1250.06 BOOL  ; RK_13 #2移载机构清料完成标志
D1250.07 BOOL  ; RK_13 #2移载机构异常标志
D1251.00 BOOL  ; RK_13 #2移载机构运行条件
D1252.00 BOOL  ; RK_13 U6_X #2移载Y轴运行条件
D1252.01 BOOL  ; RK_13 U6_X #2移载Y轴回原点条件
D1252.15 BOOL  ; RK_13 U6_X #2移载Y轴手自动运行条件
D1253.00 BOOL  ; RK_13 #2移载机构单步/自动循环运行中（总）
D1253.10 BOOL  ; RK_13 #2移载工站记忆显示（Lamp）
D1253.11 BOOL  ; RK_13 #2移载工站初始化显示（Lamp）
D1253.13 BOOL  ; RK_13 #2移载机构记忆清除（SW）
D1253.14 BOOL  ; RK_13 #2移载机构复位按钮（SW）
D1253.15 BOOL  ; RK_13 #2移载机构单步（SW）
D1254.00 BOOL  ; RK_13 #2移载机构单步运行中
D1254.01 BOOL  ; RK_13 #2移载机构单步/自动循环运行中
D1254.10 BOOL  ; RK_13 #2移载机构单步运行条件
D1255.00 BOOL  ; RK_13 #2移载机构开始运行条件
D1255.01 BOOL  ; RK_13 #2移载机构步进条件
D1255.15 BOOL  ; RK_13 #2移载机构步进
D1256 CHANNEL  ; RK_13 #2移载机构步序
D1256.00 BOOL  ; RK_13 #2移载机构自动开始（步）
D1256.01 BOOL  ; RK_13 #2移载机构升降气缸上升（步）
D1256.02 BOOL  ; RK_13 #2移载机构升降气缸下降（步）
D1256.03 BOOL  ; RK_13 #2移载机构左右定位伸缩气缸伸出（步）
D1256.04 BOOL  ; RK_13 #2移载机构Y轴压装位&导向#1/2伸缩气缸伸出（步）
D1256.05 BOOL  ; RK_13 #2移载机构导向#1/2伸缩气缸伸出（步）
D1256.06 BOOL  ; RK_13 #2移载机构定位#1/2伸缩气缸缩回（步）
D1256.07 BOOL  ; 预留
D1256.08 BOOL  ; RK_13 #2移载机构Y轴#1/2点轮廓检测位（步）
D1256.09 BOOL  ; RK_13 #2移载机构Y轴#1/2点轮廓检测结果（步）
D1256.10 BOOL  ; RK_13 #2移载机构Y轴#3/4点轮廓检测位（步）
D1256.11 BOOL  ; RK_13 #2移载机构Y轴#3/4点轮廓检测结果（步）
D1256.12 BOOL  ; RK_13 #2移载机构Y轴激光焊接位（步）
D1256.13 BOOL  ; 预留
D1256.14 BOOL  ; RK_13 #2移载机构Y轴取放料位（步）
D1256.15 BOOL  ; RK_13 #2移载机构定位#1/2伸缩气缸伸出&左右定位伸缩气缸缩回&导向#1/2伸缩气缸缩回（步）
D1257.00 BOOL  ; 预留
D1257.01 BOOL  ; RK_13 #2移载机构升降气缸上升（步）
D1257.02 BOOL  ; RK_13 #2移载机构升降气缸下降（步）
D1257.03 BOOL  ; 预留
D1257.04 BOOL  ; RK_13 #2移载机构循环完成
D1258.00 BOOL  ; RK_13 #2移载机构复位（M）
D1258.01 BOOL  ; RK_13 #2移载导向#1/2伸缩气缸缩回（复位）
D1258.02 BOOL  ; RK_13 #2移载定位#1/2伸缩气缸伸出（复位）
D1258.03 BOOL  ; RK_13 #2移载左右定位伸缩气缸缩回（复位）
D1258.04 BOOL  ; RK_13 #2移载升降气缸下降（复位）
D1258.05 BOOL  ; RK_13 #2移载导向#1/2伸缩气缸伸出（复位）
D1258.06 BOOL  ; RK_13 #2移载升降气缸下降（复位）
D1258.07 BOOL  ; RK_13 #2移载定位#1/2伸缩气缸缩回（复位）
D1258.08 BOOL  ; RK_13 #2移载左右定位伸缩气缸伸出（复位）
D1258.09 BOOL  ; RK_13 U6_X #2移载Y轴回原点（复位）
D1258.10 BOOL  ; RK_13 U6_X #2移载Y轴取放料位（复位）
D1259 CHANNEL  ; RK_13 #2移载机构步序号
D1260.00 BOOL  ; RK_14 #1压装机构初始位
D1260.05 BOOL  ; RK_14 #1压装机构停止标志
D1260.06 BOOL  ; RK_14 #1压装机构清料完成标志
D1260.07 BOOL  ; RK_14 #1压装机构异常标志
D1261.00 BOOL  ; RK_14 #1压装机构运行条件
D1263.00 BOOL  ; RK_14 #1压装机构单步/自动循环运行中（总）
D1263.10 BOOL  ; RK_14 #1压装工站记忆显示（Lamp）
D1263.11 BOOL  ; RK_14 #1压装工站初始化显示（Lamp）
D1263.13 BOOL  ; RK_14 #1压装机构记忆清除（SW）
D1263.14 BOOL  ; RK_14 #1压装机构复位按钮（SW）
D1263.15 BOOL  ; RK_14 #1压装机构单步（SW）
D1264.00 BOOL  ; RK_14 #1压装机构单步运行中
D1264.01 BOOL  ; RK_14 #1压装机构单步/自动循环运行中
D1264.10 BOOL  ; RK_14 #1压装机构单步运行条件
D1265.00 BOOL  ; RK_14 #1压装机构开始运行条件
D1265.01 BOOL  ; RK_14 #1压装机构步进条件
D1265.15 BOOL  ; RK_14 #1压装机构步进
D1266 CHANNEL  ; RK_14 #1压装机构步序
D1266.00 BOOL  ; RK_14 #1压装机构自动开始（步）
D1266.01 BOOL  ; 备用
D1266.02 BOOL  ; 备用
D1266.03 BOOL  ; 备用
D1266.04 BOOL  ; RK_14 #1压装机构压装升降气缸下降（步）
D1266.05 BOOL  ; 备用
D1266.06 BOOL  ; RK_14 #1压装机构压装升降气缸上升（步）
D1266.07 BOOL  ; 备用
D1266.08 BOOL  ; RK_14 #1压装机构循环完成
D1267.00 BOOL  ; RK_14 #1压装机构复位（M）
D1267.01 BOOL  ; RK_14 #1压装吸盘破真空（复位）
D1267.02 BOOL  ; RK_14 #1压装#1/2吸盘升降气缸上升（复位）
D1267.03 BOOL  ; RK_14 #1压装升降气缸上升（复位）
D1269 CHANNEL  ; RK_14 #1压装机构步序号
D1270.00 BOOL  ; RK_14 #2压装机构初始位
D1270.05 BOOL  ; RK_14 #2压装机构停止标志
D1270.06 BOOL  ; RK_14 #2压装机构清料完成标志
D1270.07 BOOL  ; RK_14 #2压装机构异常标志
D1271.00 BOOL  ; RK_14 #2压装机构运行条件
D1273.00 BOOL  ; RK_14 #2压装机构单步/自动循环运行中（总）
D1273.10 BOOL  ; RK_14 #2压装工站记忆显示（Lamp）
D1273.11 BOOL  ; RK_14 #2压装工站初始化显示（Lamp）
D1273.13 BOOL  ; RK_14 #2压装机构记忆清除（SW）
D1273.14 BOOL  ; RK_14 #2压装机构复位按钮（SW）
D1273.15 BOOL  ; RK_14 #2压装机构单步（SW）
D1274.00 BOOL  ; RK_14 #2压装机构单步运行中
D1274.01 BOOL  ; RK_14 #2压装机构单步/自动循环运行中
D1274.10 BOOL  ; RK_14 #2压装机构单步运行条件
D1275.00 BOOL  ; RK_14 #2压装机构开始运行条件
D1275.01 BOOL  ; RK_14 #2压装机构步进条件
D1275.15 BOOL  ; RK_14 #2压装机构步进
D1276 CHANNEL  ; RK_14 #2压装机构步序
D1276.00 BOOL  ; RK_14 #2压装机构自动开始（步）
D1276.01 BOOL  ; 备用
D1276.02 BOOL  ; 备用
D1276.03 BOOL  ; 备用
D1276.04 BOOL  ; RK_14 #2压装机构压装升降气缸下降（步）
D1276.05 BOOL  ; 备用
D1276.06 BOOL  ; RK_14 #2压装机构压装升降气缸上升（步）
D1276.07 BOOL  ; 备用
D1276.08 BOOL  ; RK_14 #2压装机构循环完成
D1277.00 BOOL  ; RK_14 #2压装机构复位（M）
D1277.01 BOOL  ; RK_14 #2压装吸盘破真空（复位）
D1277.02 BOOL  ; RK_14 #2压装#1/2吸盘升降气缸上升（复位）
D1277.03 BOOL  ; RK_14 #2压装升降气缸上升（复位）
D1279 CHANNEL  ; RK_14 #2压装机构步序号
D1280.00 BOOL  ; RK_15 轮廓检测机构初始位
D1280.05 BOOL  ; RK_15 轮廓检测机构停止标志
D1280.06 BOOL  ; RK_15 轮廓检测机构清料完成标志
D1280.07 BOOL  ; RK_15 轮廓检测机构异常标志
D1281.00 BOOL  ; RK_15 轮廓检测机构运行条件
D1283.00 BOOL  ; RK_15 轮廓检测机构单步/自动循环运行中（总）
D1283.10 BOOL  ; RK_15 轮廓检测工站记忆显示（Lamp）
D1283.11 BOOL  ; RK_15 轮廓检测工站初始化显示（Lamp）
D1283.13 BOOL  ; RK_15 轮廓检测机构记忆清除（SW）
D1283.14 BOOL  ; RK_15 轮廓检测机构复位按钮（SW）
D1283.15 BOOL  ; RK_15 轮廓检测机构单步（SW）
D1284.00 BOOL  ; RK_15 轮廓检测机构单步运行中
D1284.01 BOOL  ; RK_15 轮廓检测机构单步/自动循环运行中
D1284.10 BOOL  ; RK_15 轮廓检测机构单步运行条件
D1285.00 BOOL  ; RK_15 轮廓检测机构开始运行条件
D1285.01 BOOL  ; RK_15 轮廓检测机构步进条件
D1285.02 BOOL  ; RK_15 轮廓检测机构步进条件辅助
D1285.15 BOOL  ; RK_15 轮廓检测机构步进
D1286 CHANNEL  ; RK_15 轮廓检测机构步序
D1286.00 BOOL  ; RK_15 轮廓检测机构自动开始（步）
D1286.01 BOOL  ; RK_15 轮廓检测机构测量数据初始化（步）
D1286.02 BOOL  ; RK_15 轮廓检测机构#1伸缩气缸伸出|缩回&#2伸缩气缸伸出&#1/2移载#1/4点检测程序切换（步）
D1286.03 BOOL  ; RK_15 轮廓检测机构#1点测量数据读取（步）
D1286.04 BOOL  ; RK_15 轮廓检测机构#1点检测结果（步）
D1286.05 BOOL  ; RK_15 轮廓检测机构#2伸缩气缸缩回&#1/2移载#2/3点检测程序切换（步）
D1286.06 BOOL  ; RK_15 轮廓检测机构#2点测量数据读取（步）
D1286.07 BOOL  ; RK_15 轮廓检测机构#2点检测结果（步）
D1286.08 BOOL  ; RK_15 轮廓检测机构#2伸缩气缸缩回&#1/2移载#2/3点检测程序切换（步）
D1286.09 BOOL  ; RK_15 轮廓检测机构#3点测量数据读取（步）
D1286.10 BOOL  ; RK_15 轮廓检测机构#3点检测结果（步）
D1286.11 BOOL  ; RK_15 轮廓检测机构#2伸缩气缸伸出&#1/2移载#1/4点检测程序切换（步）
D1286.12 BOOL  ; RK_15 轮廓检测机构#4点测量数据读取（步）
D1286.13 BOOL  ; RK_15 轮廓检测机构#4点检测结果（步）
D1286.14 BOOL  ; RK_15 轮廓检测机构最终检测结果（步）
D1286.15 BOOL  ; RK_15 轮廓检测机构循环完成
D1297.00 BOOL  ; RK_15 轮廓检测机构复位（M）
D1297.01 BOOL  ; RK_15 轮廓检测#1伸缩气缸缩回（复位）
D1297.02 BOOL  ; RK_15 轮廓检测#2伸缩气缸伸出（复位）
D1299 CHANNEL  ; RK_15 轮廓检测机构步序号
D1300.00 BOOL  ; RK_16 焊接机构初始位
D1300.05 BOOL  ; RK_16 焊接机构停止标志
D1300.06 BOOL  ; RK_16 焊接机构清料完成标志
D1300.07 BOOL  ; RK_16 焊接机构异常标志
D1301.00 BOOL  ; RK_16 焊接机构运行条件
D1302.00 BOOL  ; RK_16 U6_Y 激光焊接X轴运行条件
D1302.01 BOOL  ; RK_16 U6_Y 激光焊接X轴回原点条件
D1302.02 BOOL  ; RK_16 U6_Z 激光焊接Z轴运行条件
D1302.03 BOOL  ; RK_16 U6_Z 激光焊接Z轴回原点条件
D1302.14 BOOL  ; RK_16 U6_Z 激光焊接Z轴手自动运行条件
D1302.15 BOOL  ; RK_16 U6_Y 激光焊接X轴手自动运行条件
D1303.00 BOOL  ; RK_16 焊接机构单步/自动循环运行中（总）
D1303.10 BOOL  ; RK_16 焊接工站记忆显示（Lamp）
D1303.11 BOOL  ; RK_16 焊接工站初始化显示（Lamp）
D1303.13 BOOL  ; RK_16 焊接机构记忆清除（SW）
D1303.14 BOOL  ; RK_16 焊接机构复位按钮（SW）
D1303.15 BOOL  ; RK_16 焊接机构单步（SW）
D1304.00 BOOL  ; RK_16 焊接机构单步运行中
D1304.01 BOOL  ; RK_16 焊接机构单步/自动循环运行中
D1304.10 BOOL  ; RK_16 焊接机构单步运行条件
D1305.00 BOOL  ; RK_16 焊接机构开始运行条件
D1305.01 BOOL  ; RK_16 焊接机构步进条件
D1305.15 BOOL  ; RK_16 焊接机构步进
D1306 CHANNEL  ; RK_16 焊接机构步序
D1306.00 BOOL  ; RK_16 焊接机构自动开始（步）
D1306.01 BOOL  ; RK_16 焊接机构X轴#1/2移载焊接位（步）
D1306.02 BOOL  ; RK_16 焊接机构Z轴#1/2移载焊接位（步）
D1306.03 BOOL  ; RK_16 焊接机构焊接触发（步）
D1306.04 BOOL  ; 备用
D1306.05 BOOL  ; RK_16 焊接机构Z轴待机位（步）
D1306.06 BOOL  ; 备用
D1306.07 BOOL  ; RK_16 焊接机构循环完成
D1317.00 BOOL  ; RK_16 焊接机构复位（M）
D1317.01 BOOL  ; RK_16 U6_Z 激光焊接Z轴回原点（复位）
D1317.02 BOOL  ; RK_16 U6_Z 激光焊接Z轴待机位（复位）
D1317.03 BOOL  ; RK_16 U6_Y 激光焊接X轴回原点（复位）
D1317.04 BOOL  ; RK_16 U6_Y 激光焊接X轴#1移载焊接位（复位）
D1319 CHANNEL  ; RK_16 焊接机构步序号
D139 CHANNEL  ; 电芯进料扫码数据结束字
D14 CHANNEL  ; 感应器ON延时设定值
D140 CHANNEL  ; 电芯进料实际条码开始字
D159 CHANNEL  ; 电芯进料实际条码结束字
D16 CHANNEL  ; 感应器延时时间
D17 CHANNEL  ; 伺服故障/准备好了信号延时
D18 CHANNEL  ; 自动运行条件延时时间
D1890 CHANNEL  ; 最近调出序号
D1892 CHANNEL  ; 最近保存序号
D1894 CHANNEL  ; 需要保存的参数序号
D1896 CHANNEL  ; 需要调出的参数序号
D19 CHANNEL  ; 自动运行步间间隔时间
D199 CHANNEL  ; NG扫码重试次数设置
D20000 CHANNEL  ; U0- 操作数据区域定义
D20001 CHANNEL  ; U0- 操作数据区域开始字
D20002 CHANNEL  ; U0- 轴参数定义
D20003 CHANNEL  ; U0- 未被使用
D20004 CHANNEL  ; RK_01 U0_X 电芯来料Y轴轴输入输出设定
D20005 CHANNEL  ; RK_01 U0_X 电芯来料Y轴轴操作模式选择
D20006 CHANNEL  ; RK_01 U0_X 电芯来料Y轴轴最高速度
D20007 CHANNEL  ; RK_01 U0_X 电芯来料Y轴轴最高速度
D20008 CHANNEL  ; RK_01 U0_X 电芯来料Y轴轴初始速度
D20009 CHANNEL  ; RK_01 U0_X 电芯来料Y轴轴初始速度
D20010 CHANNEL  ; RK_01 U0_X 电芯来料Y轴轴原点搜索高速
D20011 CHANNEL  ; RK_01 U0_X 电芯来料Y轴轴原点搜索高速
D20012 CHANNEL  ; RK_01 U0_X 电芯来料Y轴轴原点搜索接近速度
D20013 CHANNEL  ; RK_01 U0_X 电芯来料Y轴轴原点搜索接近速度
D20014 CHANNEL  ; RK_01 U0_X 电芯来料Y轴轴原点补偿值
D20015 CHANNEL  ; RK_01 U0_X 电芯来料Y轴轴原点补偿值
D20016 CHANNEL  ; RK_01 U0_X 电芯来料Y轴轴间隙补偿
D20017 CHANNEL  ; RK_01 U0_X 电芯来料Y轴轴间隙补偿速度
D20018 CHANNEL  ; RK_01 U0_X 电芯来料Y轴轴间隙补偿速度
D20019 CHANNEL  ; RK_01 U0_X 电芯来料Y轴轴加减速曲线
D20020 CHANNEL  ; RK_01 U0_X 电芯来料Y轴轴原点搜索加速时间
D20021 CHANNEL  ; RK_01 U0_X 电芯来料Y轴轴原点搜索加速时间
D20022 CHANNEL  ; RK_01 U0_X 电芯来料Y轴轴原点搜索减速时间
D20023 CHANNEL  ; RK_01 U0_X 电芯来料Y轴轴原点搜索减速时间
D20024 CHANNEL  ; RK_01 U0_X 电芯来料Y轴轴定位监测时间
D20025 CHANNEL  ; RK_01 U0_X 电芯来料Y轴轴负软限位
D20026 CHANNEL  ; RK_01 U0_X 电芯来料Y轴轴负软限位
D20027 CHANNEL  ; RK_01 U0_X 电芯来料Y轴轴正软限位
D20028 CHANNEL  ; RK_01 U0_X 电芯来料Y轴轴正软限位
D20029 CHANNEL  ; RK_01 U0_X 电芯来料Y轴轴为PCU保留
D20030 CHANNEL  ; RK_01 U0_X 电芯来料Y轴轴为PCU保留
D20031 CHANNEL  ; RK_01 U0_X 电芯来料Y轴轴初始脉冲定义
D20032 CHANNEL  ; RK_02 U0_Y 电芯进料X轴轴输入输出设定
D20033 CHANNEL  ; RK_02 U0_Y 电芯进料X轴轴操作模式选择
D20034 CHANNEL  ; RK_02 U0_Y 电芯进料X轴轴最高速度
D20035 CHANNEL  ; RK_02 U0_Y 电芯进料X轴轴最高速度
D20036 CHANNEL  ; RK_02 U0_Y 电芯进料X轴轴初始速度
D20037 CHANNEL  ; RK_02 U0_Y 电芯进料X轴轴初始速度
D20038 CHANNEL  ; RK_02 U0_Y 电芯进料X轴轴原点搜索高速
D20039 CHANNEL  ; RK_02 U0_Y 电芯进料X轴轴原点搜索高速
D2004 CHANNEL  ; Hipot检测仪测试电压（HMI）
D20040 CHANNEL  ; RK_02 U0_Y 电芯进料X轴轴原点搜索接近速度
D20041 CHANNEL  ; RK_02 U0_Y 电芯进料X轴轴原点搜索接近速度
D20042 CHANNEL  ; RK_02 U0_Y 电芯进料X轴轴原点补偿值
D20043 CHANNEL  ; RK_02 U0_Y 电芯进料X轴轴原点补偿值
D20044 CHANNEL  ; RK_02 U0_Y 电芯进料X轴轴间隙补偿
D20045 CHANNEL  ; RK_02 U0_Y 电芯进料X轴轴间隙补偿速度
D20046 CHANNEL  ; RK_02 U0_Y 电芯进料X轴轴间隙补偿速度
D20047 CHANNEL  ; RK_02 U0_Y 电芯进料X轴轴加减速曲线
D20048 CHANNEL  ; RK_02 U0_Y 电芯进料X轴轴原点搜索加速时间
D20049 CHANNEL  ; RK_02 U0_Y 电芯进料X轴轴原点搜索加速时间
D2005 CHANNEL  ; Hipot测试仪测试电阻（HMI）
D20050 CHANNEL  ; RK_02 U0_Y 电芯进料X轴轴原点搜索减速时间
D20051 CHANNEL  ; RK_02 U0_Y 电芯进料X轴轴原点搜索减速时间
D20052 CHANNEL  ; RK_02 U0_Y 电芯进料X轴轴定位监测时间
D20053 CHANNEL  ; RK_02 U0_Y 电芯进料X轴轴负软限位
D20054 CHANNEL  ; RK_02 U0_Y 电芯进料X轴轴负软限位
D20055 CHANNEL  ; RK_02 U0_Y 电芯进料X轴轴正软限位
D20056 CHANNEL  ; RK_02 U0_Y 电芯进料X轴轴正软限位
D20057 CHANNEL  ; RK_02 U0_Y 电芯进料X轴轴为PCU保留
D20058 CHANNEL  ; RK_02 U0_Y 电芯进料X轴轴为PCU保留
D20059 CHANNEL  ; RK_02 U0_Y 电芯进料X轴轴初始脉冲定义
D20060 CHANNEL  ; RK_02 U0_Z 电芯进料Z轴轴输入输出设定
D20061 CHANNEL  ; RK_02 U0_Z 电芯进料Z轴轴操作模式选择
D20062 CHANNEL  ; RK_02 U0_Z 电芯进料Z轴轴最高速度
D20063 CHANNEL  ; RK_02 U0_Z 电芯进料Z轴轴最高速度
D20064 CHANNEL  ; RK_02 U0_Z 电芯进料Z轴轴初始速度
D20065 CHANNEL  ; RK_02 U0_Z 电芯进料Z轴轴初始速度
D20066 CHANNEL  ; RK_02 U0_Z 电芯进料Z轴轴原点搜索高速
D20067 CHANNEL  ; RK_02 U0_Z 电芯进料Z轴轴原点搜索高速
D20068 CHANNEL  ; RK_02 U0_Z 电芯进料Z轴轴原点搜索接近速度
D20069 CHANNEL  ; RK_02 U0_Z 电芯进料Z轴轴原点搜索接近速度
D2007 CHANNEL  ; Hipot检测仪测试电流（HMI）
D20070 CHANNEL  ; RK_02 U0_Z 电芯进料Z轴轴原点补偿值
D20071 CHANNEL  ; RK_02 U0_Z 电芯进料Z轴轴原点补偿值
D20072 CHANNEL  ; RK_02 U0_Z 电芯进料Z轴轴间隙补偿
D20073 CHANNEL  ; RK_02 U0_Z 电芯进料Z轴轴间隙补偿速度
D20074 CHANNEL  ; RK_02 U0_Z 电芯进料Z轴轴间隙补偿速度
D20075 CHANNEL  ; RK_02 U0_Z 电芯进料Z轴轴加减速曲线
D20076 CHANNEL  ; RK_02 U0_Z 电芯进料Z轴轴原点搜索加速时间
D20077 CHANNEL  ; RK_02 U0_Z 电芯进料Z轴轴原点搜索加速时间
D20078 CHANNEL  ; RK_02 U0_Z 电芯进料Z轴轴原点搜索减速时间
D20079 CHANNEL  ; RK_02 U0_Z 电芯进料Z轴轴原点搜索减速时间
D20080 CHANNEL  ; RK_02 U0_Z 电芯进料Z轴轴定位监测时间
D20081 CHANNEL  ; RK_02 U0_Z 电芯进料Z轴轴负软限位
D20082 CHANNEL  ; RK_02 U0_Z 电芯进料Z轴轴负软限位
D20083 CHANNEL  ; RK_02 U0_Z 电芯进料Z轴轴正软限位
D20084 CHANNEL  ; RK_02 U0_Z 电芯进料Z轴轴正软限位
D20085 CHANNEL  ; RK_02 U0_Z 电芯进料Z轴轴为PCU保留
D20086 CHANNEL  ; RK_02 U0_Z 电芯进料Z轴轴为PCU保留
D20087 CHANNEL  ; RK_02 U0_Z 电芯进料Z轴轴初始脉冲定义
D20088 CHANNEL  ; RK_03 U0_U 电芯上料X轴轴输入输出设定
D20089 CHANNEL  ; RK_03 U0_U 电芯上料X轴轴操作模式选择
D2009 CHANNEL  ; Hipot检测仪测试结果（HMI）
D20090 CHANNEL  ; RK_03 U0_U 电芯上料X轴轴最高速度
D20091 CHANNEL  ; RK_03 U0_U 电芯上料X轴轴最高速度
D20092 CHANNEL  ; RK_03 U0_U 电芯上料X轴轴初始速度
D20093 CHANNEL  ; RK_03 U0_U 电芯上料X轴轴初始速度
D20094 CHANNEL  ; RK_03 U0_U 电芯上料X轴轴原点搜索高速
D20095 CHANNEL  ; RK_03 U0_U 电芯上料X轴轴原点搜索高速
D20096 CHANNEL  ; RK_03 U0_U 电芯上料X轴轴原点搜索接近速度
D20097 CHANNEL  ; RK_03 U0_U 电芯上料X轴轴原点搜索接近速度
D20098 CHANNEL  ; RK_03 U0_U 电芯上料X轴轴原点补偿值
D20099 CHANNEL  ; RK_03 U0_U 电芯上料X轴轴原点补偿值
D20100 CHANNEL  ; RK_03 U0_U 电芯上料X轴轴间隙补偿
D20101 CHANNEL  ; RK_03 U0_U 电芯上料X轴轴间隙补偿速度
D20102 CHANNEL  ; RK_03 U0_U 电芯上料X轴轴间隙补偿速度
D20103 CHANNEL  ; RK_03 U0_U 电芯上料X轴轴加减速曲线
D20104 CHANNEL  ; RK_03 U0_U 电芯上料X轴轴原点搜索加速时间
D20105 CHANNEL  ; RK_03 U0_U 电芯上料X轴轴原点搜索加速时间
D20106 CHANNEL  ; RK_03 U0_U 电芯上料X轴轴原点搜索减速时间
D20107 CHANNEL  ; RK_03 U0_U 电芯上料X轴轴原点搜索减速时间
D20108 CHANNEL  ; RK_03 U0_U 电芯上料X轴轴定位监测时间
D20109 CHANNEL  ; RK_03 U0_U 电芯上料X轴轴负软限位
D20110 CHANNEL  ; RK_03 U0_U 电芯上料X轴轴负软限位
D20111 CHANNEL  ; RK_03 U0_U 电芯上料X轴轴正软限位
D20112 CHANNEL  ; RK_03 U0_U 电芯上料X轴轴正软限位
D20113 CHANNEL  ; RK_03 U0_U 电芯上料X轴轴为PCU保留
D20114 CHANNEL  ; RK_03 U0_U 电芯上料X轴轴为PCU保留
D20115 CHANNEL  ; RK_03 U0_U 电芯上料X轴轴初始脉冲定义
D20200 CHANNEL  ; U2- 操作数据区域定义
D20201 CHANNEL  ; U2- 操作数据区域开始字
D20202 CHANNEL  ; U2- 轴参数定义
D20203 CHANNEL  ; U2- 未被使用
D20204 CHANNEL  ; RK_05 U2_X #1入壳Y轴轴输入输出设定
D20205 CHANNEL  ; RK_05 U2_X #1入壳Y轴轴操作模式选择
D20206 CHANNEL  ; RK_05 U2_X #1入壳Y轴轴最高速度
D20207 CHANNEL  ; RK_05 U2_X #1入壳Y轴轴最高速度
D20208 CHANNEL  ; RK_05 U2_X #1入壳Y轴轴初始速度
D20209 CHANNEL  ; RK_05 U2_X #1入壳Y轴轴初始速度
D20210 CHANNEL  ; RK_05 U2_X #1入壳Y轴轴原点搜索高速
D20211 CHANNEL  ; RK_05 U2_X #1入壳Y轴轴原点搜索高速
D20212 CHANNEL  ; RK_05 U2_X #1入壳Y轴轴原点搜索接近速度
D20213 CHANNEL  ; RK_05 U2_X #1入壳Y轴轴原点搜索接近速度
D20214 CHANNEL  ; RK_05 U2_X #1入壳Y轴轴原点补偿值
D20215 CHANNEL  ; RK_05 U2_X #1入壳Y轴轴原点补偿值
D20216 CHANNEL  ; RK_05 U2_X #1入壳Y轴轴间隙补偿
D20217 CHANNEL  ; RK_05 U2_X #1入壳Y轴轴间隙补偿速度
D20218 CHANNEL  ; RK_05 U2_X #1入壳Y轴轴间隙补偿速度
D20219 CHANNEL  ; RK_05 U2_X #1入壳Y轴轴加减速曲线
D20220 CHANNEL  ; RK_05 U2_X #1入壳Y轴轴原点搜索加速时间
D20221 CHANNEL  ; RK_05 U2_X #1入壳Y轴轴原点搜索加速时间
D20222 CHANNEL  ; RK_05 U2_X #1入壳Y轴轴原点搜索减速时间
D20223 CHANNEL  ; RK_05 U2_X #1入壳Y轴轴原点搜索减速时间
D20224 CHANNEL  ; RK_05 U2_X #1入壳Y轴轴定位监测时间
D20225 CHANNEL  ; RK_05 U2_X #1入壳Y轴轴负软限位
D20226 CHANNEL  ; RK_05 U2_X #1入壳Y轴轴负软限位
D20227 CHANNEL  ; RK_05 U2_X #1入壳Y轴轴正软限位
D20228 CHANNEL  ; RK_05 U2_X #1入壳Y轴轴正软限位
D20229 CHANNEL  ; RK_05 U2_X #1入壳Y轴轴为PCU保留
D20230 CHANNEL  ; RK_05 U2_X #1入壳Y轴轴为PCU保留
D20231 CHANNEL  ; RK_05 U2_X #1入壳Y轴轴初始脉冲定义
D20232 CHANNEL  ; RK_05 U2_Y #2入壳Y轴轴输入输出设定
D20233 CHANNEL  ; RK_05 U2_Y #2入壳Y轴轴操作模式选择
D20234 CHANNEL  ; RK_05 U2_Y #2入壳Y轴轴最高速度
D20235 CHANNEL  ; RK_05 U2_Y #2入壳Y轴轴最高速度
D20236 CHANNEL  ; RK_05 U2_Y #2入壳Y轴轴初始速度
D20237 CHANNEL  ; RK_05 U2_Y #2入壳Y轴轴初始速度
D20238 CHANNEL  ; RK_05 U2_Y #2入壳Y轴轴原点搜索高速
D20239 CHANNEL  ; RK_05 U2_Y #2入壳Y轴轴原点搜索高速
D2024 CHANNEL  ; Hipot测试仪查询电压（HMI）
D20240 CHANNEL  ; RK_05 U2_Y #2入壳Y轴轴原点搜索接近速度
D20241 CHANNEL  ; RK_05 U2_Y #2入壳Y轴轴原点搜索接近速度
D20242 CHANNEL  ; RK_05 U2_Y #2入壳Y轴轴原点补偿值
D20243 CHANNEL  ; RK_05 U2_Y #2入壳Y轴轴原点补偿值
D20244 CHANNEL  ; RK_05 U2_Y #2入壳Y轴轴间隙补偿
D20245 CHANNEL  ; RK_05 U2_Y #2入壳Y轴轴间隙补偿速度
D20246 CHANNEL  ; RK_05 U2_Y #2入壳Y轴轴间隙补偿速度
D20247 CHANNEL  ; RK_05 U2_Y #2入壳Y轴轴加减速曲线
D20248 CHANNEL  ; RK_05 U2_Y #2入壳Y轴轴原点搜索加速时间
D20249 CHANNEL  ; RK_05 U2_Y #2入壳Y轴轴原点搜索加速时间
D2025 CHANNEL  ; Hipot检测仪查询电阻（HMI）
D20250 CHANNEL  ; RK_05 U2_Y #2入壳Y轴轴原点搜索减速时间
D20251 CHANNEL  ; RK_05 U2_Y #2入壳Y轴轴原点搜索减速时间
D20252 CHANNEL  ; RK_05 U2_Y #2入壳Y轴轴定位监测时间
D20253 CHANNEL  ; RK_05 U2_Y #2入壳Y轴轴负软限位
D20254 CHANNEL  ; RK_05 U2_Y #2入壳Y轴轴负软限位
D20255 CHANNEL  ; RK_05 U2_Y #2入壳Y轴轴正软限位
D20256 CHANNEL  ; RK_05 U2_Y #2入壳Y轴轴正软限位
D20257 CHANNEL  ; RK_05 U2_Y #2入壳Y轴轴为PCU保留
D20258 CHANNEL  ; RK_05 U2_Y #2入壳Y轴轴为PCU保留
D20259 CHANNEL  ; RK_05 U2_Y #2入壳Y轴轴初始脉冲定义
D2027 CHANNEL  ; Hipot检测仪查询电流（HMI）
D20400 CHANNEL  ; U4- 操作数据区域定义
D20401 CHANNEL  ; U4- 操作数据区域开始字
D20402 CHANNEL  ; U4- 轴参数定义
D20403 CHANNEL  ; U4- 未被使用
D20404 CHANNEL  ; RK_12 U4_X 预焊上下料X轴轴输入输出设定
D20405 CHANNEL  ; RK_12 U4_X 预焊上下料X轴轴操作模式选择
D20406 CHANNEL  ; RK_12 U4_X 预焊上下料X轴轴最高速度
D20407 CHANNEL  ; RK_12 U4_X 预焊上下料X轴轴最高速度
D20408 CHANNEL  ; RK_12 U4_X 预焊上下料X轴轴初始速度
D20409 CHANNEL  ; RK_12 U4_X 预焊上下料X轴轴初始速度
D2041 CHANNEL  ; Hipot检测仪查询电阻下限（HMI）
D20410 CHANNEL  ; RK_12 U4_X 预焊上下料X轴轴原点搜索高速
D20411 CHANNEL  ; RK_12 U4_X 预焊上下料X轴轴原点搜索高速
D20412 CHANNEL  ; RK_12 U4_X 预焊上下料X轴轴原点搜索接近速度
D20413 CHANNEL  ; RK_12 U4_X 预焊上下料X轴轴原点搜索接近速度
D20414 CHANNEL  ; RK_12 U4_X 预焊上下料X轴轴原点补偿值
D20415 CHANNEL  ; RK_12 U4_X 预焊上下料X轴轴原点补偿值
D20416 CHANNEL  ; RK_12 U4_X 预焊上下料X轴轴间隙补偿
D20417 CHANNEL  ; RK_12 U4_X 预焊上下料X轴轴间隙补偿速度
D20418 CHANNEL  ; RK_12 U4_X 预焊上下料X轴轴间隙补偿速度
D20419 CHANNEL  ; RK_12 U4_X 预焊上下料X轴轴加减速曲线
D20420 CHANNEL  ; RK_12 U4_X 预焊上下料X轴轴原点搜索加速时间
D20421 CHANNEL  ; RK_12 U4_X 预焊上下料X轴轴原点搜索加速时间
D20422 CHANNEL  ; RK_12 U4_X 预焊上下料X轴轴原点搜索减速时间
D20423 CHANNEL  ; RK_12 U4_X 预焊上下料X轴轴原点搜索减速时间
D20424 CHANNEL  ; RK_12 U4_X 预焊上下料X轴轴定位监测时间
D20425 CHANNEL  ; RK_12 U4_X 预焊上下料X轴轴负软限位
D20426 CHANNEL  ; RK_12 U4_X 预焊上下料X轴轴负软限位
D20427 CHANNEL  ; RK_12 U4_X 预焊上下料X轴轴正软限位
D20428 CHANNEL  ; RK_12 U4_X 预焊上下料X轴轴正软限位
D20429 CHANNEL  ; RK_12 U4_X 预焊上下料X轴轴为PCU保留
D2043 CHANNEL  ; Hipot检测仪查询电阻上限（HMI）
D20430 CHANNEL  ; RK_12 U4_X 预焊上下料X轴轴为PCU保留
D20431 CHANNEL  ; RK_12 U4_X 预焊上下料X轴轴初始脉冲定义
D20432 CHANNEL  ; RK_12 U4_Y 预焊上料Z轴轴输入输出设定
D20433 CHANNEL  ; RK_12 U4_Y 预焊上料Z轴轴操作模式选择
D20434 CHANNEL  ; RK_12 U4_Y 预焊上料Z轴轴最高速度
D20435 CHANNEL  ; RK_12 U4_Y 预焊上料Z轴轴最高速度
D20436 CHANNEL  ; RK_12 U4_Y 预焊上料Z轴轴初始速度
D20437 CHANNEL  ; RK_12 U4_Y 预焊上料Z轴轴初始速度
D20438 CHANNEL  ; RK_12 U4_Y 预焊上料Z轴轴原点搜索高速
D20439 CHANNEL  ; RK_12 U4_Y 预焊上料Z轴轴原点搜索高速
D20440 CHANNEL  ; RK_12 U4_Y 预焊上料Z轴轴原点搜索接近速度
D20441 CHANNEL  ; RK_12 U4_Y 预焊上料Z轴轴原点搜索接近速度
D20442 CHANNEL  ; RK_12 U4_Y 预焊上料Z轴轴原点补偿值
D20443 CHANNEL  ; RK_12 U4_Y 预焊上料Z轴轴原点补偿值
D20444 CHANNEL  ; RK_12 U4_Y 预焊上料Z轴轴间隙补偿
D20445 CHANNEL  ; RK_12 U4_Y 预焊上料Z轴轴间隙补偿速度
D20446 CHANNEL  ; RK_12 U4_Y 预焊上料Z轴轴间隙补偿速度
D20447 CHANNEL  ; RK_12 U4_Y 预焊上料Z轴轴加减速曲线
D20448 CHANNEL  ; RK_12 U4_Y 预焊上料Z轴轴原点搜索加速时间
D20449 CHANNEL  ; RK_12 U4_Y 预焊上料Z轴轴原点搜索加速时间
D2045 CHANNEL  ; Hipot检测仪查询测试时间（HMI）
D20450 CHANNEL  ; RK_12 U4_Y 预焊上料Z轴轴原点搜索减速时间
D20451 CHANNEL  ; RK_12 U4_Y 预焊上料Z轴轴原点搜索减速时间
D20452 CHANNEL  ; RK_12 U4_Y 预焊上料Z轴轴定位监测时间
D20453 CHANNEL  ; RK_12 U4_Y 预焊上料Z轴轴负软限位
D20454 CHANNEL  ; RK_12 U4_Y 预焊上料Z轴轴负软限位
D20455 CHANNEL  ; RK_12 U4_Y 预焊上料Z轴轴正软限位
D20456 CHANNEL  ; RK_12 U4_Y 预焊上料Z轴轴正软限位
D20457 CHANNEL  ; RK_12 U4_Y 预焊上料Z轴轴为PCU保留
D20458 CHANNEL  ; RK_12 U4_Y 预焊上料Z轴轴为PCU保留
D20459 CHANNEL  ; RK_12 U4_Y 预焊上料Z轴轴初始脉冲定义
D20460 CHANNEL  ; RK_12 U4_Z 预焊下料Z轴轴输入输出设定
D20461 CHANNEL  ; RK_12 U4_Z 预焊下料Z轴轴操作模式选择
D20462 CHANNEL  ; RK_12 U4_Z 预焊下料Z轴轴最高速度
D20463 CHANNEL  ; RK_12 U4_Z 预焊下料Z轴轴最高速度
D20464 CHANNEL  ; RK_12 U4_Z 预焊下料Z轴轴初始速度
D20465 CHANNEL  ; RK_12 U4_Z 预焊下料Z轴轴初始速度
D20466 CHANNEL  ; RK_12 U4_Z 预焊下料Z轴轴原点搜索高速
D20467 CHANNEL  ; RK_12 U4_Z 预焊下料Z轴轴原点搜索高速
D20468 CHANNEL  ; RK_12 U4_Z 预焊下料Z轴轴原点搜索接近速度
D20469 CHANNEL  ; RK_12 U4_Z 预焊下料Z轴轴原点搜索接近速度
D20470 CHANNEL  ; RK_12 U4_Z 预焊下料Z轴轴原点补偿值
D20471 CHANNEL  ; RK_12 U4_Z 预焊下料Z轴轴原点补偿值
D20472 CHANNEL  ; RK_12 U4_Z 预焊下料Z轴轴间隙补偿
D20473 CHANNEL  ; RK_12 U4_Z 预焊下料Z轴轴间隙补偿速度
D20474 CHANNEL  ; RK_12 U4_Z 预焊下料Z轴轴间隙补偿速度
D20475 CHANNEL  ; RK_12 U4_Z 预焊下料Z轴轴加减速曲线
D20476 CHANNEL  ; RK_12 U4_Z 预焊下料Z轴轴原点搜索加速时间
D20477 CHANNEL  ; RK_12 U4_Z 预焊下料Z轴轴原点搜索加速时间
D20478 CHANNEL  ; RK_12 U4_Z 预焊下料Z轴轴原点搜索减速时间
D20479 CHANNEL  ; RK_12 U4_Z 预焊下料Z轴轴原点搜索减速时间
D20480 CHANNEL  ; RK_12 U4_Z 预焊下料Z轴轴定位监测时间
D20481 CHANNEL  ; RK_12 U4_Z 预焊下料Z轴轴负软限位
D20482 CHANNEL  ; RK_12 U4_Z 预焊下料Z轴轴负软限位
D20483 CHANNEL  ; RK_12 U4_Z 预焊下料Z轴轴正软限位
D20484 CHANNEL  ; RK_12 U4_Z 预焊下料Z轴轴正软限位
D20485 CHANNEL  ; RK_12 U4_Z 预焊下料Z轴轴为PCU保留
D20486 CHANNEL  ; RK_12 U4_Z 预焊下料Z轴轴为PCU保留
D20487 CHANNEL  ; RK_12 U4_Z 预焊下料Z轴轴初始脉冲定义
D20488 CHANNEL  ; RK_13 U4_U #1移载Y轴轴输入输出设定
D20489 CHANNEL  ; RK_13 U4_U #1移载Y轴轴操作模式选择
D20490 CHANNEL  ; RK_13 U4_U #1移载Y轴轴最高速度
D20491 CHANNEL  ; RK_13 U4_U #1移载Y轴轴最高速度
D20492 CHANNEL  ; RK_13 U4_U #1移载Y轴轴初始速度
D20493 CHANNEL  ; RK_13 U4_U #1移载Y轴轴初始速度
D20494 CHANNEL  ; RK_13 U4_U #1移载Y轴轴原点搜索高速
D20495 CHANNEL  ; RK_13 U4_U #1移载Y轴轴原点搜索高速
D20496 CHANNEL  ; RK_13 U4_U #1移载Y轴轴原点搜索接近速度
D20497 CHANNEL  ; RK_13 U4_U #1移载Y轴轴原点搜索接近速度
D20498 CHANNEL  ; RK_13 U4_U #1移载Y轴轴原点补偿值
D20499 CHANNEL  ; RK_13 U4_U #1移载Y轴轴原点补偿值
D20500 CHANNEL  ; RK_13 U4_U #1移载Y轴轴间隙补偿
D20501 CHANNEL  ; RK_13 U4_U #1移载Y轴轴间隙补偿速度
D20502 CHANNEL  ; RK_13 U4_U #1移载Y轴轴间隙补偿速度
D20503 CHANNEL  ; RK_13 U4_U #1移载Y轴轴加减速曲线
D20504 CHANNEL  ; RK_13 U4_U #1移载Y轴轴原点搜索加速时间
D20505 CHANNEL  ; RK_13 U4_U #1移载Y轴轴原点搜索加速时间
D20506 CHANNEL  ; RK_13 U4_U #1移载Y轴轴原点搜索减速时间
D20507 CHANNEL  ; RK_13 U4_U #1移载Y轴轴原点搜索减速时间
D20508 CHANNEL  ; RK_13 U4_U #1移载Y轴轴定位监测时间
D20509 CHANNEL  ; RK_13 U4_U #1移载Y轴轴负软限位
D20510 CHANNEL  ; RK_13 U4_U #1移载Y轴轴负软限位
D20511 CHANNEL  ; RK_13 U4_U #1移载Y轴轴正软限位
